// TIA Portal V20 export
// export: Created 2025-12-01T14:56:31.3857543Z, ExportSetting None, DisplayName Totally Integrated Automation Portal, DisplayVersion V20 Update 3, DisplayName TIA Portal Openness, DisplayVersion V20 Update 3, DisplayName TIA Portal Version Control Interface, DisplayVersion V20 Update 3, DisplayName STEP 7 Professional, DisplayVersion V20 Update 3, DisplayName STEP 7 Safety, DisplayVersion V20 Update 2, DisplayName WinCC Basic/Comfort/Advanced, DisplayVersion V20 Update 3, DisplayName WinCC Professional, DisplayVersion V20 Update 3, DisplayName WinCC Unified, DisplayVersion V20 Update 3
FUNCTION_BLOCK "FB438_CRTL_W_E1_S234_BLOQ_OrdJDT"   // FB438, LAD
TITLE = Control del Ramal de Salidas
{ S7_Optimized_Access := 'FALSE' }
AUTHOR : ROUTERA
NAME : 20190213
VERSION : 3.1
// stored: AutoNumber false, SetENOAutomatically false
   VAR_INPUT
      Mesa : UInt;   // Número de mesa
      En_Tension : Bool;
      pHsMx_E1 : Bool;   // pHs DE PRESENCIA de la Mesa en E1
      pHsMx_S2 : Bool;   // pHs DE AUSENCIA de la Mesa en S2
      pHsMx_S3 : Bool;   // pHs DE AUSENCIA de la Mesa en S3
      pHsMx_S4 : Bool;   // pHs DE AUSENCIA de la Mesa en S4
      Pos_WS_S2 : Bool;   // posición del desviador en S2
      Pos_WS_S3 : Bool;   // posición del desviador en S3
      Pos_WS_S4 : Bool;   // posición del desviador en S4
      Termico_E1E3 : Bool;   // Proteccion del Tx en E1E3
      Avance_Tx_Ent { ExternalVisible := 'False'} : Bool;   // Avance del Tx de entrada. Primer tramo
      Avance_Tx_Sal : Bool;   // Avance del Tx de salida.
      PTF_Sal_M2 : Bool;   // S2 >> Mesa Siguiente PTF
      NXT_Avance_S2 : Bool;   // S2 >> Mesa Siguiente avanzando
      PTF_Sal_M3 : Bool;   // S3 >> Mesa Siguiente PTF
      NXT_Avance_S3 : Bool;   // S3 >> Mesa Siguiente avanzando
      PTF_Sal_M4 : Bool;   // S4 >> Mesa Siguiente PTF
      NXT_Avance_S4 : Bool;   // S4 >> Mesa Siguiente avanzando
      F_EnvMens_Mx : Bool;   // Fin de Envio de Mensaje
      Mx_Bloq_Activo : Bool;   // Bloqueo Activo de la Mesa
      MX_FlujoPrin_S2 : Bool;   // El flujo principal es Saliendo por S2
      MX_FlujoPrin_S4 : Bool;   // El flujo principal es Saliendo por S4
      AVTF_MAnt_Mx : Bool;   // E1 >> Mesa Anterior AVTF
      Habilitar_orden_JDT : Bool := false;   // El JDT tendrá el control del cruce con orden
      Num_Cruce : UInt;   // Número de cruce.
      DB_FIFO_Cruce : UInt := 213;   // DB de la FIFO de ordenes del cruce
      Lng_FIFO_Cruce : UInt := 1;   // Longitut de la FIFO de ordenes del cruce
      Valor_Orden_S2 : Word := 16#81;   // Con que orden entra por S2
      Valor_Orden_S4 : Word := 16#82;   // Con que orden entra por S4
      MesaS2 : UInt;   // Número de mesa por S2
      MesaS3 : UInt;   // Número de mesa por S3
      MesaS4 : UInt;   // Número de mesa por S4
      V_CNT_pHsMx : UDInt := 500;   // Valor de Presencia en ms
      V_Vaciado : UDInt := 5000;   // Valor de vaciado en ms
      V_TOut_Desviador : UDInt := 2000;   // en ms
      V_TOut_Tx_Mx : UDInt := 3000;   // TimeOut de Atasco en ms
      V_CNT_ApHsMx_E1 : UDInt := 250;   // Valor de Ausencia por E1 en ms
      V_CNT_ApHsMx_S2 : UDInt := 250;   // Valor de Ausencia por S2 en ms
      V_CNT_ApHsMx_S3 : UDInt := 250;   // Valor de Ausencia por S3 en ms
      V_CNT_ApHsMx_S4 : UDInt := 250;   // Valor de Ausencia por S4 en ms
      V_Orden_bloqueo : UDInt := 3000;   // en ms
   END_VAR
   VAR_OUTPUT
      P_EnvMens_PMx : Bool;   // Permiso de Enviar Mensaje de Presencia
      Etiqueta_Jdt : UDInt;   // Etiqueta que ha sido leida
      Orden_Ejecutada_Jdt : UInt;   // Orden que se ha ejecutado
      PTF_MAnt_Mx : Bool;   // E1 >> Mesa Anterior PTF
      AVTF_Sal_M2 : Bool;   // S2 >> Mesa Siguiente AVTF
      NXT_Descarga_Act_S2 : Bool;   // S2 >> Mesa Siguiente descarga activa
      AVTF_Sal_M3 : Bool;   // S3 >> Mesa Siguiente AVTF
      NXT_Descarga_Act_S3 : Bool;   // S3 >> Mesa Siguiente descarga activa
      AVTF_Sal_M4 : Bool;   // S4 >> Mesa Siguiente AVTF
      NXT_Descarga_Act_S4 : Bool;   // S4 >> Mesa Siguiente descarga activa
   END_VAR
   VAR
      T1_ET00 : Bool;   // Reset
      T1_ET08 : Bool;
      T1_ET01 : Bool;   // Entrada Vacia
      T1_ET10 : Bool;   // Carga Entrada
      T1_ET02 : Bool;   // Entrada Cargada
      T1_ET02_JDT : Bool;
      T1_ET03 : Bool;   // Vaciando Entrada
      T1_ET20 : Bool;   // Carga Salida
      T1_ET21 : Bool;   // Salida Vacia
      T1_ET50 : Bool;   // Continuar
      T1_ET60 : Bool;   // Entrar
      T1_ET70 : Bool;   // Vaciado
      T1_ET80 : Bool;
      T1_ET110 : Bool;   // Extraer orden
      T1_ET111 : Bool;
      T1_ET112 : Bool;
      FP_ET2_JDT : Bool;
      FIFO_OK : Bool;
      TRANS_OK : Bool;
      O_Bloqueo : Bool;
      Vaciado_1 : Bool;
      PRV_CargaOK_ET03 : Bool;
      FN_ET20 : Bool;
      MemoPresenciaJDT : Bool;
      maux_fp_disparo : Bool;
      Vaciado_entrada_ok : Bool;
      Vaciado_salida_s2_ok : Bool;
      Vaciado_salida_s3_ok : Bool;
      Vaciado_salida_s4_ok : Bool;
      Maux_FN_Phs_S2 : Bool;
      mem_fn_phs_s2 : Bool;
      Maux_FN_Phs_E1 : Bool;
      mem_fn_phs_e1 : Bool;
      Maux_FP_phs_S3 : Bool;
      mem_fp_phs_s3 : Bool;
      Maux_FN_Phs_S4 : Bool;
      mem_fn_phs_s4 : Bool;
      paro : Bool;
      CNT_ERR_PHS : Int;
      TIMV_WS_E1 : UDInt;
      TIMV_WS_S2 : UDInt;
      TIMV_WS_S3 : UDInt;
      TIMV_WS_S4 : UDInt;
      TMP_Err_Piston : UDInt;
      TMP_Paro : UDInt;
      TMP_Err_Tout_avance_E : UDInt;
      TMP_Err_Tout_avance_S : UDInt;
      CNT_pHs_WS : UDInt;
      CNT_aus_s2 : UDInt;
      CNT_aus_s4 : UDInt;
      CNT_aus_e1 : UDInt;
      CNT_pres_s3 : UDInt;
      CNT_bloqueo : UDInt;
      TMP_En_tension : UDInt;
      Datos_Scanner { S7_SetPoint := 'True'} : "ROUT_Orden_Fifo_Scanner";
   END_VAR
   VAR_TEMP
      EstadoZona : "EstadoZona";   // Estado de Zona de la Mesa
      EstadoVI : "EstadosMesa";   // Estado del Vehiculo Inteliguente de la Mesa
      ConfigFB : "UDT_ConfigFB";   // Configuracion de la FB de la Mesa
      TEMP_ET00 : Bool;
      O_Salir_S3 : Bool;
      O_Salir_S2 : Bool;
      O_Salir_S4 : Bool;
      O_Vaciar : Bool;
      cnt_phs_ok : Bool;
      OK_Aus_S2 : Bool;
      OK_Aus_E1 : Bool;
      OK_Pres_S3 : Bool;
      OK_Aus_S4 : Bool;
      atasco_entrada : Bool;
      atasco_salida : Bool;
      ok_tension : Bool;
      Aux_W_Moti : Word;
      Moti_INIC : Bool;
      Moti_ERRO : Bool;
      Moti_NENC : Bool;
      Moti_NORM : Bool;
      ok_bloqueo : Bool;
      timeout_piston : Bool;
      O_S2_JDT : Bool;
      O_S3_JDT : Bool;
      O_S4_JDT : Bool;
      I_V_Ord_Salir_S2 : UInt;
      I_V_Ord_Salir_S4 : UInt;
      I_Ord_Filtrada : UInt;
      INT_ORDEN : UInt;
      Aux_W_Orden : Word;
      retval : Int;
   END_VAR
   VAR_TEMP   // added for the SCL form of the ladder/FBD networks
      _w1 : Bool;
      _w2 : Bool;
      _w3 : Bool;
      _w4 : Bool;
      _w5 : Bool;
      _w6 : Bool;
      _w7 : Bool;
   END_VAR
BEGIN

REGION Network 1: INICIALIZAR - Recoger las Variables de Estado de la Mesa
   // Se recoge - Estado_CBx
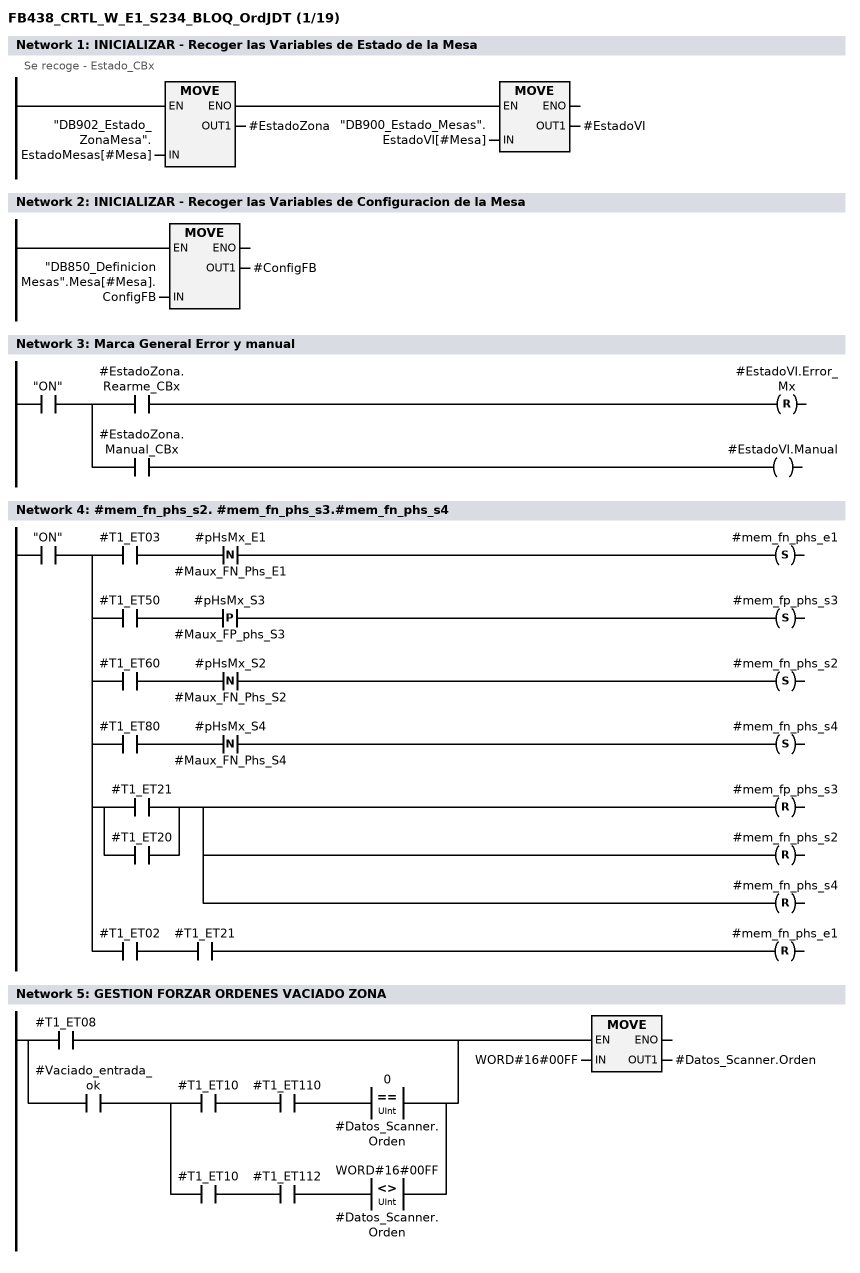
   RUNG wire#powerrail
      Move(in := "DB902_Estado_ZonaMesa".EstadoMesas[#Mesa], out1 => #EstadoZona)
      Move(in := "DB900_Estado_Mesas".EstadoVI[#Mesa], out1 => #EstadoVI)
   END_RUNG
   // the same network as SCL:
   #EstadoZona := "DB902_Estado_ZonaMesa".EstadoMesas[#Mesa];
   #EstadoVI := "DB900_Estado_Mesas".EstadoVI[#Mesa];
END_REGION

REGION Network 2: INICIALIZAR - Recoger las Variables de Configuracion de la Mesa
   RUNG wire#powerrail
      Move(in := "DB850_DefinicionMesas".Mesa[#Mesa].ConfigFB, out1 => #ConfigFB)
   END_RUNG
   // the same network as SCL:
   #ConfigFB := "DB850_DefinicionMesas".Mesa[#Mesa].ConfigFB;
END_REGION

REGION Network 3: Marca General Error y manual
   RUNG wire#powerrail
      Contact( "ON" )
      wire#w1
      Contact( #EstadoZona.Rearme_CBx )
      R_Coil( #EstadoVI.Error_Mx )
   END_RUNG
   RUNG wire#w1
      Contact( #EstadoZona.Manual_CBx )
      Coil( #EstadoVI.Manual )
   END_RUNG
   // the same network as SCL:
   IF "ON" AND #EstadoZona.Rearme_CBx THEN #EstadoVI.Error_Mx := FALSE; END_IF;
   #EstadoVI.Manual := "ON" AND #EstadoZona.Manual_CBx;
END_REGION

REGION Network 4: #mem_fn_phs_s2. #mem_fn_phs_s3.#mem_fn_phs_s4
   RUNG wire#powerrail
      Contact( "ON" )
      wire#w1
      Contact( #T1_ET03 )
      N_Contact(operand := #pHsMx_E1, bit := #Maux_FN_Phs_E1)
      S_Coil( #mem_fn_phs_e1 )
   END_RUNG
   RUNG wire#w1
      Contact( #T1_ET50 )
      P_Contact(operand := #pHsMx_S3, bit := #Maux_FP_phs_S3)
      S_Coil( #mem_fp_phs_s3 )
   END_RUNG
   RUNG wire#w1
      Contact( #T1_ET60 )
      N_Contact(operand := #pHsMx_S2, bit := #Maux_FN_Phs_S2)
      S_Coil( #mem_fn_phs_s2 )
   END_RUNG
   RUNG wire#w1
      Contact( #T1_ET80 )
      N_Contact(operand := #pHsMx_S4, bit := #Maux_FN_Phs_S4)
      S_Coil( #mem_fn_phs_s4 )
   END_RUNG
   RUNG wire#w1
      Contact( #T1_ET21 )
      wire#w2
      R_Coil( #mem_fp_phs_s3 )
   END_RUNG
   RUNG wire#w1
      Contact( #T1_ET20 )
   END_RUNG wire#w2
   RUNG wire#w2
      R_Coil( #mem_fn_phs_s2 )
   END_RUNG
   RUNG wire#w2
      R_Coil( #mem_fn_phs_s4 )
   END_RUNG
   RUNG wire#w1
      Contact( #T1_ET02 )
      Contact( #T1_ET21 )
      R_Coil( #mem_fn_phs_e1 )
   END_RUNG
   // the same network as SCL:
   #_w1 := "ON" AND #T1_ET03 AND NOT #pHsMx_E1 AND #Maux_FN_Phs_E1;   // falling edge of #pHsMx_E1
   #Maux_FN_Phs_E1 := #pHsMx_E1;
   IF #_w1 THEN #mem_fn_phs_e1 := TRUE; END_IF;
   #_w2 := "ON" AND #T1_ET50 AND #pHsMx_S3 AND NOT #Maux_FP_phs_S3;   // rising edge of #pHsMx_S3
   #Maux_FP_phs_S3 := #pHsMx_S3;
   IF #_w2 THEN #mem_fp_phs_s3 := TRUE; END_IF;
   #_w3 := "ON" AND #T1_ET60 AND NOT #pHsMx_S2 AND #Maux_FN_Phs_S2;   // falling edge of #pHsMx_S2
   #Maux_FN_Phs_S2 := #pHsMx_S2;
   IF #_w3 THEN #mem_fn_phs_s2 := TRUE; END_IF;
   #_w4 := "ON" AND #T1_ET80 AND NOT #pHsMx_S4 AND #Maux_FN_Phs_S4;   // falling edge of #pHsMx_S4
   #Maux_FN_Phs_S4 := #pHsMx_S4;
   IF #_w4 THEN #mem_fn_phs_s4 := TRUE; END_IF;
   IF "ON" AND (#T1_ET21 OR #T1_ET20) THEN
       #mem_fp_phs_s3 := FALSE;
       #mem_fn_phs_s2 := FALSE;
       #mem_fn_phs_s4 := FALSE;
   END_IF;
   IF "ON" AND #T1_ET02 AND #T1_ET21 THEN #mem_fn_phs_e1 := FALSE; END_IF;
END_REGION

REGION Network 5: GESTION FORZAR ORDENES VACIADO ZONA
   RUNG wire#powerrail
      Contact( #T1_ET08 )
      wire#w1
      { S7_GenerateENO := "TRUE" } Move(in := WORD#16#00FF, out1 => #Datos_Scanner.Orden)
   END_RUNG
   RUNG wire#powerrail
      Contact( #Vaciado_entrada_ok )
      wire#w2
      Contact( #T1_ET10 )
      Contact( #T1_ET110 )
      { S7_Templates := "SrcType := UInt" } EQ_Contact(in1 := 0, in2 := #Datos_Scanner.Orden)
   END_RUNG wire#w1
   RUNG wire#w2
      Contact( #T1_ET10 )
      Contact( #T1_ET112 )
      { S7_Templates := "SrcType := UInt" } NE_Contact(in1 := WORD#16#00FF, in2 := #Datos_Scanner.Orden)
   END_RUNG wire#w1
   // the same network as SCL:
   IF #T1_ET08 OR (#Vaciado_entrada_ok AND ((#T1_ET10 AND #T1_ET110 AND (0 = #Datos_Scanner.Orden)) OR (#T1_ET10 AND #T1_ET112 AND (WORD#16#00FF <> #Datos_Scanner.Orden)))) THEN
       #Datos_Scanner.Orden := WORD#16#00FF;
   END_IF;
END_REGION

REGION Network 6: Ordenes del JDT
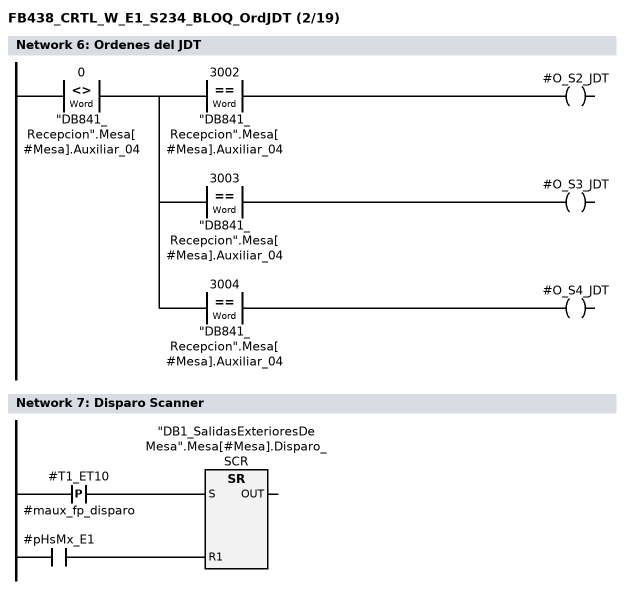
   RUNG wire#powerrail
      { S7_Templates := "SrcType := Word" } NE_Contact(in1 := 0, in2 := "DB841_Recepcion".Mesa[#Mesa].Auxiliar_04)
      wire#w1
      { S7_Templates := "SrcType := Word" } EQ_Contact(in1 := 3002, in2 := "DB841_Recepcion".Mesa[#Mesa].Auxiliar_04)
      Coil( #O_S2_JDT )
   END_RUNG
   RUNG wire#w1
      { S7_Templates := "SrcType := Word" } EQ_Contact(in1 := 3003, in2 := "DB841_Recepcion".Mesa[#Mesa].Auxiliar_04)
      Coil( #O_S3_JDT )
   END_RUNG
   RUNG wire#w1
      { S7_Templates := "SrcType := Word" } EQ_Contact(in1 := 3004, in2 := "DB841_Recepcion".Mesa[#Mesa].Auxiliar_04)
      Coil( #O_S4_JDT )
   END_RUNG
   // the same network as SCL:
   #_w1 := 0 <> "DB841_Recepcion".Mesa[#Mesa].Auxiliar_04;
   #O_S2_JDT := #_w1 AND (3002 = "DB841_Recepcion".Mesa[#Mesa].Auxiliar_04);
   #O_S3_JDT := #_w1 AND (3003 = "DB841_Recepcion".Mesa[#Mesa].Auxiliar_04);
   #O_S4_JDT := #_w1 AND (3004 = "DB841_Recepcion".Mesa[#Mesa].Auxiliar_04);
END_REGION

REGION Network 7: Disparo Scanner
   RUNG wire#powerrail
      P_Contact(operand := #T1_ET10, bit := #maux_fp_disparo)
      S_SR(operand := "DB1_SalidasExterioresDeMesa".Mesa[#Mesa].Disparo_SCR, r1 := wire#w1)
   END_RUNG
   RUNG wire#powerrail
      Contact( #pHsMx_E1 )
   END_RUNG wire#w1
   // the same network as SCL:
   #_w1 := #T1_ET10 AND NOT #maux_fp_disparo;   // rising edge of #T1_ET10
   #maux_fp_disparo := #T1_ET10;
   IF #_w1 THEN
       "DB1_SalidasExterioresDeMesa".Mesa[#Mesa].Disparo_SCR := TRUE;   // SR flip-flop
   END_IF;
   IF #pHsMx_E1 THEN "DB1_SalidasExterioresDeMesa".Mesa[#Mesa].Disparo_SCR := FALSE; END_IF;
END_REGION

REGION Network 8: extraer orden
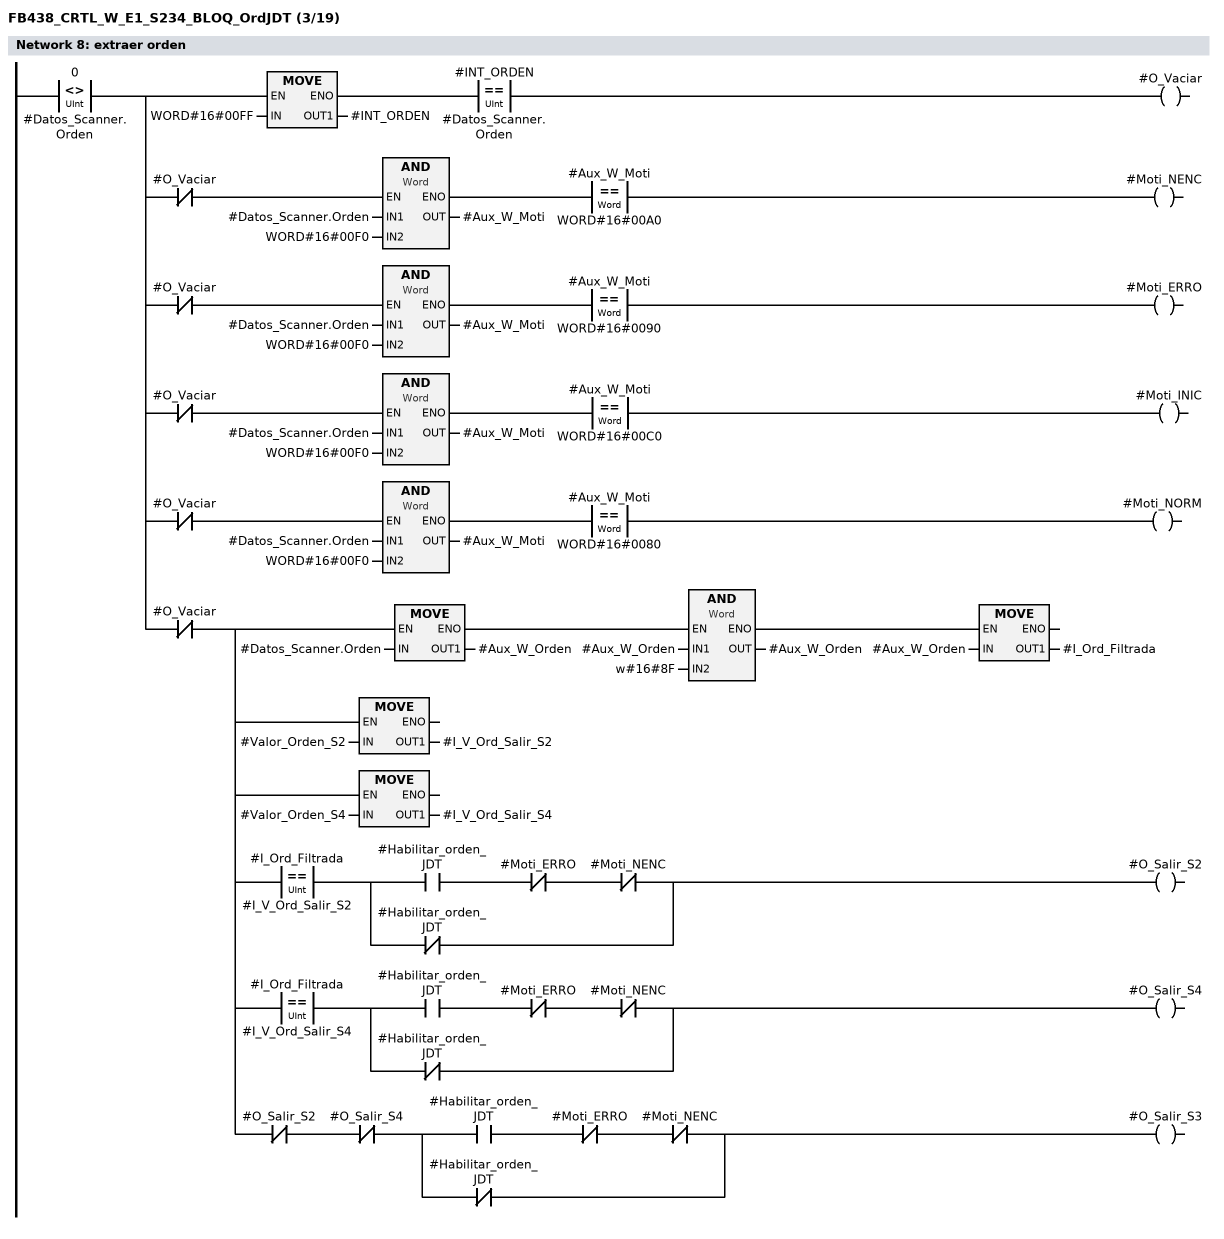
   RUNG wire#powerrail
      { S7_Templates := "SrcType := UInt" } NE_Contact(in1 := 0, in2 := #Datos_Scanner.Orden)
      wire#w1
      { S7_GenerateENO := "TRUE" } Move(in := WORD#16#00FF, out1 => #INT_ORDEN)
      { S7_Templates := "SrcType := UInt" } EQ_Contact(in1 := #INT_ORDEN, in2 := #Datos_Scanner.Orden)
      Coil( #O_Vaciar )
   END_RUNG
   RUNG wire#w1
      I_Contact( #O_Vaciar )
      { S7_Templates := "SrcType := Word"; S7_GenerateENO := "TRUE" } And(in1 := #Datos_Scanner.Orden, in2 := WORD#16#00F0, out => #Aux_W_Moti)
      { S7_Templates := "SrcType := Word" } EQ_Contact(in1 := #Aux_W_Moti, in2 := WORD#16#00A0)
      Coil( #Moti_NENC )
   END_RUNG
   RUNG wire#w1
      I_Contact( #O_Vaciar )
      { S7_Templates := "SrcType := Word"; S7_GenerateENO := "TRUE" } And(in1 := #Datos_Scanner.Orden, in2 := WORD#16#00F0, out => #Aux_W_Moti)
      { S7_Templates := "SrcType := Word" } EQ_Contact(in1 := #Aux_W_Moti, in2 := WORD#16#0090)
      Coil( #Moti_ERRO )
   END_RUNG
   RUNG wire#w1
      I_Contact( #O_Vaciar )
      { S7_Templates := "SrcType := Word"; S7_GenerateENO := "TRUE" } And(in1 := #Datos_Scanner.Orden, in2 := WORD#16#00F0, out => #Aux_W_Moti)
      { S7_Templates := "SrcType := Word" } EQ_Contact(in1 := #Aux_W_Moti, in2 := WORD#16#00C0)
      Coil( #Moti_INIC )
   END_RUNG
   RUNG wire#w1
      I_Contact( #O_Vaciar )
      { S7_Templates := "SrcType := Word"; S7_GenerateENO := "TRUE" } And(in1 := #Datos_Scanner.Orden, in2 := WORD#16#00F0, out => #Aux_W_Moti)
      { S7_Templates := "SrcType := Word" } EQ_Contact(in1 := #Aux_W_Moti, in2 := WORD#16#0080)
      Coil( #Moti_NORM )
   END_RUNG
   RUNG wire#w1
      I_Contact( #O_Vaciar )
      wire#w2
      { S7_GenerateENO := "TRUE" } Move(in := #Datos_Scanner.Orden, out1 => #Aux_W_Orden)
      { S7_Templates := "SrcType := Word"; S7_GenerateENO := "TRUE" } And(in1 := #Aux_W_Orden, in2 := w#16#8F, out => #Aux_W_Orden)
      { S7_GenerateENO := "TRUE" } Move(in := #Aux_W_Orden, out1 => #I_Ord_Filtrada)
   END_RUNG
   RUNG wire#w2
      { S7_GenerateENO := "TRUE" } Move(in := #Valor_Orden_S2, out1 => #I_V_Ord_Salir_S2)
   END_RUNG
   RUNG wire#w2
      { S7_GenerateENO := "TRUE" } Move(in := #Valor_Orden_S4, out1 => #I_V_Ord_Salir_S4)
   END_RUNG
   RUNG wire#w2
      { S7_Templates := "SrcType := UInt" } EQ_Contact(in1 := #I_Ord_Filtrada, in2 := #I_V_Ord_Salir_S2)
      wire#w3
      Contact( #Habilitar_orden_JDT )
      I_Contact( #Moti_ERRO )
      I_Contact( #Moti_NENC )
      wire#w4
      Coil( #O_Salir_S2 )
   END_RUNG
   RUNG wire#w3
      I_Contact( #Habilitar_orden_JDT )
   END_RUNG wire#w4
   RUNG wire#w2
      { S7_Templates := "SrcType := UInt" } EQ_Contact(in1 := #I_Ord_Filtrada, in2 := #I_V_Ord_Salir_S4)
      wire#w5
      Contact( #Habilitar_orden_JDT )
      I_Contact( #Moti_ERRO )
      I_Contact( #Moti_NENC )
      wire#w6
      Coil( #O_Salir_S4 )
   END_RUNG
   RUNG wire#w5
      I_Contact( #Habilitar_orden_JDT )
   END_RUNG wire#w6
   RUNG wire#w2
      I_Contact( #O_Salir_S2 )
      I_Contact( #O_Salir_S4 )
      wire#w7
      Contact( #Habilitar_orden_JDT )
      I_Contact( #Moti_ERRO )
      I_Contact( #Moti_NENC )
      wire#w8
      Coil( #O_Salir_S3 )
   END_RUNG
   RUNG wire#w7
      I_Contact( #Habilitar_orden_JDT )
   END_RUNG wire#w8
   // the same network as SCL:
   // ENO of a box is taken as its EN; it also drops when the box reports an error
   #_w1 := 0 <> #Datos_Scanner.Orden;
   IF #_w1 THEN #INT_ORDEN := WORD#16#00FF; END_IF;
   #O_Vaciar := #_w1 AND (#INT_ORDEN = #Datos_Scanner.Orden);
   #_w2 := #_w1 AND NOT #O_Vaciar;
   IF #_w2 THEN #Aux_W_Moti := #Datos_Scanner.Orden AND WORD#16#00F0; END_IF;
   #Moti_NENC := #_w2 AND (#Aux_W_Moti = WORD#16#00A0);
   #_w3 := #_w1 AND NOT #O_Vaciar;
   IF #_w3 THEN #Aux_W_Moti := #Datos_Scanner.Orden AND WORD#16#00F0; END_IF;
   #Moti_ERRO := #_w3 AND (#Aux_W_Moti = WORD#16#0090);
   #_w4 := #_w1 AND NOT #O_Vaciar;
   IF #_w4 THEN #Aux_W_Moti := #Datos_Scanner.Orden AND WORD#16#00F0; END_IF;
   #Moti_INIC := #_w4 AND (#Aux_W_Moti = WORD#16#00C0);
   #_w5 := #_w1 AND NOT #O_Vaciar;
   IF #_w5 THEN #Aux_W_Moti := #Datos_Scanner.Orden AND WORD#16#00F0; END_IF;
   #Moti_NORM := #_w5 AND (#Aux_W_Moti = WORD#16#0080);
   #_w6 := #_w1 AND NOT #O_Vaciar;
   IF #_w6 THEN
       #Aux_W_Orden := #Datos_Scanner.Orden;
       #Aux_W_Orden := #Aux_W_Orden AND w#16#8F;
       #I_Ord_Filtrada := #Aux_W_Orden;
       #I_V_Ord_Salir_S2 := #Valor_Orden_S2;
       #I_V_Ord_Salir_S4 := #Valor_Orden_S4;
   END_IF;
   #O_Salir_S2 := #_w6 AND (#I_Ord_Filtrada = #I_V_Ord_Salir_S2) AND ((#Habilitar_orden_JDT AND NOT #Moti_ERRO AND NOT #Moti_NENC) OR NOT #Habilitar_orden_JDT);
   #O_Salir_S4 := #_w6 AND (#I_Ord_Filtrada = #I_V_Ord_Salir_S4) AND ((#Habilitar_orden_JDT AND NOT #Moti_ERRO AND NOT #Moti_NENC) OR NOT #Habilitar_orden_JDT);
   #O_Salir_S3 := #_w6 AND NOT #O_Salir_S2 AND NOT #O_Salir_S4 AND ((#Habilitar_orden_JDT AND NOT #Moti_ERRO AND NOT #Moti_NENC) OR NOT #Habilitar_orden_JDT);
END_REGION

REGION Network 9: cnt presencia
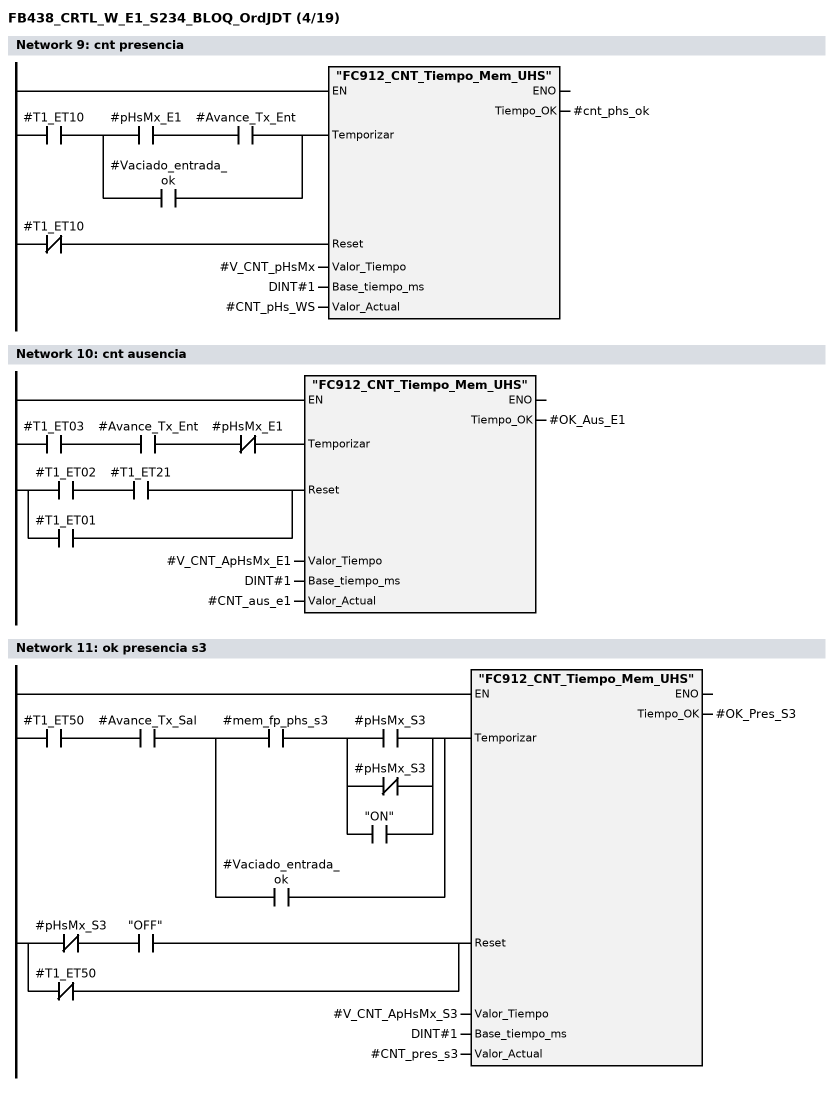
   RUNG wire#powerrail
      "FC912_CNT_Tiempo_Mem_UHS"(Temporizar := wire#w2, Reset := wire#w3, Valor_Tiempo := #V_CNT_pHsMx, Base_tiempo_ms := DINT#1, Valor_Actual := #CNT_pHs_WS, Tiempo_OK => #cnt_phs_ok)
   END_RUNG
   RUNG wire#powerrail
      Contact( #T1_ET10 )
      wire#w1
      Contact( #pHsMx_E1 )
      Contact( #Avance_Tx_Ent )
   END_RUNG wire#w2
   RUNG wire#w1
      Contact( #Vaciado_entrada_ok )
   END_RUNG wire#w2
   RUNG wire#powerrail
      I_Contact( #T1_ET10 )
   END_RUNG wire#w3
   // the same network as SCL:
   "FC912_CNT_Tiempo_Mem_UHS"(Temporizar := #T1_ET10 AND ((#pHsMx_E1 AND #Avance_Tx_Ent) OR #Vaciado_entrada_ok),
                           Reset := NOT #T1_ET10,
                           Valor_Tiempo := #V_CNT_pHsMx,
                           Base_tiempo_ms := DINT#1,
                           Valor_Actual := #CNT_pHs_WS,
                           Tiempo_OK => #cnt_phs_ok);
END_REGION

REGION Network 10: cnt ausencia
   RUNG wire#powerrail
      "FC912_CNT_Tiempo_Mem_UHS"(Temporizar := wire#w1, Reset := wire#w2, Valor_Tiempo := #V_CNT_ApHsMx_E1, Base_tiempo_ms := DINT#1, Valor_Actual := #CNT_aus_e1, Tiempo_OK => #OK_Aus_E1)
   END_RUNG
   RUNG wire#powerrail
      Contact( #T1_ET03 )
      Contact( #Avance_Tx_Ent )
      I_Contact( #pHsMx_E1 )
   END_RUNG wire#w1
   RUNG wire#powerrail
      Contact( #T1_ET02 )
      Contact( #T1_ET21 )
   END_RUNG wire#w2
   RUNG wire#powerrail
      Contact( #T1_ET01 )
   END_RUNG wire#w2
   // the same network as SCL:
   "FC912_CNT_Tiempo_Mem_UHS"(Temporizar := #T1_ET03 AND #Avance_Tx_Ent AND NOT #pHsMx_E1,
                           Reset := (#T1_ET02 AND #T1_ET21) OR #T1_ET01,
                           Valor_Tiempo := #V_CNT_ApHsMx_E1,
                           Base_tiempo_ms := DINT#1,
                           Valor_Actual := #CNT_aus_e1,
                           Tiempo_OK => #OK_Aus_E1);
END_REGION

REGION Network 11: ok presencia s3
   RUNG wire#powerrail
      "FC912_CNT_Tiempo_Mem_UHS"(Temporizar := wire#w3, Reset := wire#w4, Valor_Tiempo := #V_CNT_ApHsMx_S3, Base_tiempo_ms := DINT#1, Valor_Actual := #CNT_pres_s3, Tiempo_OK => #OK_Pres_S3)
   END_RUNG
   RUNG wire#powerrail
      Contact( #T1_ET50 )
      Contact( #Avance_Tx_Sal )
      wire#w1
      Contact( #mem_fp_phs_s3 )
      wire#w2
      Contact( #pHsMx_S3 )
   END_RUNG wire#w3
   RUNG wire#w2
      I_Contact( #pHsMx_S3 )
   END_RUNG wire#w3
   RUNG wire#w2
      Contact( "ON" )
   END_RUNG wire#w3
   RUNG wire#w1
      Contact( #Vaciado_entrada_ok )
   END_RUNG wire#w3
   RUNG wire#powerrail
      I_Contact( #pHsMx_S3 )
      Contact( "OFF" )
   END_RUNG wire#w4
   RUNG wire#powerrail
      I_Contact( #T1_ET50 )
   END_RUNG wire#w4
   // the same network as SCL:
   "FC912_CNT_Tiempo_Mem_UHS"(Temporizar := #T1_ET50 AND #Avance_Tx_Sal AND ((#mem_fp_phs_s3 AND (#pHsMx_S3 OR NOT #pHsMx_S3 OR "ON")) OR #Vaciado_entrada_ok),
                           Reset := (NOT #pHsMx_S3 AND "OFF") OR NOT #T1_ET50,
                           Valor_Tiempo := #V_CNT_ApHsMx_S3,
                           Base_tiempo_ms := DINT#1,
                           Valor_Actual := #CNT_pres_s3,
                           Tiempo_OK => #OK_Pres_S3);
END_REGION

REGION Network 12: ok ausencia s2
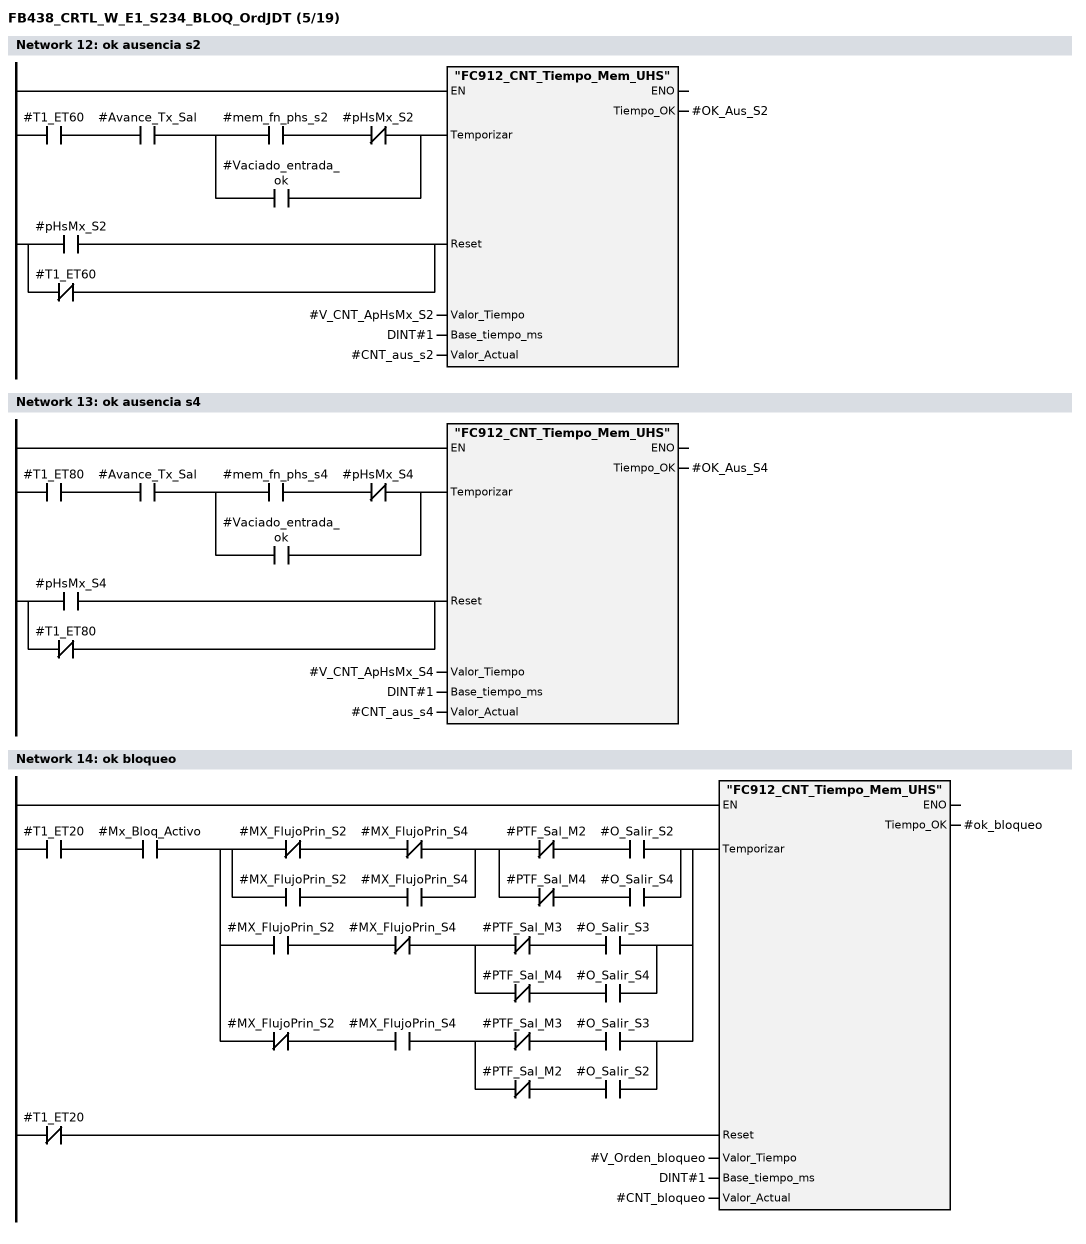
   RUNG wire#powerrail
      "FC912_CNT_Tiempo_Mem_UHS"(Temporizar := wire#w2, Reset := wire#w3, Valor_Tiempo := #V_CNT_ApHsMx_S2, Base_tiempo_ms := DINT#1, Valor_Actual := #CNT_aus_s2, Tiempo_OK => #OK_Aus_S2)
   END_RUNG
   RUNG wire#powerrail
      Contact( #T1_ET60 )
      Contact( #Avance_Tx_Sal )
      wire#w1
      Contact( #mem_fn_phs_s2 )
      I_Contact( #pHsMx_S2 )
   END_RUNG wire#w2
   RUNG wire#w1
      Contact( #Vaciado_entrada_ok )
   END_RUNG wire#w2
   RUNG wire#powerrail
      Contact( #pHsMx_S2 )
   END_RUNG wire#w3
   RUNG wire#powerrail
      I_Contact( #T1_ET60 )
   END_RUNG wire#w3
   // the same network as SCL:
   "FC912_CNT_Tiempo_Mem_UHS"(Temporizar := #T1_ET60 AND #Avance_Tx_Sal AND ((#mem_fn_phs_s2 AND NOT #pHsMx_S2) OR #Vaciado_entrada_ok),
                           Reset := #pHsMx_S2 OR NOT #T1_ET60,
                           Valor_Tiempo := #V_CNT_ApHsMx_S2,
                           Base_tiempo_ms := DINT#1,
                           Valor_Actual := #CNT_aus_s2,
                           Tiempo_OK => #OK_Aus_S2);
END_REGION

REGION Network 13: ok ausencia s4
   RUNG wire#powerrail
      "FC912_CNT_Tiempo_Mem_UHS"(Temporizar := wire#w2, Reset := wire#w3, Valor_Tiempo := #V_CNT_ApHsMx_S4, Base_tiempo_ms := DINT#1, Valor_Actual := #CNT_aus_s4, Tiempo_OK => #OK_Aus_S4)
   END_RUNG
   RUNG wire#powerrail
      Contact( #T1_ET80 )
      Contact( #Avance_Tx_Sal )
      wire#w1
      Contact( #mem_fn_phs_s4 )
      I_Contact( #pHsMx_S4 )
   END_RUNG wire#w2
   RUNG wire#w1
      Contact( #Vaciado_entrada_ok )
   END_RUNG wire#w2
   RUNG wire#powerrail
      Contact( #pHsMx_S4 )
   END_RUNG wire#w3
   RUNG wire#powerrail
      I_Contact( #T1_ET80 )
   END_RUNG wire#w3
   // the same network as SCL:
   "FC912_CNT_Tiempo_Mem_UHS"(Temporizar := #T1_ET80 AND #Avance_Tx_Sal AND ((#mem_fn_phs_s4 AND NOT #pHsMx_S4) OR #Vaciado_entrada_ok),
                           Reset := #pHsMx_S4 OR NOT #T1_ET80,
                           Valor_Tiempo := #V_CNT_ApHsMx_S4,
                           Base_tiempo_ms := DINT#1,
                           Valor_Actual := #CNT_aus_s4,
                           Tiempo_OK => #OK_Aus_S4);
END_REGION

REGION Network 14: ok bloqueo
   RUNG wire#powerrail
      "FC912_CNT_Tiempo_Mem_UHS"(Temporizar := wire#w5, Reset := wire#w6, Valor_Tiempo := #V_Orden_bloqueo, Base_tiempo_ms := DINT#1, Valor_Actual := #CNT_bloqueo, Tiempo_OK => #ok_bloqueo)
   END_RUNG
   RUNG wire#powerrail
      Contact( #T1_ET20 )
      Contact( #Mx_Bloq_Activo )
      wire#w1
      I_Contact( #MX_FlujoPrin_S2 )
      I_Contact( #MX_FlujoPrin_S4 )
      wire#w2
      I_Contact( #PTF_Sal_M2 )
      Contact( #O_Salir_S2 )
   END_RUNG wire#w5
   RUNG wire#w1
      Contact( #MX_FlujoPrin_S2 )
      Contact( #MX_FlujoPrin_S4 )
   END_RUNG wire#w2
   RUNG wire#w2
      I_Contact( #PTF_Sal_M4 )
      Contact( #O_Salir_S4 )
   END_RUNG wire#w5
   RUNG wire#w1
      Contact( #MX_FlujoPrin_S2 )
      I_Contact( #MX_FlujoPrin_S4 )
      wire#w3
      I_Contact( #PTF_Sal_M3 )
      Contact( #O_Salir_S3 )
   END_RUNG wire#w5
   RUNG wire#w3
      I_Contact( #PTF_Sal_M4 )
      Contact( #O_Salir_S4 )
   END_RUNG wire#w5
   RUNG wire#w1
      I_Contact( #MX_FlujoPrin_S2 )
      Contact( #MX_FlujoPrin_S4 )
      wire#w4
      I_Contact( #PTF_Sal_M3 )
      Contact( #O_Salir_S3 )
   END_RUNG wire#w5
   RUNG wire#w4
      I_Contact( #PTF_Sal_M2 )
      Contact( #O_Salir_S2 )
   END_RUNG wire#w5
   RUNG wire#powerrail
      I_Contact( #T1_ET20 )
   END_RUNG wire#w6
   // the same network as SCL:
   "FC912_CNT_Tiempo_Mem_UHS"(Temporizar := #T1_ET20 AND #Mx_Bloq_Activo AND ((((NOT #MX_FlujoPrin_S2 AND NOT #MX_FlujoPrin_S4) OR (#MX_FlujoPrin_S2 AND #MX_FlujoPrin_S4)) AND ((NOT #PTF_Sal_M2 AND #O_Salir_S2) OR (NOT #PTF_Sal_M4 AND #O_Salir_S4))) OR (#MX_FlujoPrin_S2 AND NOT #MX_FlujoPrin_S4 AND ((NOT #PTF_Sal_M3 AND #O_Salir_S3) OR (NOT #PTF_Sal_M4 AND #O_Salir_S4))) OR (NOT #MX_FlujoPrin_S2 AND #MX_FlujoPrin_S4 AND ((NOT #PTF_Sal_M3 AND #O_Salir_S3) OR (NOT #PTF_Sal_M2 AND #O_Salir_S2)))),
                           Reset := NOT #T1_ET20,
                           Valor_Tiempo := #V_Orden_bloqueo,
                           Base_tiempo_ms := DINT#1,
                           Valor_Actual := #CNT_bloqueo,
                           Tiempo_OK => #ok_bloqueo);
END_REGION

REGION Network 15: TIMV_WS_E1
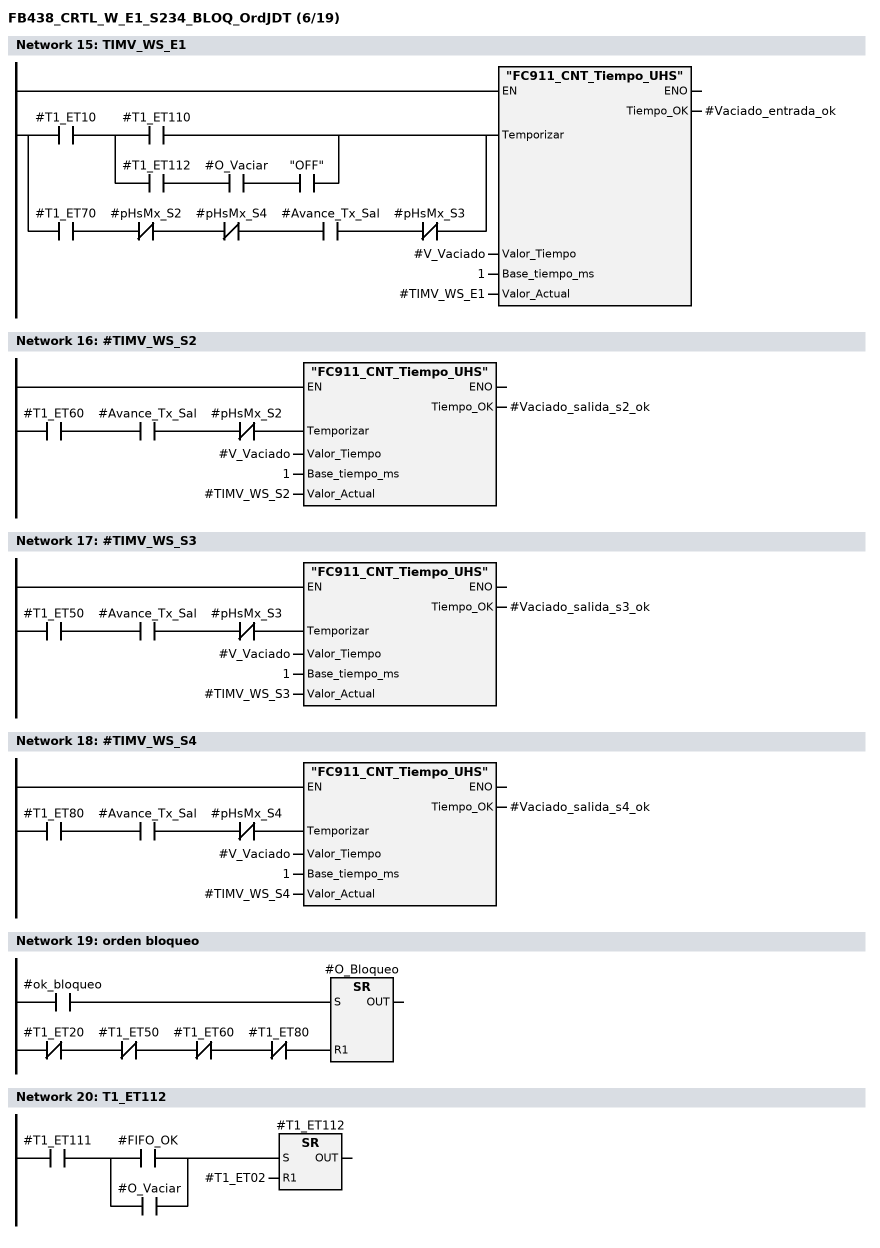
   RUNG wire#powerrail
      "FC911_CNT_Tiempo_UHS"(Temporizar := wire#w2, Valor_Tiempo := #V_Vaciado, Base_tiempo_ms := 1, Valor_Actual := #TIMV_WS_E1, Tiempo_OK => #Vaciado_entrada_ok)
   END_RUNG
   RUNG wire#powerrail
      Contact( #T1_ET10 )
      wire#w1
      Contact( #T1_ET110 )
   END_RUNG wire#w2
   RUNG wire#w1
      Contact( #T1_ET112 )
      Contact( #O_Vaciar )
      Contact( "OFF" )
   END_RUNG wire#w2
   RUNG wire#powerrail
      Contact( #T1_ET70 )
      I_Contact( #pHsMx_S2 )
      I_Contact( #pHsMx_S4 )
      Contact( #Avance_Tx_Sal )
      I_Contact( #pHsMx_S3 )
   END_RUNG wire#w2
   // the same network as SCL:
   "FC911_CNT_Tiempo_UHS"(Temporizar := (#T1_ET10 AND (#T1_ET110 OR (#T1_ET112 AND #O_Vaciar AND "OFF"))) OR (#T1_ET70 AND NOT #pHsMx_S2 AND NOT #pHsMx_S4 AND #Avance_Tx_Sal AND NOT #pHsMx_S3),
                          Valor_Tiempo := #V_Vaciado,
                          Base_tiempo_ms := 1,
                          Valor_Actual := #TIMV_WS_E1,
                          Tiempo_OK => #Vaciado_entrada_ok);
END_REGION

REGION Network 16: #TIMV_WS_S2
   RUNG wire#powerrail
      "FC911_CNT_Tiempo_UHS"(Temporizar := wire#w1, Valor_Tiempo := #V_Vaciado, Base_tiempo_ms := 1, Valor_Actual := #TIMV_WS_S2, Tiempo_OK => #Vaciado_salida_s2_ok)
   END_RUNG
   RUNG wire#powerrail
      Contact( #T1_ET60 )
      Contact( #Avance_Tx_Sal )
      I_Contact( #pHsMx_S2 )
   END_RUNG wire#w1
   // the same network as SCL:
   "FC911_CNT_Tiempo_UHS"(Temporizar := #T1_ET60 AND #Avance_Tx_Sal AND NOT #pHsMx_S2,
                          Valor_Tiempo := #V_Vaciado,
                          Base_tiempo_ms := 1,
                          Valor_Actual := #TIMV_WS_S2,
                          Tiempo_OK => #Vaciado_salida_s2_ok);
END_REGION

REGION Network 17: #TIMV_WS_S3
   RUNG wire#powerrail
      "FC911_CNT_Tiempo_UHS"(Temporizar := wire#w1, Valor_Tiempo := #V_Vaciado, Base_tiempo_ms := 1, Valor_Actual := #TIMV_WS_S3, Tiempo_OK => #Vaciado_salida_s3_ok)
   END_RUNG
   RUNG wire#powerrail
      Contact( #T1_ET50 )
      Contact( #Avance_Tx_Sal )
      I_Contact( #pHsMx_S3 )
   END_RUNG wire#w1
   // the same network as SCL:
   "FC911_CNT_Tiempo_UHS"(Temporizar := #T1_ET50 AND #Avance_Tx_Sal AND NOT #pHsMx_S3,
                          Valor_Tiempo := #V_Vaciado,
                          Base_tiempo_ms := 1,
                          Valor_Actual := #TIMV_WS_S3,
                          Tiempo_OK => #Vaciado_salida_s3_ok);
END_REGION

REGION Network 18: #TIMV_WS_S4
   RUNG wire#powerrail
      "FC911_CNT_Tiempo_UHS"(Temporizar := wire#w1, Valor_Tiempo := #V_Vaciado, Base_tiempo_ms := 1, Valor_Actual := #TIMV_WS_S4, Tiempo_OK => #Vaciado_salida_s4_ok)
   END_RUNG
   RUNG wire#powerrail
      Contact( #T1_ET80 )
      Contact( #Avance_Tx_Sal )
      I_Contact( #pHsMx_S4 )
   END_RUNG wire#w1
   // the same network as SCL:
   "FC911_CNT_Tiempo_UHS"(Temporizar := #T1_ET80 AND #Avance_Tx_Sal AND NOT #pHsMx_S4,
                          Valor_Tiempo := #V_Vaciado,
                          Base_tiempo_ms := 1,
                          Valor_Actual := #TIMV_WS_S4,
                          Tiempo_OK => #Vaciado_salida_s4_ok);
END_REGION

REGION Network 19: orden bloqueo
   RUNG wire#powerrail
      Contact( #ok_bloqueo )
      S_SR(operand := #O_Bloqueo, r1 := wire#w1)
   END_RUNG
   RUNG wire#powerrail
      I_Contact( #T1_ET20 )
      I_Contact( #T1_ET50 )
      I_Contact( #T1_ET60 )
      I_Contact( #T1_ET80 )
   END_RUNG wire#w1
   // the same network as SCL:
   IF #ok_bloqueo THEN
       #O_Bloqueo := TRUE;   // SR flip-flop
   END_IF;
   IF NOT #T1_ET20 AND NOT #T1_ET50 AND NOT #T1_ET60 AND NOT #T1_ET80 THEN #O_Bloqueo := FALSE; END_IF;
END_REGION

REGION Network 20: T1_ET112
   RUNG wire#powerrail
      Contact( #T1_ET111 )
      wire#w1
      Contact( #FIFO_OK )
      wire#w2
      S_SR(operand := #T1_ET112, r1 := #T1_ET02)
   END_RUNG
   RUNG wire#w1
      Contact( #O_Vaciar )
   END_RUNG wire#w2
   // the same network as SCL:
   IF #T1_ET111 AND (#FIFO_OK OR #O_Vaciar) THEN
       #T1_ET112 := TRUE;   // SR flip-flop
   END_IF;
   IF #T1_ET02 THEN #T1_ET112 := FALSE; END_IF;
END_REGION

REGION Network 21: T1_ET111
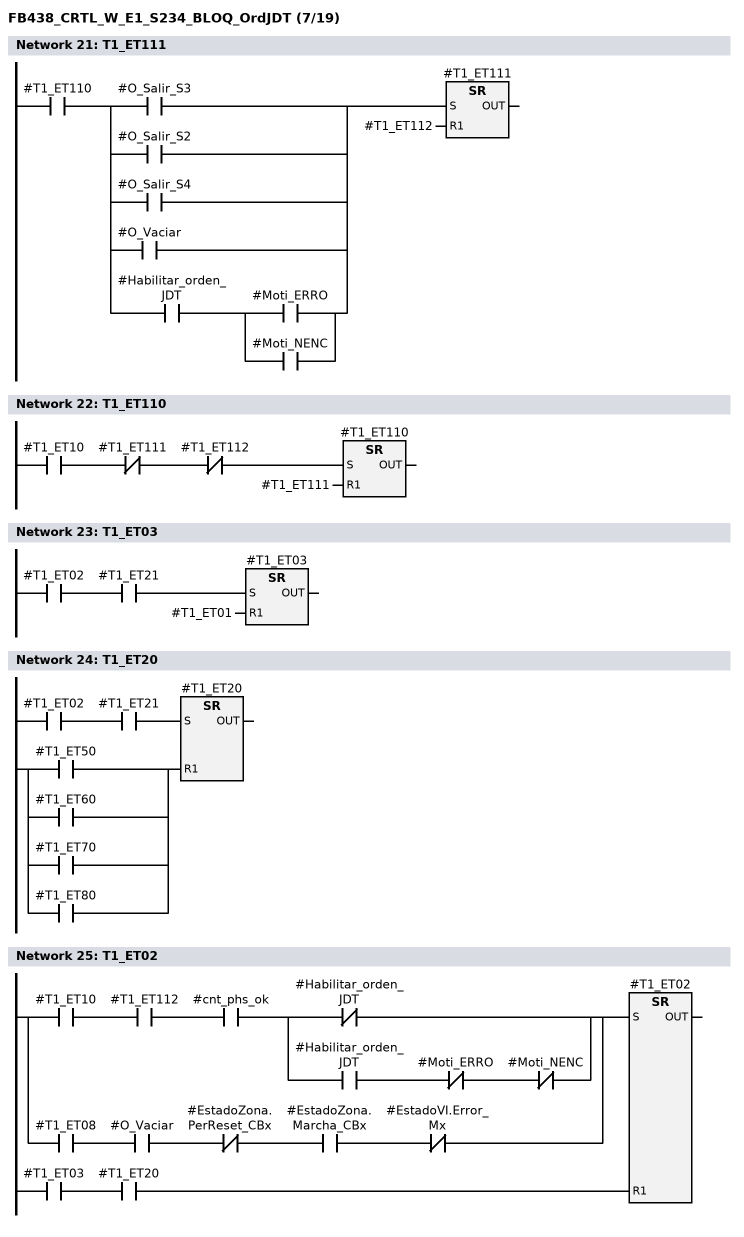
   RUNG wire#powerrail
      Contact( #T1_ET110 )
      wire#w1
      Contact( #O_Salir_S3 )
      wire#w2
      S_SR(operand := #T1_ET111, r1 := #T1_ET112)
   END_RUNG
   RUNG wire#w1
      Contact( #O_Salir_S2 )
   END_RUNG wire#w2
   RUNG wire#w1
      Contact( #O_Salir_S4 )
   END_RUNG wire#w2
   RUNG wire#w1
      Contact( #O_Vaciar )
   END_RUNG wire#w2
   RUNG wire#w1
      Contact( #Habilitar_orden_JDT )
      wire#w3
      Contact( #Moti_ERRO )
   END_RUNG wire#w2
   RUNG wire#w3
      Contact( #Moti_NENC )
   END_RUNG wire#w2
   // the same network as SCL:
   IF #T1_ET110 AND (#O_Salir_S3 OR #O_Salir_S2 OR #O_Salir_S4 OR #O_Vaciar OR (#Habilitar_orden_JDT AND (#Moti_ERRO OR #Moti_NENC))) THEN
       #T1_ET111 := TRUE;   // SR flip-flop
   END_IF;
   IF #T1_ET112 THEN #T1_ET111 := FALSE; END_IF;
END_REGION

REGION Network 22: T1_ET110
   RUNG wire#powerrail
      Contact( #T1_ET10 )
      I_Contact( #T1_ET111 )
      I_Contact( #T1_ET112 )
      S_SR(operand := #T1_ET110, r1 := #T1_ET111)
   END_RUNG
   // the same network as SCL:
   IF #T1_ET10 AND NOT #T1_ET111 AND NOT #T1_ET112 THEN
       #T1_ET110 := TRUE;   // SR flip-flop
   END_IF;
   IF #T1_ET111 THEN #T1_ET110 := FALSE; END_IF;
END_REGION

REGION Network 23: T1_ET03
   RUNG wire#powerrail
      Contact( #T1_ET02 )
      Contact( #T1_ET21 )
      S_SR(operand := #T1_ET03, r1 := #T1_ET01)
   END_RUNG
   // the same network as SCL:
   IF #T1_ET02 AND #T1_ET21 THEN
       #T1_ET03 := TRUE;   // SR flip-flop
   END_IF;
   IF #T1_ET01 THEN #T1_ET03 := FALSE; END_IF;
END_REGION

REGION Network 24: T1_ET20
   RUNG wire#powerrail
      Contact( #T1_ET02 )
      Contact( #T1_ET21 )
      S_SR(operand := #T1_ET20, r1 := wire#w1)
   END_RUNG
   RUNG wire#powerrail
      Contact( #T1_ET50 )
   END_RUNG wire#w1
   RUNG wire#powerrail
      Contact( #T1_ET60 )
   END_RUNG wire#w1
   RUNG wire#powerrail
      Contact( #T1_ET70 )
   END_RUNG wire#w1
   RUNG wire#powerrail
      Contact( #T1_ET80 )
   END_RUNG wire#w1
   // the same network as SCL:
   IF #T1_ET02 AND #T1_ET21 THEN
       #T1_ET20 := TRUE;   // SR flip-flop
   END_IF;
   IF #T1_ET50 OR #T1_ET60 OR #T1_ET70 OR #T1_ET80 THEN #T1_ET20 := FALSE; END_IF;
END_REGION

REGION Network 25: T1_ET02
   RUNG wire#powerrail
      Contact( #T1_ET10 )
      Contact( #T1_ET112 )
      Contact( #cnt_phs_ok )
      wire#w1
      I_Contact( #Habilitar_orden_JDT )
      wire#w2
      S_SR(operand := #T1_ET02, r1 := wire#w3)
   END_RUNG
   RUNG wire#w1
      Contact( #Habilitar_orden_JDT )
      I_Contact( #Moti_ERRO )
      I_Contact( #Moti_NENC )
   END_RUNG wire#w2
   RUNG wire#powerrail
      Contact( #T1_ET08 )
      Contact( #O_Vaciar )
      I_Contact( #EstadoZona.PerReset_CBx )
      Contact( #EstadoZona.Marcha_CBx )
      I_Contact( #EstadoVI.Error_Mx )
   END_RUNG wire#w2
   RUNG wire#powerrail
      Contact( #T1_ET03 )
      Contact( #T1_ET20 )
   END_RUNG wire#w3
   // the same network as SCL:
   IF (#T1_ET10 AND #T1_ET112 AND #cnt_phs_ok AND (NOT #Habilitar_orden_JDT OR (#Habilitar_orden_JDT AND NOT #Moti_ERRO AND NOT #Moti_NENC))) OR (#T1_ET08 AND #O_Vaciar AND NOT #EstadoZona.PerReset_CBx AND #EstadoZona.Marcha_CBx AND NOT #EstadoVI.Error_Mx) THEN
       #T1_ET02 := TRUE;   // SR flip-flop
   END_IF;
   IF #T1_ET03 AND #T1_ET20 THEN #T1_ET02 := FALSE; END_IF;
END_REGION

REGION Network 26: T1_ET02_JDT
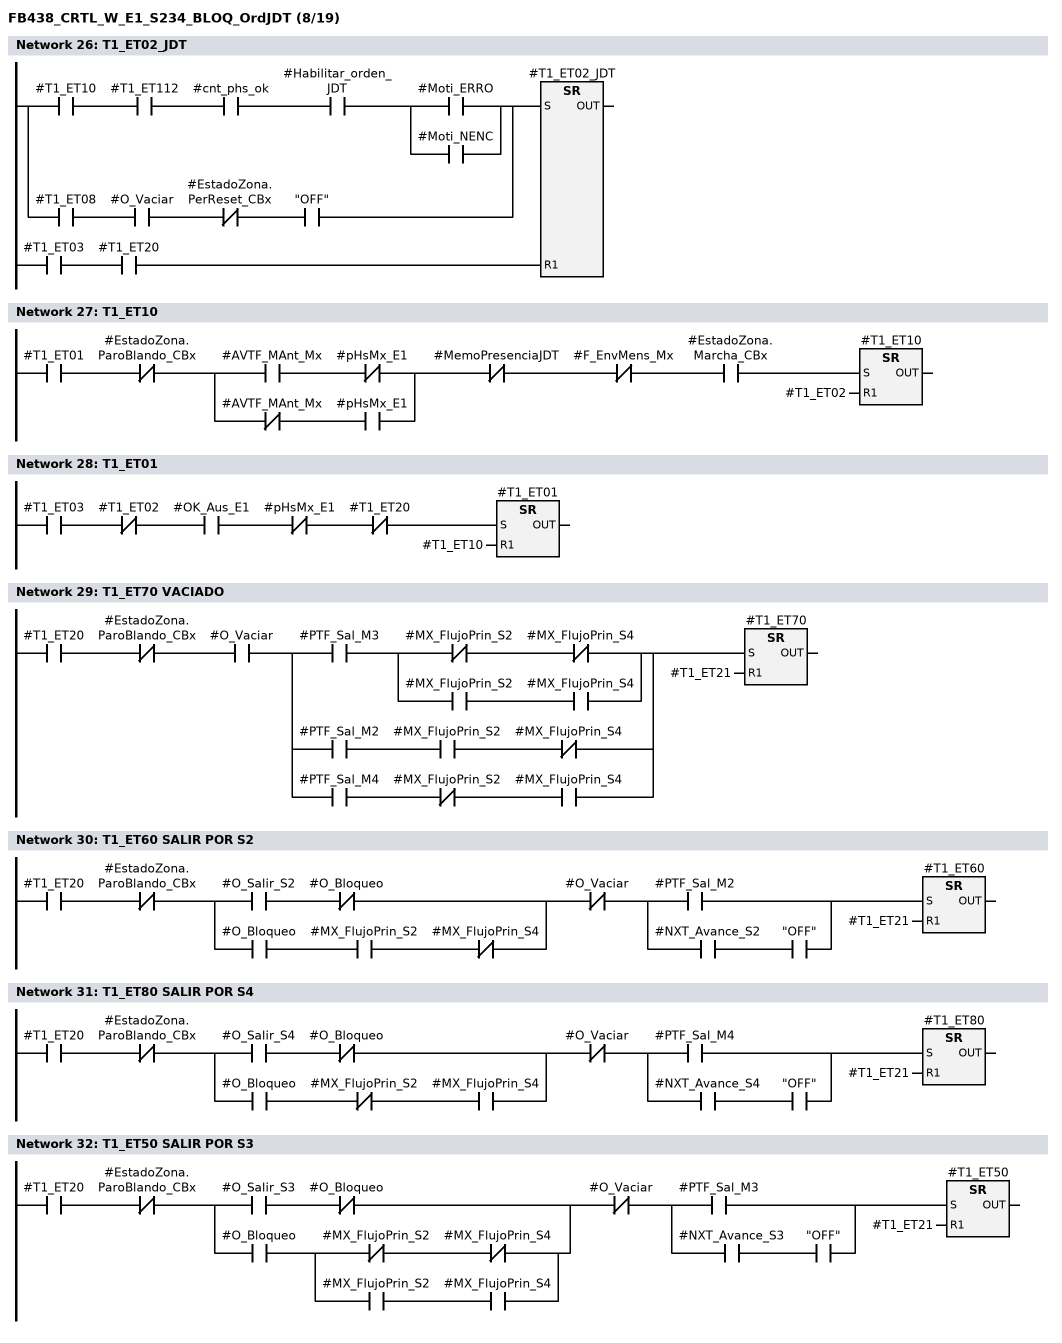
   RUNG wire#powerrail
      Contact( #T1_ET10 )
      Contact( #T1_ET112 )
      Contact( #cnt_phs_ok )
      Contact( #Habilitar_orden_JDT )
      wire#w1
      Contact( #Moti_ERRO )
      wire#w2
      S_SR(operand := #T1_ET02_JDT, r1 := wire#w3)
   END_RUNG
   RUNG wire#w1
      Contact( #Moti_NENC )
   END_RUNG wire#w2
   RUNG wire#powerrail
      Contact( #T1_ET08 )
      Contact( #O_Vaciar )
      I_Contact( #EstadoZona.PerReset_CBx )
      Contact( "OFF" )
   END_RUNG wire#w2
   RUNG wire#powerrail
      Contact( #T1_ET03 )
      Contact( #T1_ET20 )
   END_RUNG wire#w3
   // the same network as SCL:
   IF (#T1_ET10 AND #T1_ET112 AND #cnt_phs_ok AND #Habilitar_orden_JDT AND (#Moti_ERRO OR #Moti_NENC)) OR (#T1_ET08 AND #O_Vaciar AND NOT #EstadoZona.PerReset_CBx AND "OFF") THEN
       #T1_ET02_JDT := TRUE;   // SR flip-flop
   END_IF;
   IF #T1_ET03 AND #T1_ET20 THEN #T1_ET02_JDT := FALSE; END_IF;
END_REGION

REGION Network 27: T1_ET10
   RUNG wire#powerrail
      Contact( #T1_ET01 )
      I_Contact( #EstadoZona.ParoBlando_CBx )
      wire#w1
      Contact( #AVTF_MAnt_Mx )
      I_Contact( #pHsMx_E1 )
      wire#w2
      I_Contact( #MemoPresenciaJDT )
      I_Contact( #F_EnvMens_Mx )
      Contact( #EstadoZona.Marcha_CBx )
      S_SR(operand := #T1_ET10, r1 := #T1_ET02)
   END_RUNG
   RUNG wire#w1
      I_Contact( #AVTF_MAnt_Mx )
      Contact( #pHsMx_E1 )
   END_RUNG wire#w2
   // the same network as SCL:
   IF #T1_ET01 AND NOT #EstadoZona.ParoBlando_CBx AND ((#AVTF_MAnt_Mx AND NOT #pHsMx_E1) OR (NOT #AVTF_MAnt_Mx AND #pHsMx_E1)) AND NOT #MemoPresenciaJDT AND NOT #F_EnvMens_Mx AND #EstadoZona.Marcha_CBx THEN
       #T1_ET10 := TRUE;   // SR flip-flop
   END_IF;
   IF #T1_ET02 THEN #T1_ET10 := FALSE; END_IF;
END_REGION

REGION Network 28: T1_ET01
   RUNG wire#powerrail
      Contact( #T1_ET03 )
      I_Contact( #T1_ET02 )
      Contact( #OK_Aus_E1 )
      I_Contact( #pHsMx_E1 )
      I_Contact( #T1_ET20 )
      S_SR(operand := #T1_ET01, r1 := #T1_ET10)
   END_RUNG
   // the same network as SCL:
   IF #T1_ET03 AND NOT #T1_ET02 AND #OK_Aus_E1 AND NOT #pHsMx_E1 AND NOT #T1_ET20 THEN
       #T1_ET01 := TRUE;   // SR flip-flop
   END_IF;
   IF #T1_ET10 THEN #T1_ET01 := FALSE; END_IF;
END_REGION

REGION Network 29: T1_ET70 VACIADO
   RUNG wire#powerrail
      Contact( #T1_ET20 )
      I_Contact( #EstadoZona.ParoBlando_CBx )
      Contact( #O_Vaciar )
      wire#w1
      Contact( #PTF_Sal_M3 )
      wire#w2
      I_Contact( #MX_FlujoPrin_S2 )
      I_Contact( #MX_FlujoPrin_S4 )
      wire#w3
      S_SR(operand := #T1_ET70, r1 := #T1_ET21)
   END_RUNG
   RUNG wire#w2
      Contact( #MX_FlujoPrin_S2 )
      Contact( #MX_FlujoPrin_S4 )
   END_RUNG wire#w3
   RUNG wire#w1
      Contact( #PTF_Sal_M2 )
      Contact( #MX_FlujoPrin_S2 )
      I_Contact( #MX_FlujoPrin_S4 )
   END_RUNG wire#w3
   RUNG wire#w1
      Contact( #PTF_Sal_M4 )
      I_Contact( #MX_FlujoPrin_S2 )
      Contact( #MX_FlujoPrin_S4 )
   END_RUNG wire#w3
   // the same network as SCL:
   IF #T1_ET20 AND NOT #EstadoZona.ParoBlando_CBx AND #O_Vaciar AND ((#PTF_Sal_M3 AND ((NOT #MX_FlujoPrin_S2 AND NOT #MX_FlujoPrin_S4) OR (#MX_FlujoPrin_S2 AND #MX_FlujoPrin_S4))) OR (#PTF_Sal_M2 AND #MX_FlujoPrin_S2 AND NOT #MX_FlujoPrin_S4) OR (#PTF_Sal_M4 AND NOT #MX_FlujoPrin_S2 AND #MX_FlujoPrin_S4)) THEN
       #T1_ET70 := TRUE;   // SR flip-flop
   END_IF;
   IF #T1_ET21 THEN #T1_ET70 := FALSE; END_IF;
END_REGION

REGION Network 30: T1_ET60 SALIR POR S2
   RUNG wire#powerrail
      Contact( #T1_ET20 )
      I_Contact( #EstadoZona.ParoBlando_CBx )
      wire#w1
      Contact( #O_Salir_S2 )
      I_Contact( #O_Bloqueo )
      wire#w2
      I_Contact( #O_Vaciar )
      wire#w3
      Contact( #PTF_Sal_M2 )
      wire#w4
      S_SR(operand := #T1_ET60, r1 := #T1_ET21)
   END_RUNG
   RUNG wire#w1
      Contact( #O_Bloqueo )
      Contact( #MX_FlujoPrin_S2 )
      I_Contact( #MX_FlujoPrin_S4 )
   END_RUNG wire#w2
   RUNG wire#w3
      Contact( #NXT_Avance_S2 )
      Contact( "OFF" )
   END_RUNG wire#w4
   // the same network as SCL:
   IF #T1_ET20 AND NOT #EstadoZona.ParoBlando_CBx AND ((#O_Salir_S2 AND NOT #O_Bloqueo) OR (#O_Bloqueo AND #MX_FlujoPrin_S2 AND NOT #MX_FlujoPrin_S4)) AND NOT #O_Vaciar AND (#PTF_Sal_M2 OR (#NXT_Avance_S2 AND "OFF")) THEN
       #T1_ET60 := TRUE;   // SR flip-flop
   END_IF;
   IF #T1_ET21 THEN #T1_ET60 := FALSE; END_IF;
END_REGION

REGION Network 31: T1_ET80 SALIR POR S4
   RUNG wire#powerrail
      Contact( #T1_ET20 )
      I_Contact( #EstadoZona.ParoBlando_CBx )
      wire#w1
      Contact( #O_Salir_S4 )
      I_Contact( #O_Bloqueo )
      wire#w2
      I_Contact( #O_Vaciar )
      wire#w3
      Contact( #PTF_Sal_M4 )
      wire#w4
      S_SR(operand := #T1_ET80, r1 := #T1_ET21)
   END_RUNG
   RUNG wire#w1
      Contact( #O_Bloqueo )
      I_Contact( #MX_FlujoPrin_S2 )
      Contact( #MX_FlujoPrin_S4 )
   END_RUNG wire#w2
   RUNG wire#w3
      Contact( #NXT_Avance_S4 )
      Contact( "OFF" )
   END_RUNG wire#w4
   // the same network as SCL:
   IF #T1_ET20 AND NOT #EstadoZona.ParoBlando_CBx AND ((#O_Salir_S4 AND NOT #O_Bloqueo) OR (#O_Bloqueo AND NOT #MX_FlujoPrin_S2 AND #MX_FlujoPrin_S4)) AND NOT #O_Vaciar AND (#PTF_Sal_M4 OR (#NXT_Avance_S4 AND "OFF")) THEN
       #T1_ET80 := TRUE;   // SR flip-flop
   END_IF;
   IF #T1_ET21 THEN #T1_ET80 := FALSE; END_IF;
END_REGION

REGION Network 32: T1_ET50 SALIR POR S3
   RUNG wire#powerrail
      Contact( #T1_ET20 )
      I_Contact( #EstadoZona.ParoBlando_CBx )
      wire#w1
      Contact( #O_Salir_S3 )
      I_Contact( #O_Bloqueo )
      wire#w2
      I_Contact( #O_Vaciar )
      wire#w4
      Contact( #PTF_Sal_M3 )
      wire#w5
      S_SR(operand := #T1_ET50, r1 := #T1_ET21)
   END_RUNG
   RUNG wire#w1
      Contact( #O_Bloqueo )
      wire#w3
      I_Contact( #MX_FlujoPrin_S2 )
      I_Contact( #MX_FlujoPrin_S4 )
   END_RUNG wire#w2
   RUNG wire#w3
      Contact( #MX_FlujoPrin_S2 )
      Contact( #MX_FlujoPrin_S4 )
   END_RUNG wire#w2
   RUNG wire#w4
      Contact( #NXT_Avance_S3 )
      Contact( "OFF" )
   END_RUNG wire#w5
   // the same network as SCL:
   IF #T1_ET20 AND NOT #EstadoZona.ParoBlando_CBx AND ((#O_Salir_S3 AND NOT #O_Bloqueo) OR (#O_Bloqueo AND ((NOT #MX_FlujoPrin_S2 AND NOT #MX_FlujoPrin_S4) OR (#MX_FlujoPrin_S2 AND #MX_FlujoPrin_S4)))) AND NOT #O_Vaciar AND (#PTF_Sal_M3 OR (#NXT_Avance_S3 AND "OFF")) THEN
       #T1_ET50 := TRUE;   // SR flip-flop
   END_IF;
   IF #T1_ET21 THEN #T1_ET50 := FALSE; END_IF;
END_REGION

REGION Network 33: T1_ET21
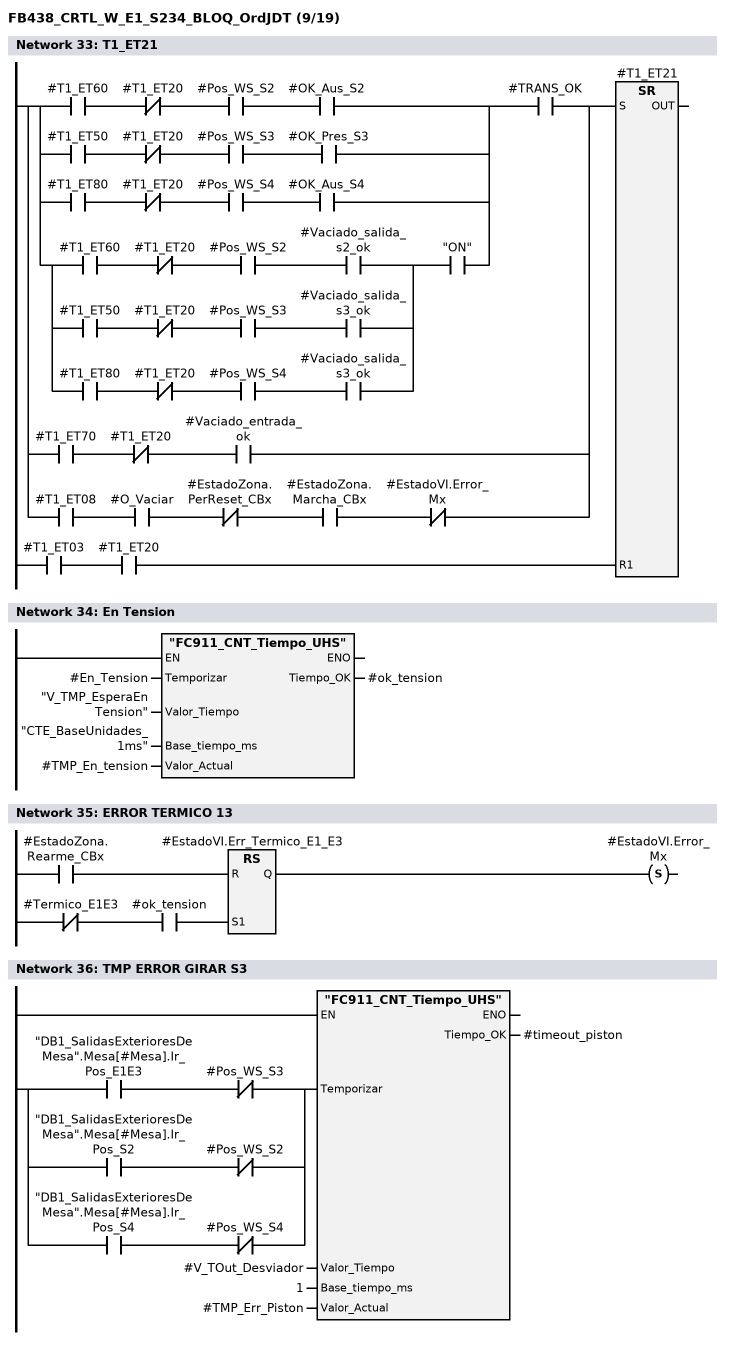
   RUNG wire#powerrail
      Contact( #T1_ET60 )
      I_Contact( #T1_ET20 )
      Contact( #Pos_WS_S2 )
      Contact( #OK_Aus_S2 )
      wire#w1
      Contact( #TRANS_OK )
      wire#w3
      S_SR(operand := #T1_ET21, r1 := wire#w4)
   END_RUNG
   RUNG wire#powerrail
      Contact( #T1_ET50 )
      I_Contact( #T1_ET20 )
      Contact( #Pos_WS_S3 )
      Contact( #OK_Pres_S3 )
   END_RUNG wire#w1
   RUNG wire#powerrail
      Contact( #T1_ET80 )
      I_Contact( #T1_ET20 )
      Contact( #Pos_WS_S4 )
      Contact( #OK_Aus_S4 )
   END_RUNG wire#w1
   RUNG wire#powerrail
      Contact( #T1_ET60 )
      I_Contact( #T1_ET20 )
      Contact( #Pos_WS_S2 )
      Contact( #Vaciado_salida_s2_ok )
      wire#w2
      Contact( "ON" )
   END_RUNG wire#w1
   RUNG wire#powerrail
      Contact( #T1_ET50 )
      I_Contact( #T1_ET20 )
      Contact( #Pos_WS_S3 )
      Contact( #Vaciado_salida_s3_ok )
   END_RUNG wire#w2
   RUNG wire#powerrail
      Contact( #T1_ET80 )
      I_Contact( #T1_ET20 )
      Contact( #Pos_WS_S4 )
      Contact( #Vaciado_salida_s3_ok )
   END_RUNG wire#w2
   RUNG wire#powerrail
      Contact( #T1_ET70 )
      I_Contact( #T1_ET20 )
      Contact( #Vaciado_entrada_ok )
   END_RUNG wire#w3
   RUNG wire#powerrail
      Contact( #T1_ET08 )
      Contact( #O_Vaciar )
      I_Contact( #EstadoZona.PerReset_CBx )
      Contact( #EstadoZona.Marcha_CBx )
      I_Contact( #EstadoVI.Error_Mx )
   END_RUNG wire#w3
   RUNG wire#powerrail
      Contact( #T1_ET03 )
      Contact( #T1_ET20 )
   END_RUNG wire#w4
   // the same network as SCL:
   IF (((#T1_ET60 AND NOT #T1_ET20 AND #Pos_WS_S2 AND #OK_Aus_S2) OR (#T1_ET50 AND NOT #T1_ET20 AND #Pos_WS_S3 AND #OK_Pres_S3) OR (#T1_ET80 AND NOT #T1_ET20 AND #Pos_WS_S4 AND #OK_Aus_S4) OR (((#T1_ET60 AND NOT #T1_ET20 AND #Pos_WS_S2 AND #Vaciado_salida_s2_ok) OR (#T1_ET50 AND NOT #T1_ET20 AND #Pos_WS_S3 AND #Vaciado_salida_s3_ok) OR (#T1_ET80 AND NOT #T1_ET20 AND #Pos_WS_S4 AND #Vaciado_salida_s3_ok)) AND "ON")) AND #TRANS_OK) OR (#T1_ET70 AND NOT #T1_ET20 AND #Vaciado_entrada_ok) OR (#T1_ET08 AND #O_Vaciar AND NOT #EstadoZona.PerReset_CBx AND #EstadoZona.Marcha_CBx AND NOT #EstadoVI.Error_Mx) THEN
       #T1_ET21 := TRUE;   // SR flip-flop
   END_IF;
   IF #T1_ET03 AND #T1_ET20 THEN #T1_ET21 := FALSE; END_IF;
END_REGION

REGION Network 34: En Tension
   RUNG wire#powerrail
      "FC911_CNT_Tiempo_UHS"(Temporizar := #En_Tension, Valor_Tiempo := "V_TMP_EsperaEnTension", Base_tiempo_ms := "CTE_BaseUnidades_1ms", Valor_Actual := #TMP_En_tension, Tiempo_OK => #ok_tension)
   END_RUNG
   // the same network as SCL:
   "FC911_CNT_Tiempo_UHS"(Temporizar := #En_Tension,
                          Valor_Tiempo := "V_TMP_EsperaEnTension",
                          Base_tiempo_ms := "CTE_BaseUnidades_1ms",
                          Valor_Actual := #TMP_En_tension,
                          Tiempo_OK => #ok_tension);
END_REGION

REGION Network 35: ERROR TERMICO 13
   RUNG wire#powerrail
      Contact( #EstadoZona.Rearme_CBx )
      S_RS(operand := #EstadoVI.Err_Termico_E1_E3, s1 := wire#w1)
      S_Coil( #EstadoVI.Error_Mx )
   END_RUNG
   RUNG wire#powerrail
      I_Contact( #Termico_E1E3 )
      Contact( #ok_tension )
   END_RUNG wire#w1
   // the same network as SCL:
   IF #EstadoZona.Rearme_CBx THEN
       #EstadoVI.Err_Termico_E1_E3 := FALSE;   // RS flip-flop
   END_IF;
   IF NOT #Termico_E1E3 AND #ok_tension THEN #EstadoVI.Err_Termico_E1_E3 := TRUE; END_IF;
   IF #EstadoVI.Err_Termico_E1_E3 THEN #EstadoVI.Error_Mx := TRUE; END_IF;
END_REGION

REGION Network 36: TMP ERROR GIRAR S3
   RUNG wire#powerrail
      "FC911_CNT_Tiempo_UHS"(Temporizar := wire#w1, Valor_Tiempo := #V_TOut_Desviador, Base_tiempo_ms := 1, Valor_Actual := #TMP_Err_Piston, Tiempo_OK => #timeout_piston)
   END_RUNG
   RUNG wire#powerrail
      Contact( "DB1_SalidasExterioresDeMesa".Mesa[#Mesa].Ir_Pos_E1E3 )
      I_Contact( #Pos_WS_S3 )
   END_RUNG wire#w1
   RUNG wire#powerrail
      Contact( "DB1_SalidasExterioresDeMesa".Mesa[#Mesa].Ir_Pos_S2 )
      I_Contact( #Pos_WS_S2 )
   END_RUNG wire#w1
   RUNG wire#powerrail
      Contact( "DB1_SalidasExterioresDeMesa".Mesa[#Mesa].Ir_Pos_S4 )
      I_Contact( #Pos_WS_S4 )
   END_RUNG wire#w1
   // the same network as SCL:
   "FC911_CNT_Tiempo_UHS"(Temporizar := ("DB1_SalidasExterioresDeMesa".Mesa[#Mesa].Ir_Pos_E1E3 AND NOT #Pos_WS_S3) OR ("DB1_SalidasExterioresDeMesa".Mesa[#Mesa].Ir_Pos_S2 AND NOT #Pos_WS_S2) OR ("DB1_SalidasExterioresDeMesa".Mesa[#Mesa].Ir_Pos_S4 AND NOT #Pos_WS_S4),
                          Valor_Tiempo := #V_TOut_Desviador,
                          Base_tiempo_ms := 1,
                          Valor_Actual := #TMP_Err_Piston,
                          Tiempo_OK => #timeout_piston);
END_REGION

REGION Network 37: ERROR POSICION 0
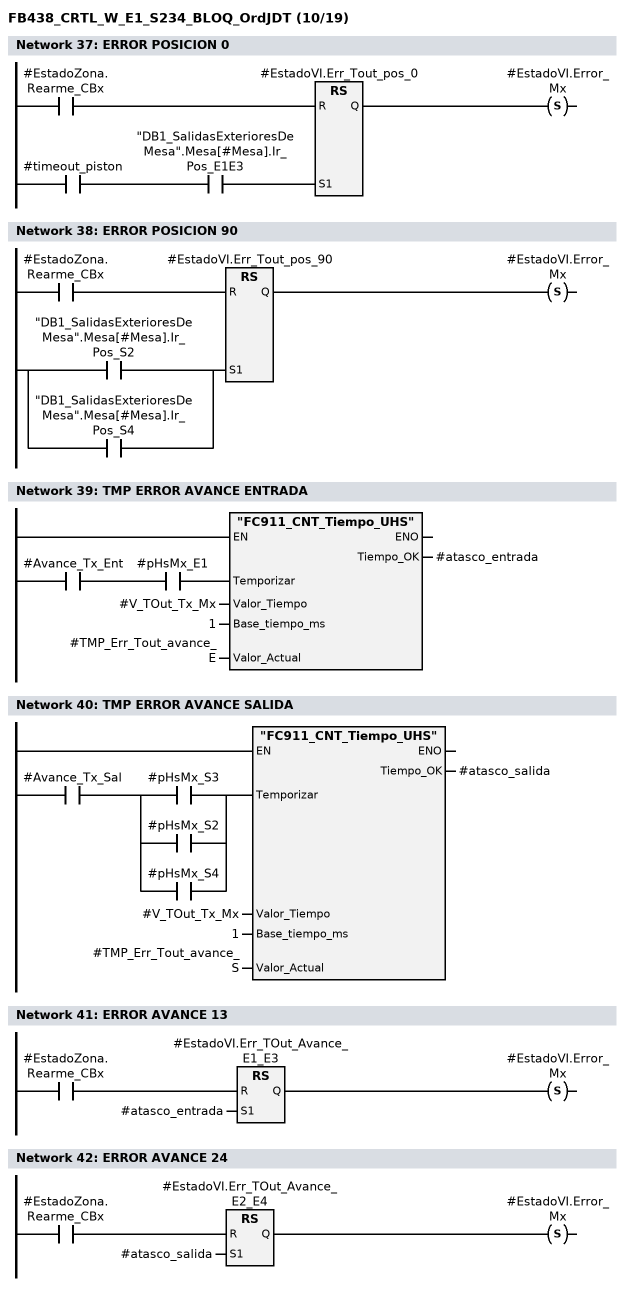
   RUNG wire#powerrail
      Contact( #EstadoZona.Rearme_CBx )
      S_RS(operand := #EstadoVI.Err_Tout_pos_0, s1 := wire#w1)
      S_Coil( #EstadoVI.Error_Mx )
   END_RUNG
   RUNG wire#powerrail
      Contact( #timeout_piston )
      Contact( "DB1_SalidasExterioresDeMesa".Mesa[#Mesa].Ir_Pos_E1E3 )
   END_RUNG wire#w1
   // the same network as SCL:
   IF #EstadoZona.Rearme_CBx THEN
       #EstadoVI.Err_Tout_pos_0 := FALSE;   // RS flip-flop
   END_IF;
   IF #timeout_piston AND "DB1_SalidasExterioresDeMesa".Mesa[#Mesa].Ir_Pos_E1E3 THEN
       #EstadoVI.Err_Tout_pos_0 := TRUE;
   END_IF;
   IF #EstadoVI.Err_Tout_pos_0 THEN #EstadoVI.Error_Mx := TRUE; END_IF;
END_REGION

REGION Network 38: ERROR POSICION 90
   RUNG wire#powerrail
      Contact( #EstadoZona.Rearme_CBx )
      S_RS(operand := #EstadoVI.Err_Tout_pos_90, s1 := wire#w1)
      S_Coil( #EstadoVI.Error_Mx )
   END_RUNG
   RUNG wire#powerrail
      Contact( "DB1_SalidasExterioresDeMesa".Mesa[#Mesa].Ir_Pos_S2 )
   END_RUNG wire#w1
   RUNG wire#powerrail
      Contact( "DB1_SalidasExterioresDeMesa".Mesa[#Mesa].Ir_Pos_S4 )
   END_RUNG wire#w1
   // the same network as SCL:
   IF #EstadoZona.Rearme_CBx THEN
       #EstadoVI.Err_Tout_pos_90 := FALSE;   // RS flip-flop
   END_IF;
   IF "DB1_SalidasExterioresDeMesa".Mesa[#Mesa].Ir_Pos_S2 OR "DB1_SalidasExterioresDeMesa".Mesa[#Mesa].Ir_Pos_S4 THEN
       #EstadoVI.Err_Tout_pos_90 := TRUE;
   END_IF;
   IF #EstadoVI.Err_Tout_pos_90 THEN #EstadoVI.Error_Mx := TRUE; END_IF;
END_REGION

REGION Network 39: TMP ERROR AVANCE ENTRADA
   RUNG wire#powerrail
      "FC911_CNT_Tiempo_UHS"(Temporizar := wire#w1, Valor_Tiempo := #V_TOut_Tx_Mx, Base_tiempo_ms := 1, Valor_Actual := #TMP_Err_Tout_avance_E, Tiempo_OK => #atasco_entrada)
   END_RUNG
   RUNG wire#powerrail
      Contact( #Avance_Tx_Ent )
      Contact( #pHsMx_E1 )
   END_RUNG wire#w1
   // the same network as SCL:
   "FC911_CNT_Tiempo_UHS"(Temporizar := #Avance_Tx_Ent AND #pHsMx_E1,
                          Valor_Tiempo := #V_TOut_Tx_Mx,
                          Base_tiempo_ms := 1,
                          Valor_Actual := #TMP_Err_Tout_avance_E,
                          Tiempo_OK => #atasco_entrada);
END_REGION

REGION Network 40: TMP ERROR AVANCE SALIDA
   RUNG wire#powerrail
      "FC911_CNT_Tiempo_UHS"(Temporizar := wire#w2, Valor_Tiempo := #V_TOut_Tx_Mx, Base_tiempo_ms := 1, Valor_Actual := #TMP_Err_Tout_avance_S, Tiempo_OK => #atasco_salida)
   END_RUNG
   RUNG wire#powerrail
      Contact( #Avance_Tx_Sal )
      wire#w1
      Contact( #pHsMx_S3 )
   END_RUNG wire#w2
   RUNG wire#w1
      Contact( #pHsMx_S2 )
   END_RUNG wire#w2
   RUNG wire#w1
      Contact( #pHsMx_S4 )
   END_RUNG wire#w2
   // the same network as SCL:
   "FC911_CNT_Tiempo_UHS"(Temporizar := #Avance_Tx_Sal AND (#pHsMx_S3 OR #pHsMx_S2 OR #pHsMx_S4),
                          Valor_Tiempo := #V_TOut_Tx_Mx,
                          Base_tiempo_ms := 1,
                          Valor_Actual := #TMP_Err_Tout_avance_S,
                          Tiempo_OK => #atasco_salida);
END_REGION

REGION Network 41: ERROR AVANCE 13
   RUNG wire#powerrail
      Contact( #EstadoZona.Rearme_CBx )
      S_RS(operand := #EstadoVI.Err_TOut_Avance_E1_E3, s1 := #atasco_entrada)
      S_Coil( #EstadoVI.Error_Mx )
   END_RUNG
   // the same network as SCL:
   IF #EstadoZona.Rearme_CBx THEN
       #EstadoVI.Err_TOut_Avance_E1_E3 := FALSE;   // RS flip-flop
   END_IF;
   IF #atasco_entrada THEN #EstadoVI.Err_TOut_Avance_E1_E3 := TRUE; END_IF;
   IF #EstadoVI.Err_TOut_Avance_E1_E3 THEN #EstadoVI.Error_Mx := TRUE; END_IF;
END_REGION

REGION Network 42: ERROR AVANCE 24
   RUNG wire#powerrail
      Contact( #EstadoZona.Rearme_CBx )
      S_RS(operand := #EstadoVI.Err_TOut_Avance_E2_E4, s1 := #atasco_salida)
      S_Coil( #EstadoVI.Error_Mx )
   END_RUNG
   // the same network as SCL:
   IF #EstadoZona.Rearme_CBx THEN
       #EstadoVI.Err_TOut_Avance_E2_E4 := FALSE;   // RS flip-flop
   END_IF;
   IF #atasco_salida THEN #EstadoVI.Err_TOut_Avance_E2_E4 := TRUE; END_IF;
   IF #EstadoVI.Err_TOut_Avance_E2_E4 THEN #EstadoVI.Error_Mx := TRUE; END_IF;
END_REGION

REGION Network 43: ERROR MESA OCUPADA
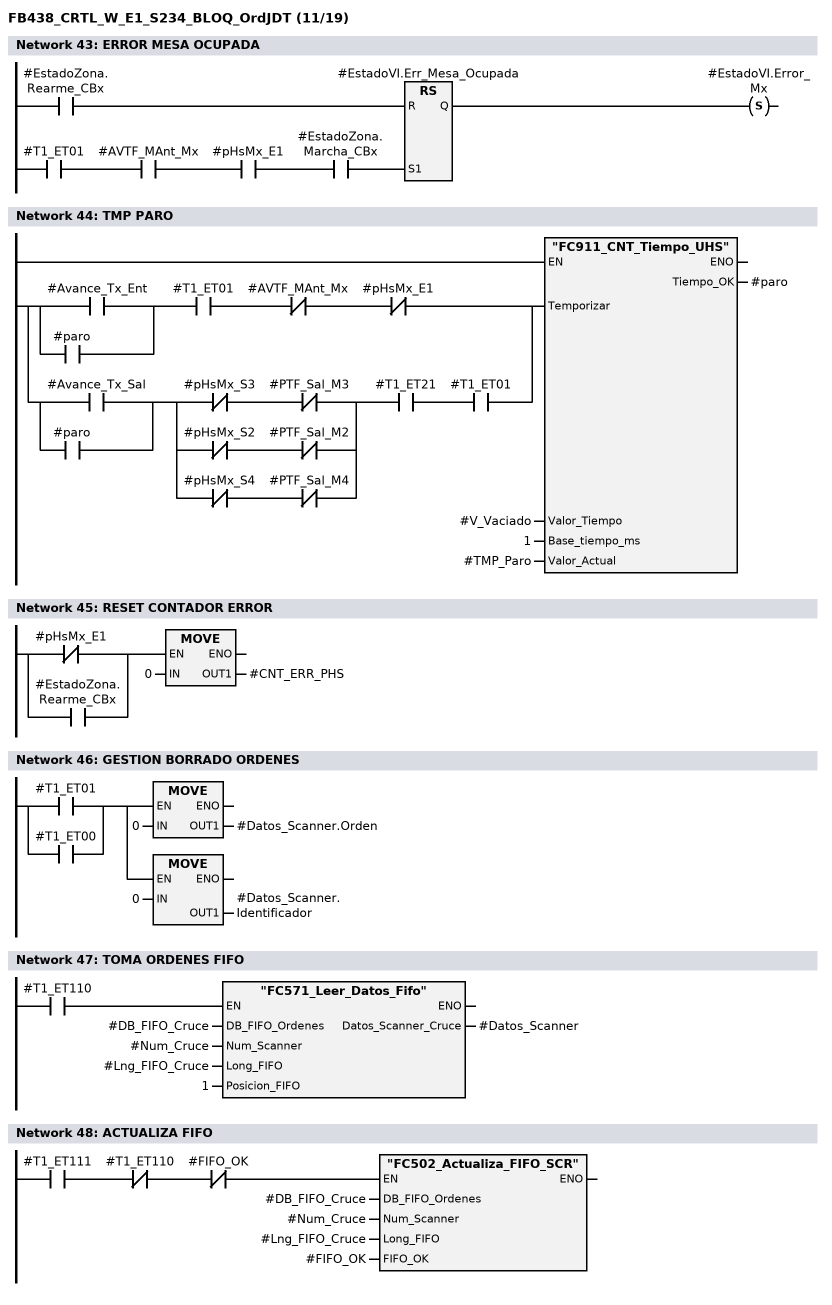
   RUNG wire#powerrail
      Contact( #EstadoZona.Rearme_CBx )
      S_RS(operand := #EstadoVI.Err_Mesa_Ocupada, s1 := wire#w1)
      S_Coil( #EstadoVI.Error_Mx )
   END_RUNG
   RUNG wire#powerrail
      Contact( #T1_ET01 )
      Contact( #AVTF_MAnt_Mx )
      Contact( #pHsMx_E1 )
      Contact( #EstadoZona.Marcha_CBx )
   END_RUNG wire#w1
   // the same network as SCL:
   IF #EstadoZona.Rearme_CBx THEN
       #EstadoVI.Err_Mesa_Ocupada := FALSE;   // RS flip-flop
   END_IF;
   IF #T1_ET01 AND #AVTF_MAnt_Mx AND #pHsMx_E1 AND #EstadoZona.Marcha_CBx THEN
       #EstadoVI.Err_Mesa_Ocupada := TRUE;
   END_IF;
   IF #EstadoVI.Err_Mesa_Ocupada THEN #EstadoVI.Error_Mx := TRUE; END_IF;
END_REGION

REGION Network 44: TMP PARO
   RUNG wire#powerrail
      "FC911_CNT_Tiempo_UHS"(Temporizar := wire#w4, Valor_Tiempo := #V_Vaciado, Base_tiempo_ms := 1, Valor_Actual := #TMP_Paro, Tiempo_OK => #paro)
   END_RUNG
   RUNG wire#powerrail
      Contact( #Avance_Tx_Ent )
      wire#w1
      Contact( #T1_ET01 )
      I_Contact( #AVTF_MAnt_Mx )
      I_Contact( #pHsMx_E1 )
   END_RUNG wire#w4
   RUNG wire#powerrail
      Contact( #paro )
   END_RUNG wire#w1
   RUNG wire#powerrail
      Contact( #Avance_Tx_Sal )
      wire#w2
      I_Contact( #pHsMx_S3 )
      I_Contact( #PTF_Sal_M3 )
      wire#w3
      Contact( #T1_ET21 )
      Contact( #T1_ET01 )
   END_RUNG wire#w4
   RUNG wire#powerrail
      Contact( #paro )
   END_RUNG wire#w2
   RUNG wire#w2
      I_Contact( #pHsMx_S2 )
      I_Contact( #PTF_Sal_M2 )
   END_RUNG wire#w3
   RUNG wire#w2
      I_Contact( #pHsMx_S4 )
      I_Contact( #PTF_Sal_M4 )
   END_RUNG wire#w3
   // the same network as SCL:
   "FC911_CNT_Tiempo_UHS"(Temporizar := ((#Avance_Tx_Ent OR #paro) AND #T1_ET01 AND NOT #AVTF_MAnt_Mx AND NOT #pHsMx_E1) OR ((#Avance_Tx_Sal OR #paro) AND ((NOT #pHsMx_S3 AND NOT #PTF_Sal_M3) OR (NOT #pHsMx_S2 AND NOT #PTF_Sal_M2) OR (NOT #pHsMx_S4 AND NOT #PTF_Sal_M4)) AND #T1_ET21 AND #T1_ET01),
                          Valor_Tiempo := #V_Vaciado,
                          Base_tiempo_ms := 1,
                          Valor_Actual := #TMP_Paro,
                          Tiempo_OK => #paro);
END_REGION

REGION Network 45: RESET CONTADOR ERROR
   RUNG wire#powerrail
      I_Contact( #pHsMx_E1 )
      wire#w1
      { S7_GenerateENO := "TRUE" } Move(in := 0, out1 => #CNT_ERR_PHS)
   END_RUNG
   RUNG wire#powerrail
      Contact( #EstadoZona.Rearme_CBx )
   END_RUNG wire#w1
   // the same network as SCL:
   IF NOT #pHsMx_E1 OR #EstadoZona.Rearme_CBx THEN #CNT_ERR_PHS := 0; END_IF;
END_REGION

REGION Network 46: GESTION BORRADO ORDENES
   RUNG wire#powerrail
      Contact( #T1_ET01 )
      wire#w1
      { S7_GenerateENO := "TRUE" } Move(in := 0, out1 => #Datos_Scanner.Orden)
   END_RUNG
   RUNG wire#powerrail
      Contact( #T1_ET00 )
   END_RUNG wire#w1
   RUNG wire#w1
      { S7_GenerateENO := "TRUE" } Move(in := 0, out1 => #Datos_Scanner.Identificador)
   END_RUNG
   // the same network as SCL:
   IF #T1_ET01 OR #T1_ET00 THEN
       #Datos_Scanner.Orden := 0;
       #Datos_Scanner.Identificador := 0;
   END_IF;
END_REGION

REGION Network 47: TOMA ORDENES FIFO
   RUNG wire#powerrail
      Contact( #T1_ET110 )
      "FC571_Leer_Datos_Fifo"(DB_FIFO_Ordenes := #DB_FIFO_Cruce, Num_Scanner := #Num_Cruce, Long_FIFO := #Lng_FIFO_Cruce, Posicion_FIFO := 1, Datos_Scanner_Cruce => #Datos_Scanner)
   END_RUNG
   // the same network as SCL:
   IF #T1_ET110 THEN
       "FC571_Leer_Datos_Fifo"(DB_FIFO_Ordenes := #DB_FIFO_Cruce,
                               Num_Scanner := #Num_Cruce,
                               Long_FIFO := #Lng_FIFO_Cruce,
                               Posicion_FIFO := 1,
                               Datos_Scanner_Cruce => #Datos_Scanner);
   END_IF;
END_REGION

REGION Network 48: ACTUALIZA FIFO
   RUNG wire#powerrail
      Contact( #T1_ET111 )
      I_Contact( #T1_ET110 )
      I_Contact( #FIFO_OK )
      "FC502_Actualiza_FIFO_SCR"(DB_FIFO_Ordenes := #DB_FIFO_Cruce, Num_Scanner := #Num_Cruce, Long_FIFO := #Lng_FIFO_Cruce, FIFO_OK := #FIFO_OK)
   END_RUNG
   // the same network as SCL:
   IF #T1_ET111 AND NOT #T1_ET110 AND NOT #FIFO_OK THEN
       "FC502_Actualiza_FIFO_SCR"(DB_FIFO_Ordenes := #DB_FIFO_Cruce,
                               Num_Scanner := #Num_Cruce,
                               Long_FIFO := #Lng_FIFO_Cruce,
                               FIFO_OK := #FIFO_OK);
   END_IF;
END_REGION

REGION Network 49: BORRA FIFO
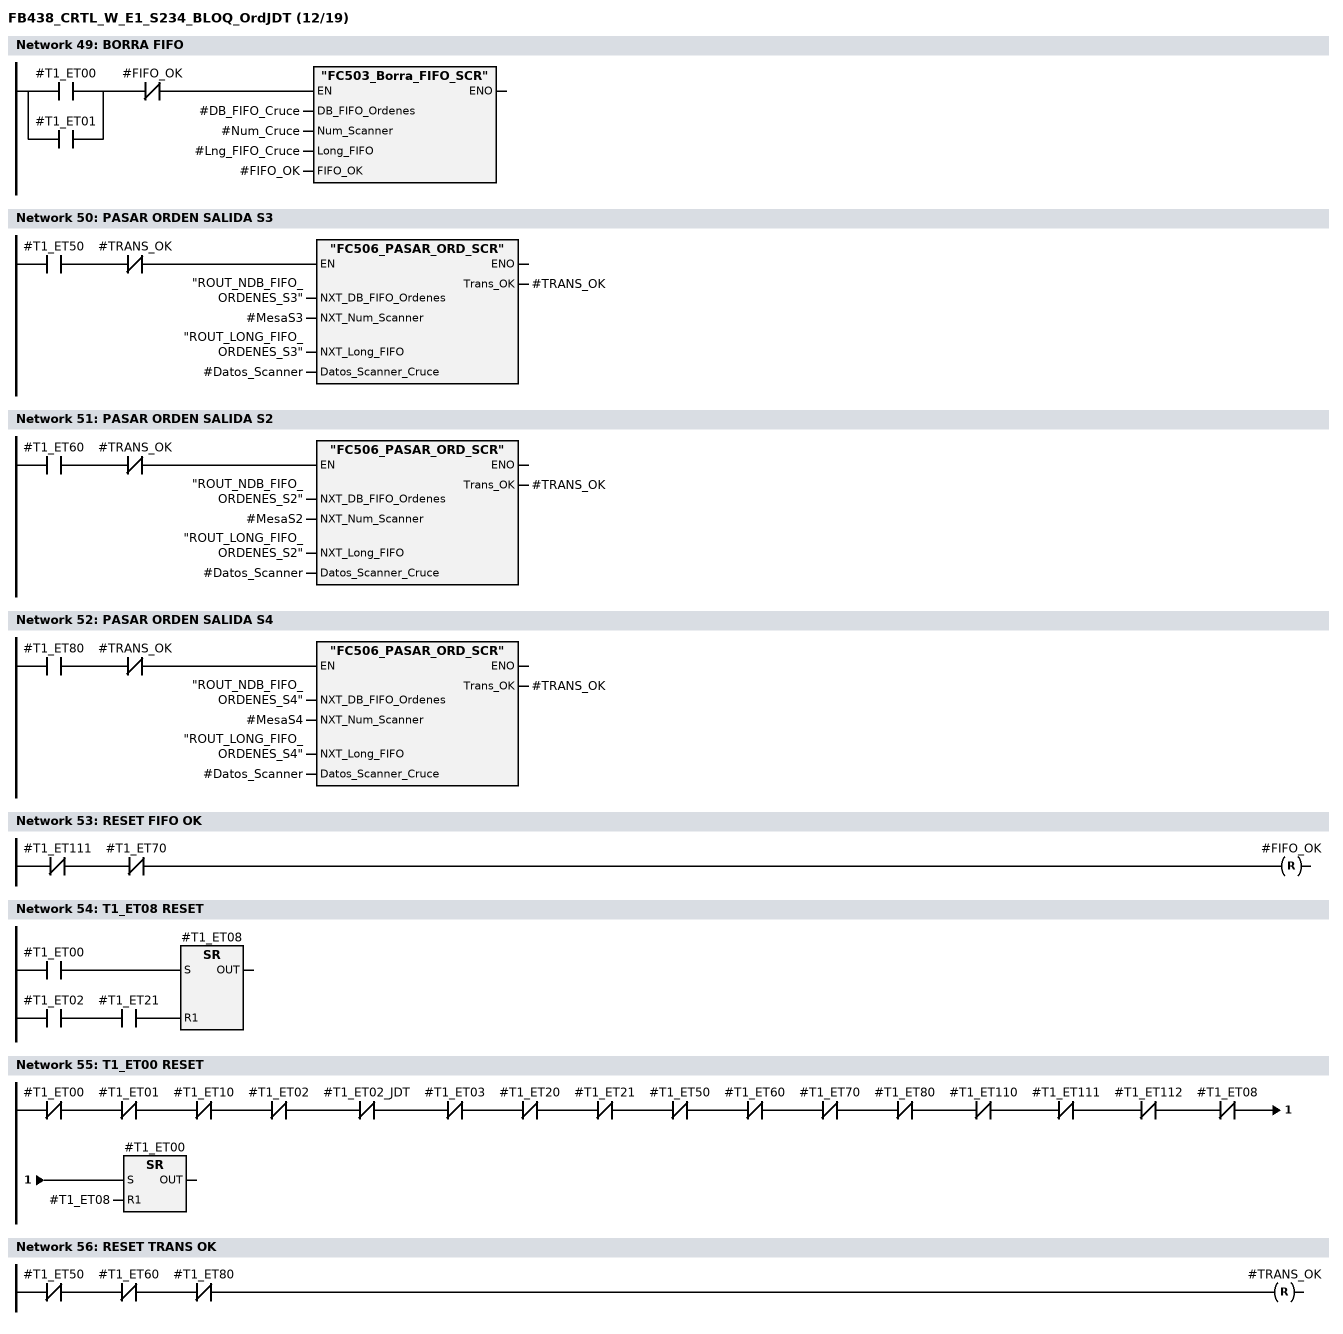
   RUNG wire#powerrail
      Contact( #T1_ET00 )
      wire#w1
      I_Contact( #FIFO_OK )
      "FC503_Borra_FIFO_SCR"(DB_FIFO_Ordenes := #DB_FIFO_Cruce, Num_Scanner := #Num_Cruce, Long_FIFO := #Lng_FIFO_Cruce, FIFO_OK := #FIFO_OK)
   END_RUNG
   RUNG wire#powerrail
      Contact( #T1_ET01 )
   END_RUNG wire#w1
   // the same network as SCL:
   IF (#T1_ET00 OR #T1_ET01) AND NOT #FIFO_OK THEN
       "FC503_Borra_FIFO_SCR"(DB_FIFO_Ordenes := #DB_FIFO_Cruce,
                              Num_Scanner := #Num_Cruce,
                              Long_FIFO := #Lng_FIFO_Cruce,
                              FIFO_OK := #FIFO_OK);
   END_IF;
END_REGION

REGION Network 50: PASAR ORDEN SALIDA S3
   RUNG wire#powerrail
      Contact( #T1_ET50 )
      I_Contact( #TRANS_OK )
      "FC506_PASAR_ORD_SCR"(NXT_DB_FIFO_Ordenes := "ROUT_NDB_FIFO_ORDENES_S3", NXT_Num_Scanner := #MesaS3, NXT_Long_FIFO := "ROUT_LONG_FIFO_ORDENES_S3", Datos_Scanner_Cruce := #Datos_Scanner, Trans_OK => #TRANS_OK)
   END_RUNG
   // the same network as SCL:
   IF #T1_ET50 AND NOT #TRANS_OK THEN
       "FC506_PASAR_ORD_SCR"(NXT_DB_FIFO_Ordenes := "ROUT_NDB_FIFO_ORDENES_S3",
                             NXT_Num_Scanner := #MesaS3,
                             NXT_Long_FIFO := "ROUT_LONG_FIFO_ORDENES_S3",
                             Datos_Scanner_Cruce := #Datos_Scanner,
                             Trans_OK => #TRANS_OK);
   END_IF;
END_REGION

REGION Network 51: PASAR ORDEN SALIDA S2
   RUNG wire#powerrail
      Contact( #T1_ET60 )
      I_Contact( #TRANS_OK )
      "FC506_PASAR_ORD_SCR"(NXT_DB_FIFO_Ordenes := "ROUT_NDB_FIFO_ORDENES_S2", NXT_Num_Scanner := #MesaS2, NXT_Long_FIFO := "ROUT_LONG_FIFO_ORDENES_S2", Datos_Scanner_Cruce := #Datos_Scanner, Trans_OK => #TRANS_OK)
   END_RUNG
   // the same network as SCL:
   IF #T1_ET60 AND NOT #TRANS_OK THEN
       "FC506_PASAR_ORD_SCR"(NXT_DB_FIFO_Ordenes := "ROUT_NDB_FIFO_ORDENES_S2",
                             NXT_Num_Scanner := #MesaS2,
                             NXT_Long_FIFO := "ROUT_LONG_FIFO_ORDENES_S2",
                             Datos_Scanner_Cruce := #Datos_Scanner,
                             Trans_OK => #TRANS_OK);
   END_IF;
END_REGION

REGION Network 52: PASAR ORDEN SALIDA S4
   RUNG wire#powerrail
      Contact( #T1_ET80 )
      I_Contact( #TRANS_OK )
      "FC506_PASAR_ORD_SCR"(NXT_DB_FIFO_Ordenes := "ROUT_NDB_FIFO_ORDENES_S4", NXT_Num_Scanner := #MesaS4, NXT_Long_FIFO := "ROUT_LONG_FIFO_ORDENES_S4", Datos_Scanner_Cruce := #Datos_Scanner, Trans_OK => #TRANS_OK)
   END_RUNG
   // the same network as SCL:
   IF #T1_ET80 AND NOT #TRANS_OK THEN
       "FC506_PASAR_ORD_SCR"(NXT_DB_FIFO_Ordenes := "ROUT_NDB_FIFO_ORDENES_S4",
                             NXT_Num_Scanner := #MesaS4,
                             NXT_Long_FIFO := "ROUT_LONG_FIFO_ORDENES_S4",
                             Datos_Scanner_Cruce := #Datos_Scanner,
                             Trans_OK => #TRANS_OK);
   END_IF;
END_REGION

REGION Network 53: RESET FIFO OK
   RUNG wire#powerrail
      I_Contact( #T1_ET111 )
      I_Contact( #T1_ET70 )
      R_Coil( #FIFO_OK )
   END_RUNG
   // the same network as SCL:
   IF NOT #T1_ET111 AND NOT #T1_ET70 THEN #FIFO_OK := FALSE; END_IF;
END_REGION

REGION Network 54: T1_ET08 RESET
   RUNG wire#powerrail
      Contact( #T1_ET00 )
      S_SR(operand := #T1_ET08, r1 := wire#w1)
   END_RUNG
   RUNG wire#powerrail
      Contact( #T1_ET02 )
      Contact( #T1_ET21 )
   END_RUNG wire#w1
   // the same network as SCL:
   IF #T1_ET00 THEN
       #T1_ET08 := TRUE;   // SR flip-flop
   END_IF;
   IF #T1_ET02 AND #T1_ET21 THEN #T1_ET08 := FALSE; END_IF;
END_REGION

REGION Network 55: T1_ET00 RESET
   RUNG wire#powerrail
      I_Contact( #T1_ET00 )
      I_Contact( #T1_ET01 )
      I_Contact( #T1_ET10 )
      I_Contact( #T1_ET02 )
      I_Contact( #T1_ET02_JDT )
      I_Contact( #T1_ET03 )
      I_Contact( #T1_ET20 )
      I_Contact( #T1_ET21 )
      I_Contact( #T1_ET50 )
      I_Contact( #T1_ET60 )
      I_Contact( #T1_ET70 )
      I_Contact( #T1_ET80 )
      I_Contact( #T1_ET110 )
      I_Contact( #T1_ET111 )
      I_Contact( #T1_ET112 )
      I_Contact( #T1_ET08 )
      S_SR(operand := #T1_ET00, r1 := #T1_ET08)
   END_RUNG
   // the same network as SCL:
   IF NOT #T1_ET00 AND NOT #T1_ET01 AND NOT #T1_ET10 AND NOT #T1_ET02 AND NOT #T1_ET02_JDT AND NOT #T1_ET03 AND NOT #T1_ET20 AND NOT #T1_ET21 AND NOT #T1_ET50 AND NOT #T1_ET60 AND NOT #T1_ET70 AND NOT #T1_ET80 AND NOT #T1_ET110 AND NOT #T1_ET111 AND NOT #T1_ET112 AND NOT #T1_ET08 THEN
       #T1_ET00 := TRUE;   // SR flip-flop
   END_IF;
   IF #T1_ET08 THEN #T1_ET00 := FALSE; END_IF;
END_REGION

REGION Network 56: RESET TRANS OK
   RUNG wire#powerrail
      I_Contact( #T1_ET50 )
      I_Contact( #T1_ET60 )
      I_Contact( #T1_ET80 )
      R_Coil( #TRANS_OK )
   END_RUNG
   // the same network as SCL:
   IF NOT #T1_ET50 AND NOT #T1_ET60 AND NOT #T1_ET80 THEN #TRANS_OK := FALSE; END_IF;
END_REGION

REGION Network 57: #PRV_CARGA_OK
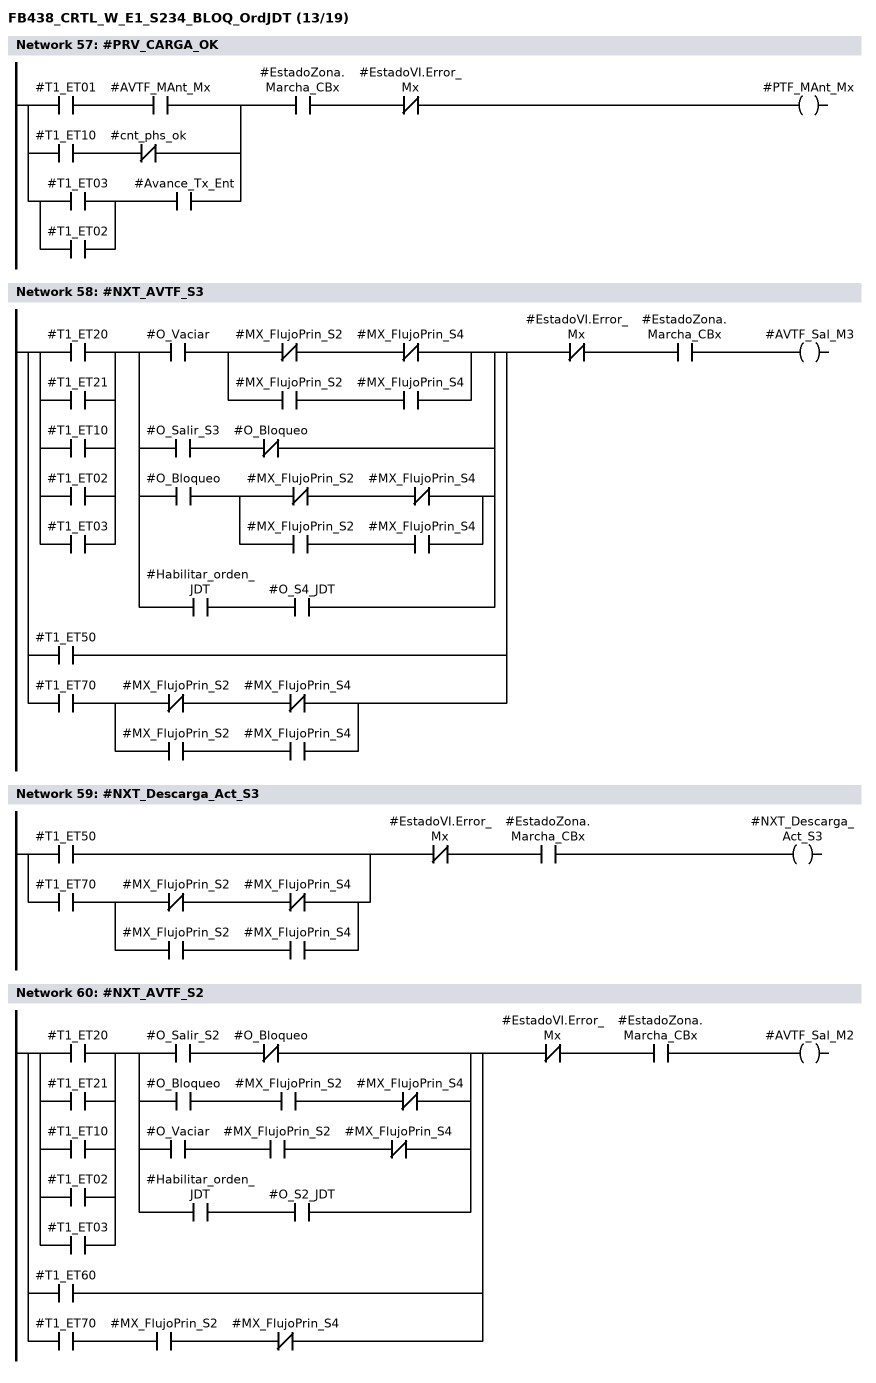
   RUNG wire#powerrail
      Contact( #T1_ET01 )
      Contact( #AVTF_MAnt_Mx )
      wire#w1
      Contact( #EstadoZona.Marcha_CBx )
      I_Contact( #EstadoVI.Error_Mx )
      Coil( #PTF_MAnt_Mx )
   END_RUNG
   RUNG wire#powerrail
      Contact( #T1_ET10 )
      I_Contact( #cnt_phs_ok )
   END_RUNG wire#w1
   RUNG wire#powerrail
      Contact( #T1_ET03 )
      wire#w2
      Contact( #Avance_Tx_Ent )
   END_RUNG wire#w1
   RUNG wire#powerrail
      Contact( #T1_ET02 )
   END_RUNG wire#w2
   // the same network as SCL:
   #PTF_MAnt_Mx := ((#T1_ET01 AND #AVTF_MAnt_Mx) OR (#T1_ET10 AND NOT #cnt_phs_ok) OR ((#T1_ET03 OR #T1_ET02) AND #Avance_Tx_Ent)) AND #EstadoZona.Marcha_CBx AND NOT #EstadoVI.Error_Mx;
END_REGION

REGION Network 58: #NXT_AVTF_S3
   RUNG wire#powerrail
      Contact( #T1_ET20 )
      wire#w1
      Contact( #O_Vaciar )
      wire#w2
      I_Contact( #MX_FlujoPrin_S2 )
      I_Contact( #MX_FlujoPrin_S4 )
      wire#w3
      I_Contact( #EstadoVI.Error_Mx )
      Contact( #EstadoZona.Marcha_CBx )
      Coil( #AVTF_Sal_M3 )
   END_RUNG
   RUNG wire#powerrail
      Contact( #T1_ET21 )
   END_RUNG wire#w1
   RUNG wire#powerrail
      Contact( #T1_ET10 )
   END_RUNG wire#w1
   RUNG wire#powerrail
      Contact( #T1_ET02 )
   END_RUNG wire#w1
   RUNG wire#powerrail
      Contact( #T1_ET03 )
   END_RUNG wire#w1
   RUNG wire#w2
      Contact( #MX_FlujoPrin_S2 )
      Contact( #MX_FlujoPrin_S4 )
   END_RUNG wire#w3
   RUNG wire#w1
      Contact( #O_Salir_S3 )
      I_Contact( #O_Bloqueo )
   END_RUNG wire#w3
   RUNG wire#w1
      Contact( #O_Bloqueo )
      wire#w4
      I_Contact( #MX_FlujoPrin_S2 )
      I_Contact( #MX_FlujoPrin_S4 )
   END_RUNG wire#w3
   RUNG wire#w4
      Contact( #MX_FlujoPrin_S2 )
      Contact( #MX_FlujoPrin_S4 )
   END_RUNG wire#w3
   RUNG wire#w1
      Contact( #Habilitar_orden_JDT )
      Contact( #O_S4_JDT )
   END_RUNG wire#w3
   RUNG wire#powerrail
      Contact( #T1_ET50 )
   END_RUNG wire#w3
   RUNG wire#powerrail
      Contact( #T1_ET70 )
      wire#w5
      I_Contact( #MX_FlujoPrin_S2 )
      I_Contact( #MX_FlujoPrin_S4 )
   END_RUNG wire#w3
   RUNG wire#w5
      Contact( #MX_FlujoPrin_S2 )
      Contact( #MX_FlujoPrin_S4 )
   END_RUNG wire#w3
   // the same network as SCL:
   #AVTF_Sal_M3 := (((#T1_ET20 OR #T1_ET21 OR #T1_ET10 OR #T1_ET02 OR #T1_ET03) AND ((#O_Vaciar AND ((NOT #MX_FlujoPrin_S2 AND NOT #MX_FlujoPrin_S4) OR (#MX_FlujoPrin_S2 AND #MX_FlujoPrin_S4))) OR (#O_Salir_S3 AND NOT #O_Bloqueo) OR (#O_Bloqueo AND ((NOT #MX_FlujoPrin_S2 AND NOT #MX_FlujoPrin_S4) OR (#MX_FlujoPrin_S2 AND #MX_FlujoPrin_S4))) OR (#Habilitar_orden_JDT AND #O_S4_JDT))) OR #T1_ET50 OR (#T1_ET70 AND ((NOT #MX_FlujoPrin_S2 AND NOT #MX_FlujoPrin_S4) OR (#MX_FlujoPrin_S2 AND #MX_FlujoPrin_S4)))) AND NOT #EstadoVI.Error_Mx AND #EstadoZona.Marcha_CBx;
END_REGION

REGION Network 59: #NXT_Descarga_Act_S3
   RUNG wire#powerrail
      Contact( #T1_ET50 )
      wire#w1
      I_Contact( #EstadoVI.Error_Mx )
      Contact( #EstadoZona.Marcha_CBx )
      Coil( #NXT_Descarga_Act_S3 )
   END_RUNG
   RUNG wire#powerrail
      Contact( #T1_ET70 )
      wire#w2
      I_Contact( #MX_FlujoPrin_S2 )
      I_Contact( #MX_FlujoPrin_S4 )
   END_RUNG wire#w1
   RUNG wire#w2
      Contact( #MX_FlujoPrin_S2 )
      Contact( #MX_FlujoPrin_S4 )
   END_RUNG wire#w1
   // the same network as SCL:
   #NXT_Descarga_Act_S3 := (#T1_ET50 OR (#T1_ET70 AND ((NOT #MX_FlujoPrin_S2 AND NOT #MX_FlujoPrin_S4) OR (#MX_FlujoPrin_S2 AND #MX_FlujoPrin_S4)))) AND NOT #EstadoVI.Error_Mx AND #EstadoZona.Marcha_CBx;
END_REGION

REGION Network 60: #NXT_AVTF_S2
   RUNG wire#powerrail
      Contact( #T1_ET20 )
      wire#w1
      Contact( #O_Salir_S2 )
      I_Contact( #O_Bloqueo )
      wire#w2
      I_Contact( #EstadoVI.Error_Mx )
      Contact( #EstadoZona.Marcha_CBx )
      Coil( #AVTF_Sal_M2 )
   END_RUNG
   RUNG wire#powerrail
      Contact( #T1_ET21 )
   END_RUNG wire#w1
   RUNG wire#powerrail
      Contact( #T1_ET10 )
   END_RUNG wire#w1
   RUNG wire#powerrail
      Contact( #T1_ET02 )
   END_RUNG wire#w1
   RUNG wire#powerrail
      Contact( #T1_ET03 )
   END_RUNG wire#w1
   RUNG wire#w1
      Contact( #O_Bloqueo )
      Contact( #MX_FlujoPrin_S2 )
      I_Contact( #MX_FlujoPrin_S4 )
   END_RUNG wire#w2
   RUNG wire#w1
      Contact( #O_Vaciar )
      Contact( #MX_FlujoPrin_S2 )
      I_Contact( #MX_FlujoPrin_S4 )
   END_RUNG wire#w2
   RUNG wire#w1
      Contact( #Habilitar_orden_JDT )
      Contact( #O_S2_JDT )
   END_RUNG wire#w2
   RUNG wire#powerrail
      Contact( #T1_ET60 )
   END_RUNG wire#w2
   RUNG wire#powerrail
      Contact( #T1_ET70 )
      Contact( #MX_FlujoPrin_S2 )
      I_Contact( #MX_FlujoPrin_S4 )
   END_RUNG wire#w2
   // the same network as SCL:
   #AVTF_Sal_M2 := (((#T1_ET20 OR #T1_ET21 OR #T1_ET10 OR #T1_ET02 OR #T1_ET03) AND ((#O_Salir_S2 AND NOT #O_Bloqueo) OR (#O_Bloqueo AND #MX_FlujoPrin_S2 AND NOT #MX_FlujoPrin_S4) OR (#O_Vaciar AND #MX_FlujoPrin_S2 AND NOT #MX_FlujoPrin_S4) OR (#Habilitar_orden_JDT AND #O_S2_JDT))) OR #T1_ET60 OR (#T1_ET70 AND #MX_FlujoPrin_S2 AND NOT #MX_FlujoPrin_S4)) AND NOT #EstadoVI.Error_Mx AND #EstadoZona.Marcha_CBx;
END_REGION

REGION Network 61: #NXT_AVTF_S4
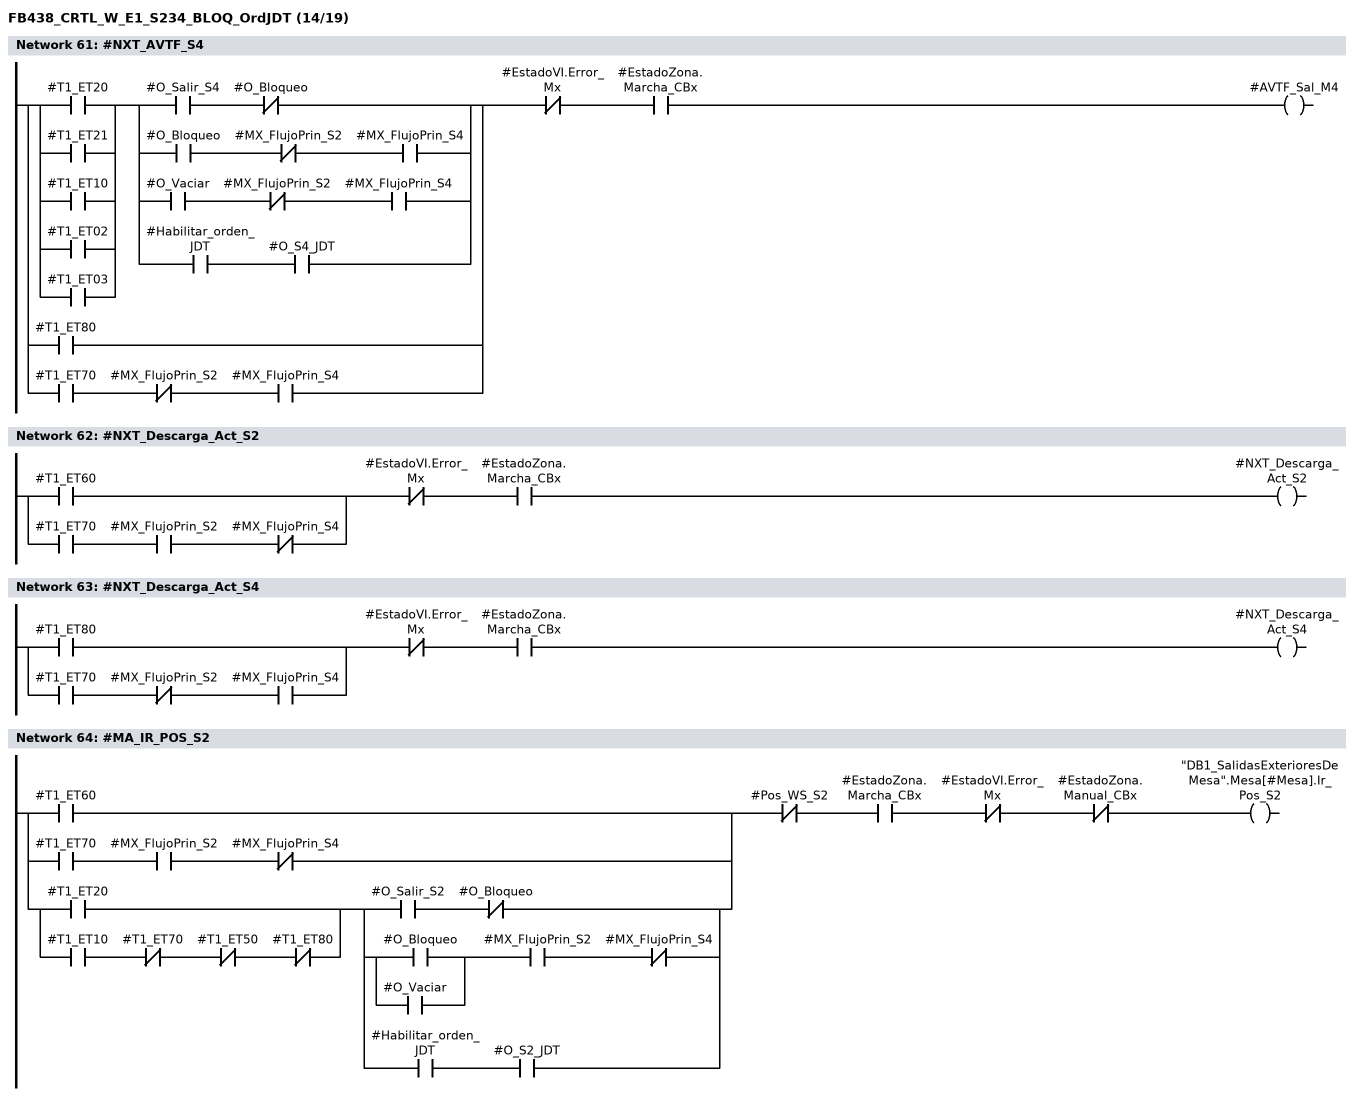
   RUNG wire#powerrail
      Contact( #T1_ET20 )
      wire#w1
      Contact( #O_Salir_S4 )
      I_Contact( #O_Bloqueo )
      wire#w2
      I_Contact( #EstadoVI.Error_Mx )
      Contact( #EstadoZona.Marcha_CBx )
      Coil( #AVTF_Sal_M4 )
   END_RUNG
   RUNG wire#powerrail
      Contact( #T1_ET21 )
   END_RUNG wire#w1
   RUNG wire#powerrail
      Contact( #T1_ET10 )
   END_RUNG wire#w1
   RUNG wire#powerrail
      Contact( #T1_ET02 )
   END_RUNG wire#w1
   RUNG wire#powerrail
      Contact( #T1_ET03 )
   END_RUNG wire#w1
   RUNG wire#w1
      Contact( #O_Bloqueo )
      I_Contact( #MX_FlujoPrin_S2 )
      Contact( #MX_FlujoPrin_S4 )
   END_RUNG wire#w2
   RUNG wire#w1
      Contact( #O_Vaciar )
      I_Contact( #MX_FlujoPrin_S2 )
      Contact( #MX_FlujoPrin_S4 )
   END_RUNG wire#w2
   RUNG wire#w1
      Contact( #Habilitar_orden_JDT )
      Contact( #O_S4_JDT )
   END_RUNG wire#w2
   RUNG wire#powerrail
      Contact( #T1_ET80 )
   END_RUNG wire#w2
   RUNG wire#powerrail
      Contact( #T1_ET70 )
      I_Contact( #MX_FlujoPrin_S2 )
      Contact( #MX_FlujoPrin_S4 )
   END_RUNG wire#w2
   // the same network as SCL:
   #AVTF_Sal_M4 := (((#T1_ET20 OR #T1_ET21 OR #T1_ET10 OR #T1_ET02 OR #T1_ET03) AND ((#O_Salir_S4 AND NOT #O_Bloqueo) OR (#O_Bloqueo AND NOT #MX_FlujoPrin_S2 AND #MX_FlujoPrin_S4) OR (#O_Vaciar AND NOT #MX_FlujoPrin_S2 AND #MX_FlujoPrin_S4) OR (#Habilitar_orden_JDT AND #O_S4_JDT))) OR #T1_ET80 OR (#T1_ET70 AND NOT #MX_FlujoPrin_S2 AND #MX_FlujoPrin_S4)) AND NOT #EstadoVI.Error_Mx AND #EstadoZona.Marcha_CBx;
END_REGION

REGION Network 62: #NXT_Descarga_Act_S2
   RUNG wire#powerrail
      Contact( #T1_ET60 )
      wire#w1
      I_Contact( #EstadoVI.Error_Mx )
      Contact( #EstadoZona.Marcha_CBx )
      Coil( #NXT_Descarga_Act_S2 )
   END_RUNG
   RUNG wire#powerrail
      Contact( #T1_ET70 )
      Contact( #MX_FlujoPrin_S2 )
      I_Contact( #MX_FlujoPrin_S4 )
   END_RUNG wire#w1
   // the same network as SCL:
   #NXT_Descarga_Act_S2 := (#T1_ET60 OR (#T1_ET70 AND #MX_FlujoPrin_S2 AND NOT #MX_FlujoPrin_S4)) AND NOT #EstadoVI.Error_Mx AND #EstadoZona.Marcha_CBx;
END_REGION

REGION Network 63: #NXT_Descarga_Act_S4
   RUNG wire#powerrail
      Contact( #T1_ET80 )
      wire#w1
      I_Contact( #EstadoVI.Error_Mx )
      Contact( #EstadoZona.Marcha_CBx )
      Coil( #NXT_Descarga_Act_S4 )
   END_RUNG
   RUNG wire#powerrail
      Contact( #T1_ET70 )
      I_Contact( #MX_FlujoPrin_S2 )
      Contact( #MX_FlujoPrin_S4 )
   END_RUNG wire#w1
   // the same network as SCL:
   #NXT_Descarga_Act_S4 := (#T1_ET80 OR (#T1_ET70 AND NOT #MX_FlujoPrin_S2 AND #MX_FlujoPrin_S4)) AND NOT #EstadoVI.Error_Mx AND #EstadoZona.Marcha_CBx;
END_REGION

REGION Network 64: #MA_IR_POS_S2
   RUNG wire#powerrail
      Contact( #T1_ET60 )
      wire#w1
      I_Contact( #Pos_WS_S2 )
      Contact( #EstadoZona.Marcha_CBx )
      I_Contact( #EstadoVI.Error_Mx )
      I_Contact( #EstadoZona.Manual_CBx )
      Coil( "DB1_SalidasExterioresDeMesa".Mesa[#Mesa].Ir_Pos_S2 )
   END_RUNG
   RUNG wire#powerrail
      Contact( #T1_ET70 )
      Contact( #MX_FlujoPrin_S2 )
      I_Contact( #MX_FlujoPrin_S4 )
   END_RUNG wire#w1
   RUNG wire#powerrail
      Contact( #T1_ET20 )
      wire#w2
      Contact( #O_Salir_S2 )
      I_Contact( #O_Bloqueo )
   END_RUNG wire#w1
   RUNG wire#powerrail
      Contact( #T1_ET10 )
      I_Contact( #T1_ET70 )
      I_Contact( #T1_ET50 )
      I_Contact( #T1_ET80 )
   END_RUNG wire#w2
   RUNG wire#w2
      Contact( #O_Bloqueo )
      wire#w3
      Contact( #MX_FlujoPrin_S2 )
      I_Contact( #MX_FlujoPrin_S4 )
   END_RUNG wire#w1
   RUNG wire#w2
      Contact( #O_Vaciar )
   END_RUNG wire#w3
   RUNG wire#w2
      Contact( #Habilitar_orden_JDT )
      Contact( #O_S2_JDT )
   END_RUNG wire#w1
   // the same network as SCL:
   "DB1_SalidasExterioresDeMesa".Mesa[#Mesa].Ir_Pos_S2 := (#T1_ET60 OR (#T1_ET70 AND #MX_FlujoPrin_S2 AND NOT #MX_FlujoPrin_S4) OR ((#T1_ET20 OR (#T1_ET10 AND NOT #T1_ET70 AND NOT #T1_ET50 AND NOT #T1_ET80)) AND ((#O_Salir_S2 AND NOT #O_Bloqueo) OR ((#O_Bloqueo OR #O_Vaciar) AND #MX_FlujoPrin_S2 AND NOT #MX_FlujoPrin_S4) OR (#Habilitar_orden_JDT AND #O_S2_JDT)))) AND NOT #Pos_WS_S2 AND #EstadoZona.Marcha_CBx AND NOT #EstadoVI.Error_Mx AND NOT #EstadoZona.Manual_CBx;
END_REGION

REGION Network 65: #MA_IR_POS_S4
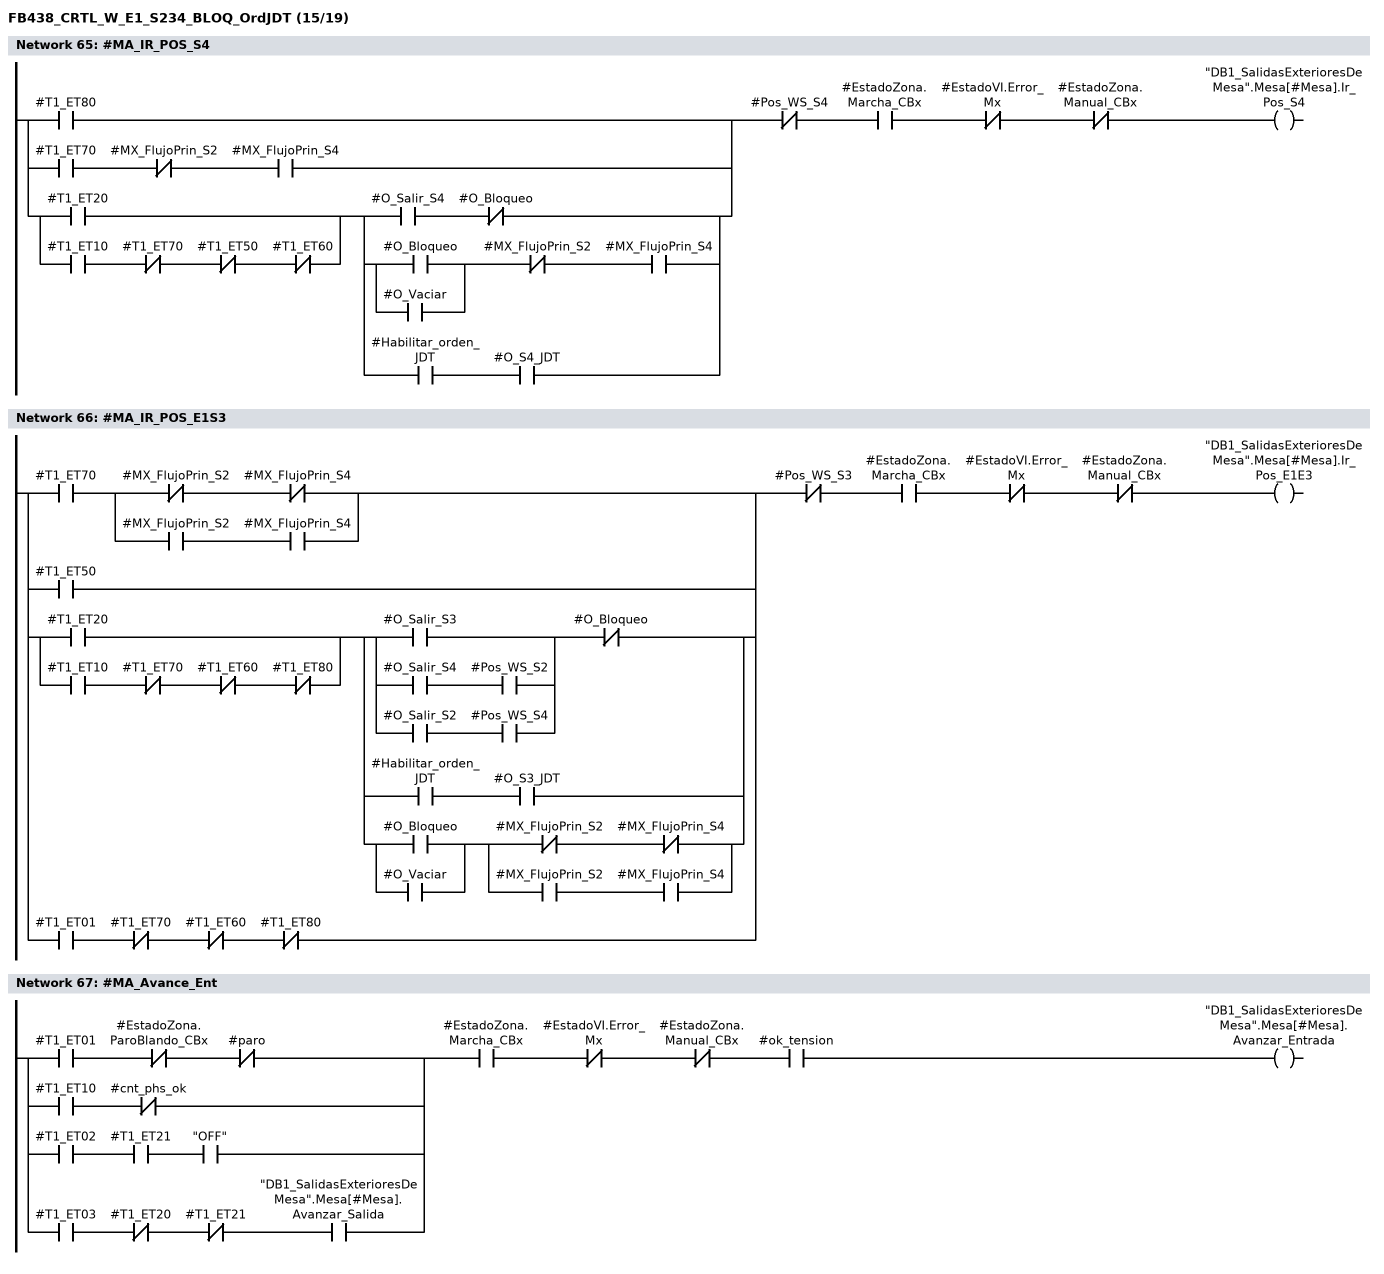
   RUNG wire#powerrail
      Contact( #T1_ET80 )
      wire#w1
      I_Contact( #Pos_WS_S4 )
      Contact( #EstadoZona.Marcha_CBx )
      I_Contact( #EstadoVI.Error_Mx )
      I_Contact( #EstadoZona.Manual_CBx )
      Coil( "DB1_SalidasExterioresDeMesa".Mesa[#Mesa].Ir_Pos_S4 )
   END_RUNG
   RUNG wire#powerrail
      Contact( #T1_ET70 )
      I_Contact( #MX_FlujoPrin_S2 )
      Contact( #MX_FlujoPrin_S4 )
   END_RUNG wire#w1
   RUNG wire#powerrail
      Contact( #T1_ET20 )
      wire#w2
      Contact( #O_Salir_S4 )
      I_Contact( #O_Bloqueo )
   END_RUNG wire#w1
   RUNG wire#powerrail
      Contact( #T1_ET10 )
      I_Contact( #T1_ET70 )
      I_Contact( #T1_ET50 )
      I_Contact( #T1_ET60 )
   END_RUNG wire#w2
   RUNG wire#w2
      Contact( #O_Bloqueo )
      wire#w3
      I_Contact( #MX_FlujoPrin_S2 )
      Contact( #MX_FlujoPrin_S4 )
   END_RUNG wire#w1
   RUNG wire#w2
      Contact( #O_Vaciar )
   END_RUNG wire#w3
   RUNG wire#w2
      Contact( #Habilitar_orden_JDT )
      Contact( #O_S4_JDT )
   END_RUNG wire#w1
   // the same network as SCL:
   "DB1_SalidasExterioresDeMesa".Mesa[#Mesa].Ir_Pos_S4 := (#T1_ET80 OR (#T1_ET70 AND NOT #MX_FlujoPrin_S2 AND #MX_FlujoPrin_S4) OR ((#T1_ET20 OR (#T1_ET10 AND NOT #T1_ET70 AND NOT #T1_ET50 AND NOT #T1_ET60)) AND ((#O_Salir_S4 AND NOT #O_Bloqueo) OR ((#O_Bloqueo OR #O_Vaciar) AND NOT #MX_FlujoPrin_S2 AND #MX_FlujoPrin_S4) OR (#Habilitar_orden_JDT AND #O_S4_JDT)))) AND NOT #Pos_WS_S4 AND #EstadoZona.Marcha_CBx AND NOT #EstadoVI.Error_Mx AND NOT #EstadoZona.Manual_CBx;
END_REGION

REGION Network 66: #MA_IR_POS_E1S3
   RUNG wire#powerrail
      Contact( #T1_ET70 )
      wire#w1
      I_Contact( #MX_FlujoPrin_S2 )
      I_Contact( #MX_FlujoPrin_S4 )
      wire#w2
      I_Contact( #Pos_WS_S3 )
      Contact( #EstadoZona.Marcha_CBx )
      I_Contact( #EstadoVI.Error_Mx )
      I_Contact( #EstadoZona.Manual_CBx )
      Coil( "DB1_SalidasExterioresDeMesa".Mesa[#Mesa].Ir_Pos_E1E3 )
   END_RUNG
   RUNG wire#w1
      Contact( #MX_FlujoPrin_S2 )
      Contact( #MX_FlujoPrin_S4 )
   END_RUNG wire#w2
   RUNG wire#powerrail
      Contact( #T1_ET50 )
   END_RUNG wire#w2
   RUNG wire#powerrail
      Contact( #T1_ET20 )
      wire#w3
      Contact( #O_Salir_S3 )
      wire#w4
      I_Contact( #O_Bloqueo )
   END_RUNG wire#w2
   RUNG wire#powerrail
      Contact( #T1_ET10 )
      I_Contact( #T1_ET70 )
      I_Contact( #T1_ET60 )
      I_Contact( #T1_ET80 )
   END_RUNG wire#w3
   RUNG wire#w3
      Contact( #O_Salir_S4 )
      Contact( #Pos_WS_S2 )
   END_RUNG wire#w4
   RUNG wire#w3
      Contact( #O_Salir_S2 )
      Contact( #Pos_WS_S4 )
   END_RUNG wire#w4
   RUNG wire#w3
      Contact( #Habilitar_orden_JDT )
      Contact( #O_S3_JDT )
   END_RUNG wire#w2
   RUNG wire#w3
      Contact( #O_Bloqueo )
      wire#w5
      I_Contact( #MX_FlujoPrin_S2 )
      I_Contact( #MX_FlujoPrin_S4 )
   END_RUNG wire#w2
   RUNG wire#w3
      Contact( #O_Vaciar )
   END_RUNG wire#w5
   RUNG wire#w5
      Contact( #MX_FlujoPrin_S2 )
      Contact( #MX_FlujoPrin_S4 )
   END_RUNG wire#w2
   RUNG wire#powerrail
      Contact( #T1_ET01 )
      I_Contact( #T1_ET70 )
      I_Contact( #T1_ET60 )
      I_Contact( #T1_ET80 )
   END_RUNG wire#w2
   // the same network as SCL:
   "DB1_SalidasExterioresDeMesa".Mesa[#Mesa].Ir_Pos_E1E3 := ((#T1_ET70 AND ((NOT #MX_FlujoPrin_S2 AND NOT #MX_FlujoPrin_S4) OR (#MX_FlujoPrin_S2 AND #MX_FlujoPrin_S4))) OR #T1_ET50 OR ((#T1_ET20 OR (#T1_ET10 AND NOT #T1_ET70 AND NOT #T1_ET60 AND NOT #T1_ET80)) AND (((#O_Salir_S3 OR (#O_Salir_S4 AND #Pos_WS_S2) OR (#O_Salir_S2 AND #Pos_WS_S4)) AND NOT #O_Bloqueo) OR (#Habilitar_orden_JDT AND #O_S3_JDT) OR ((#O_Bloqueo OR #O_Vaciar) AND ((NOT #MX_FlujoPrin_S2 AND NOT #MX_FlujoPrin_S4) OR (#MX_FlujoPrin_S2 AND #MX_FlujoPrin_S4))))) OR (#T1_ET01 AND NOT #T1_ET70 AND NOT #T1_ET60 AND NOT #T1_ET80)) AND NOT #Pos_WS_S3 AND #EstadoZona.Marcha_CBx AND NOT #EstadoVI.Error_Mx AND NOT #EstadoZona.Manual_CBx;
END_REGION

REGION Network 67: #MA_Avance_Ent
   RUNG wire#powerrail
      Contact( #T1_ET01 )
      I_Contact( #EstadoZona.ParoBlando_CBx )
      I_Contact( #paro )
      wire#w1
      Contact( #EstadoZona.Marcha_CBx )
      I_Contact( #EstadoVI.Error_Mx )
      I_Contact( #EstadoZona.Manual_CBx )
      Contact( #ok_tension )
      Coil( "DB1_SalidasExterioresDeMesa".Mesa[#Mesa].Avanzar_Entrada )
   END_RUNG
   RUNG wire#powerrail
      Contact( #T1_ET10 )
      I_Contact( #cnt_phs_ok )
   END_RUNG wire#w1
   RUNG wire#powerrail
      Contact( #T1_ET02 )
      Contact( #T1_ET21 )
      Contact( "OFF" )
   END_RUNG wire#w1
   RUNG wire#powerrail
      Contact( #T1_ET03 )
      I_Contact( #T1_ET20 )
      I_Contact( #T1_ET21 )
      Contact( "DB1_SalidasExterioresDeMesa".Mesa[#Mesa].Avanzar_Salida )
   END_RUNG wire#w1
   // the same network as SCL:
   "DB1_SalidasExterioresDeMesa".Mesa[#Mesa].Avanzar_Entrada := ((#T1_ET01 AND NOT #EstadoZona.ParoBlando_CBx AND NOT #paro) OR (#T1_ET10 AND NOT #cnt_phs_ok) OR (#T1_ET02 AND #T1_ET21 AND "OFF") OR (#T1_ET03 AND NOT #T1_ET20 AND NOT #T1_ET21 AND "DB1_SalidasExterioresDeMesa".Mesa[#Mesa].Avanzar_Salida)) AND #EstadoZona.Marcha_CBx AND NOT #EstadoVI.Error_Mx AND NOT #EstadoZona.Manual_CBx AND #ok_tension;
END_REGION

REGION Network 68: #MA_Avance_Sal
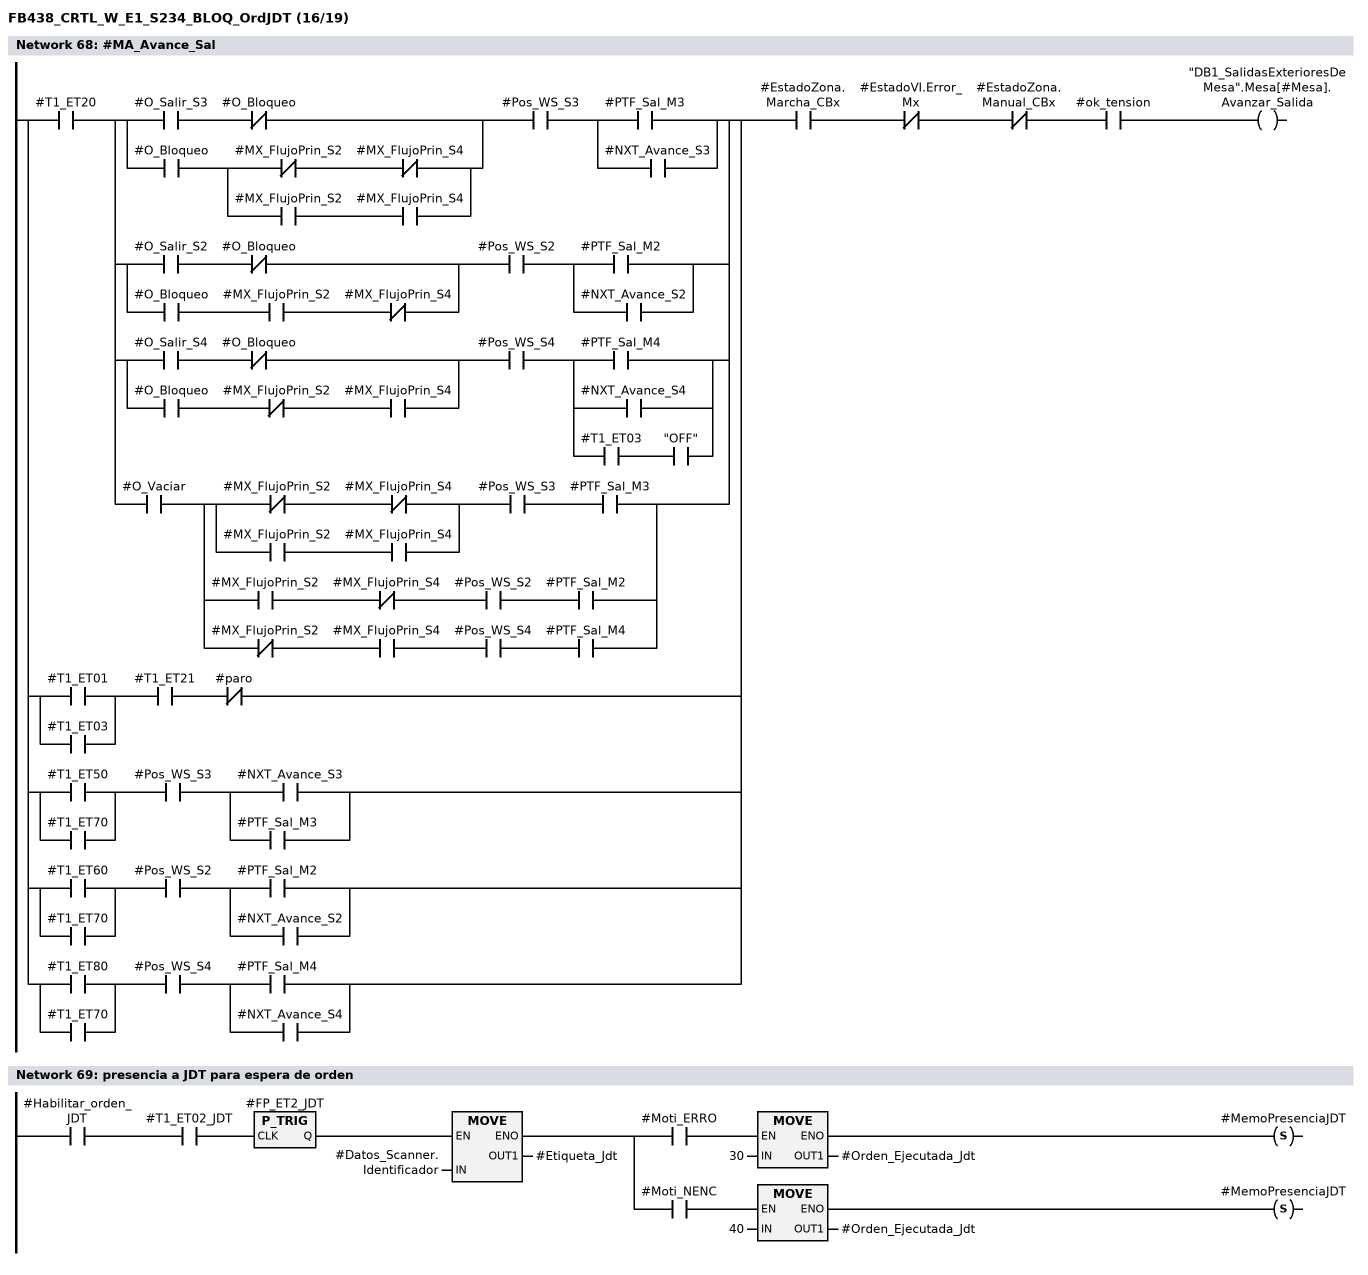
   RUNG wire#powerrail
      Contact( #T1_ET20 )
      wire#w1
      Contact( #O_Salir_S3 )
      I_Contact( #O_Bloqueo )
      wire#w2
      Contact( #Pos_WS_S3 )
      wire#w4
      Contact( #PTF_Sal_M3 )
      wire#w5
      Contact( #EstadoZona.Marcha_CBx )
      I_Contact( #EstadoVI.Error_Mx )
      I_Contact( #EstadoZona.Manual_CBx )
      Contact( #ok_tension )
      Coil( "DB1_SalidasExterioresDeMesa".Mesa[#Mesa].Avanzar_Salida )
   END_RUNG
   RUNG wire#w1
      Contact( #O_Bloqueo )
      wire#w3
      I_Contact( #MX_FlujoPrin_S2 )
      I_Contact( #MX_FlujoPrin_S4 )
   END_RUNG wire#w2
   RUNG wire#w3
      Contact( #MX_FlujoPrin_S2 )
      Contact( #MX_FlujoPrin_S4 )
   END_RUNG wire#w2
   RUNG wire#w4
      Contact( #NXT_Avance_S3 )
   END_RUNG wire#w5
   RUNG wire#w1
      Contact( #O_Salir_S2 )
      I_Contact( #O_Bloqueo )
      wire#w6
      Contact( #Pos_WS_S2 )
      wire#w7
      Contact( #PTF_Sal_M2 )
   END_RUNG wire#w5
   RUNG wire#w1
      Contact( #O_Bloqueo )
      Contact( #MX_FlujoPrin_S2 )
      I_Contact( #MX_FlujoPrin_S4 )
   END_RUNG wire#w6
   RUNG wire#w7
      Contact( #NXT_Avance_S2 )
   END_RUNG wire#w5
   RUNG wire#w1
      Contact( #O_Salir_S4 )
      I_Contact( #O_Bloqueo )
      wire#w8
      Contact( #Pos_WS_S4 )
      wire#w9
      Contact( #PTF_Sal_M4 )
   END_RUNG wire#w5
   RUNG wire#w1
      Contact( #O_Bloqueo )
      I_Contact( #MX_FlujoPrin_S2 )
      Contact( #MX_FlujoPrin_S4 )
   END_RUNG wire#w8
   RUNG wire#w9
      Contact( #NXT_Avance_S4 )
   END_RUNG wire#w5
   RUNG wire#w9
      Contact( #T1_ET03 )
      Contact( "OFF" )
   END_RUNG wire#w5
   RUNG wire#w1
      Contact( #O_Vaciar )
      wire#w10
      I_Contact( #MX_FlujoPrin_S2 )
      I_Contact( #MX_FlujoPrin_S4 )
      wire#w11
      Contact( #Pos_WS_S3 )
      Contact( #PTF_Sal_M3 )
   END_RUNG wire#w5
   RUNG wire#w10
      Contact( #MX_FlujoPrin_S2 )
      Contact( #MX_FlujoPrin_S4 )
   END_RUNG wire#w11
   RUNG wire#w10
      Contact( #MX_FlujoPrin_S2 )
      I_Contact( #MX_FlujoPrin_S4 )
      Contact( #Pos_WS_S2 )
      Contact( #PTF_Sal_M2 )
   END_RUNG wire#w5
   RUNG wire#w10
      I_Contact( #MX_FlujoPrin_S2 )
      Contact( #MX_FlujoPrin_S4 )
      Contact( #Pos_WS_S4 )
      Contact( #PTF_Sal_M4 )
   END_RUNG wire#w5
   RUNG wire#powerrail
      Contact( #T1_ET01 )
      wire#w12
      Contact( #T1_ET21 )
      I_Contact( #paro )
   END_RUNG wire#w5
   RUNG wire#powerrail
      Contact( #T1_ET03 )
   END_RUNG wire#w12
   RUNG wire#powerrail
      Contact( #T1_ET50 )
      wire#w13
      Contact( #Pos_WS_S3 )
      wire#w14
      Contact( #NXT_Avance_S3 )
   END_RUNG wire#w5
   RUNG wire#powerrail
      Contact( #T1_ET70 )
   END_RUNG wire#w13
   RUNG wire#w14
      Contact( #PTF_Sal_M3 )
   END_RUNG wire#w5
   RUNG wire#powerrail
      Contact( #T1_ET60 )
      wire#w15
      Contact( #Pos_WS_S2 )
      wire#w16
      Contact( #PTF_Sal_M2 )
   END_RUNG wire#w5
   RUNG wire#powerrail
      Contact( #T1_ET70 )
   END_RUNG wire#w15
   RUNG wire#w16
      Contact( #NXT_Avance_S2 )
   END_RUNG wire#w5
   RUNG wire#powerrail
      Contact( #T1_ET80 )
      wire#w17
      Contact( #Pos_WS_S4 )
      wire#w18
      Contact( #PTF_Sal_M4 )
   END_RUNG wire#w5
   RUNG wire#powerrail
      Contact( #T1_ET70 )
   END_RUNG wire#w17
   RUNG wire#w18
      Contact( #NXT_Avance_S4 )
   END_RUNG wire#w5
   // the same network as SCL:
   "DB1_SalidasExterioresDeMesa".Mesa[#Mesa].Avanzar_Salida := ((#T1_ET20 AND ((((#O_Salir_S3 AND NOT #O_Bloqueo) OR (#O_Bloqueo AND ((NOT #MX_FlujoPrin_S2 AND NOT #MX_FlujoPrin_S4) OR (#MX_FlujoPrin_S2 AND #MX_FlujoPrin_S4)))) AND #Pos_WS_S3 AND (#PTF_Sal_M3 OR #NXT_Avance_S3)) OR (((#O_Salir_S2 AND NOT #O_Bloqueo) OR (#O_Bloqueo AND #MX_FlujoPrin_S2 AND NOT #MX_FlujoPrin_S4)) AND #Pos_WS_S2 AND (#PTF_Sal_M2 OR #NXT_Avance_S2)) OR (((#O_Salir_S4 AND NOT #O_Bloqueo) OR (#O_Bloqueo AND NOT #MX_FlujoPrin_S2 AND #MX_FlujoPrin_S4)) AND #Pos_WS_S4 AND (#PTF_Sal_M4 OR #NXT_Avance_S4 OR (#T1_ET03 AND "OFF"))) OR (#O_Vaciar AND ((((NOT #MX_FlujoPrin_S2 AND NOT #MX_FlujoPrin_S4) OR (#MX_FlujoPrin_S2 AND #MX_FlujoPrin_S4)) AND #Pos_WS_S3 AND #PTF_Sal_M3) OR (#MX_FlujoPrin_S2 AND NOT #MX_FlujoPrin_S4 AND #Pos_WS_S2 AND #PTF_Sal_M2) OR (NOT #MX_FlujoPrin_S2 AND #MX_FlujoPrin_S4 AND #Pos_WS_S4 AND #PTF_Sal_M4))))) OR ((#T1_ET01 OR #T1_ET03) AND #T1_ET21 AND NOT #paro) OR ((#T1_ET50 OR #T1_ET70) AND #Pos_WS_S3 AND (#NXT_Avance_S3 OR #PTF_Sal_M3)) OR ((#T1_ET60 OR #T1_ET70) AND #Pos_WS_S2 AND (#PTF_Sal_M2 OR #NXT_Avance_S2)) OR ((#T1_ET80 OR #T1_ET70) AND #Pos_WS_S4 AND (#PTF_Sal_M4 OR #NXT_Avance_S4))) AND #EstadoZona.Marcha_CBx AND NOT #EstadoVI.Error_Mx AND NOT #EstadoZona.Manual_CBx AND #ok_tension;
END_REGION

REGION Network 69: presencia a JDT para espera de orden
   RUNG wire#powerrail
      Contact( #Habilitar_orden_JDT )
      Contact( #T1_ET02_JDT )
      P_Trig( #FP_ET2_JDT )
      { S7_GenerateENO := "TRUE" } Move(in := #Datos_Scanner.Identificador, out1 => #Etiqueta_Jdt)
      wire#w1
      Contact( #Moti_ERRO )
      { S7_GenerateENO := "TRUE" } Move(in := 30, out1 => #Orden_Ejecutada_Jdt)
      S_Coil( #MemoPresenciaJDT )
   END_RUNG
   RUNG wire#w1
      Contact( #Moti_NENC )
      { S7_GenerateENO := "TRUE" } Move(in := 40, out1 => #Orden_Ejecutada_Jdt)
      S_Coil( #MemoPresenciaJDT )
   END_RUNG
   // the same network as SCL:
   // ENO of a box is taken as its EN; it also drops when the box reports an error
   #_w1 := #Habilitar_orden_JDT AND #T1_ET02_JDT;
   #_w2 := #_w1 AND NOT #FP_ET2_JDT;   // rising edge
   #FP_ET2_JDT := #_w1;
   IF #_w2 THEN #Etiqueta_Jdt := #Datos_Scanner.Identificador; END_IF;
   IF #_w2 AND #Moti_ERRO THEN
       #Orden_Ejecutada_Jdt := 30;
       #MemoPresenciaJDT := TRUE;
   END_IF;
   IF #_w2 AND #Moti_NENC THEN
       #Orden_Ejecutada_Jdt := 40;
       #MemoPresenciaJDT := TRUE;
   END_IF;
END_REGION

REGION Network 70: PASAR ETIQUETA JDT
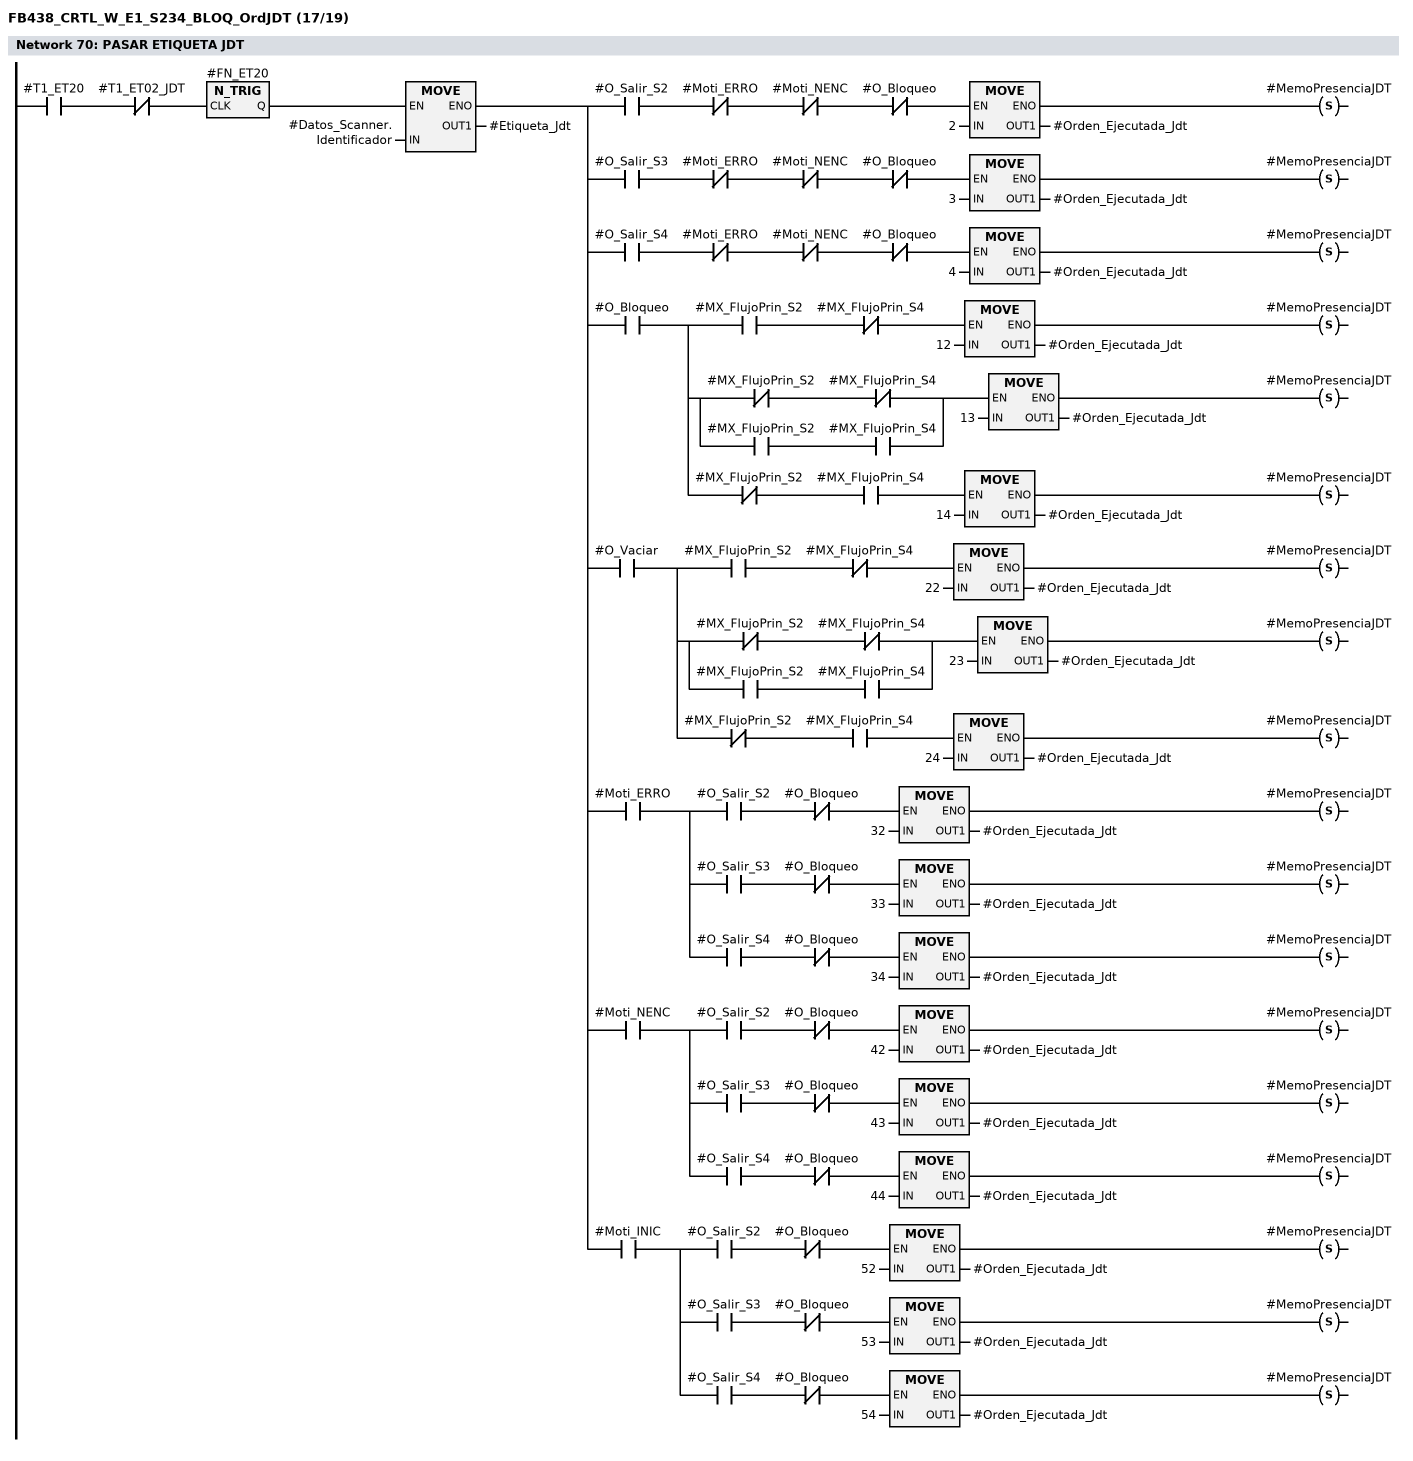
   RUNG wire#powerrail
      Contact( #T1_ET20 )
      I_Contact( #T1_ET02_JDT )
      N_Trig( #FN_ET20 )
      { S7_GenerateENO := "TRUE" } Move(in := #Datos_Scanner.Identificador, out1 => #Etiqueta_Jdt)
      wire#w1
      Contact( #O_Salir_S2 )
      I_Contact( #Moti_ERRO )
      I_Contact( #Moti_NENC )
      I_Contact( #O_Bloqueo )
      { S7_GenerateENO := "TRUE" } Move(in := 2, out1 => #Orden_Ejecutada_Jdt)
      S_Coil( #MemoPresenciaJDT )
   END_RUNG
   RUNG wire#w1
      Contact( #O_Salir_S3 )
      I_Contact( #Moti_ERRO )
      I_Contact( #Moti_NENC )
      I_Contact( #O_Bloqueo )
      { S7_GenerateENO := "TRUE" } Move(in := 3, out1 => #Orden_Ejecutada_Jdt)
      S_Coil( #MemoPresenciaJDT )
   END_RUNG
   RUNG wire#w1
      Contact( #O_Salir_S4 )
      I_Contact( #Moti_ERRO )
      I_Contact( #Moti_NENC )
      I_Contact( #O_Bloqueo )
      { S7_GenerateENO := "TRUE" } Move(in := 4, out1 => #Orden_Ejecutada_Jdt)
      S_Coil( #MemoPresenciaJDT )
   END_RUNG
   RUNG wire#w1
      Contact( #O_Bloqueo )
      wire#w2
      Contact( #MX_FlujoPrin_S2 )
      I_Contact( #MX_FlujoPrin_S4 )
      { S7_GenerateENO := "TRUE" } Move(in := 12, out1 => #Orden_Ejecutada_Jdt)
      S_Coil( #MemoPresenciaJDT )
   END_RUNG
   RUNG wire#w2
      I_Contact( #MX_FlujoPrin_S2 )
      I_Contact( #MX_FlujoPrin_S4 )
      wire#w3
      { S7_GenerateENO := "TRUE" } Move(in := 13, out1 => #Orden_Ejecutada_Jdt)
      S_Coil( #MemoPresenciaJDT )
   END_RUNG
   RUNG wire#w2
      Contact( #MX_FlujoPrin_S2 )
      Contact( #MX_FlujoPrin_S4 )
   END_RUNG wire#w3
   RUNG wire#w2
      I_Contact( #MX_FlujoPrin_S2 )
      Contact( #MX_FlujoPrin_S4 )
      { S7_GenerateENO := "TRUE" } Move(in := 14, out1 => #Orden_Ejecutada_Jdt)
      S_Coil( #MemoPresenciaJDT )
   END_RUNG
   RUNG wire#w1
      Contact( #O_Vaciar )
      wire#w4
      Contact( #MX_FlujoPrin_S2 )
      I_Contact( #MX_FlujoPrin_S4 )
      { S7_GenerateENO := "TRUE" } Move(in := 22, out1 => #Orden_Ejecutada_Jdt)
      S_Coil( #MemoPresenciaJDT )
   END_RUNG
   RUNG wire#w4
      I_Contact( #MX_FlujoPrin_S2 )
      I_Contact( #MX_FlujoPrin_S4 )
      wire#w5
      { S7_GenerateENO := "TRUE" } Move(in := 23, out1 => #Orden_Ejecutada_Jdt)
      S_Coil( #MemoPresenciaJDT )
   END_RUNG
   RUNG wire#w4
      Contact( #MX_FlujoPrin_S2 )
      Contact( #MX_FlujoPrin_S4 )
   END_RUNG wire#w5
   RUNG wire#w4
      I_Contact( #MX_FlujoPrin_S2 )
      Contact( #MX_FlujoPrin_S4 )
      { S7_GenerateENO := "TRUE" } Move(in := 24, out1 => #Orden_Ejecutada_Jdt)
      S_Coil( #MemoPresenciaJDT )
   END_RUNG
   RUNG wire#w1
      Contact( #Moti_ERRO )
      wire#w6
      Contact( #O_Salir_S2 )
      I_Contact( #O_Bloqueo )
      { S7_GenerateENO := "TRUE" } Move(in := 32, out1 => #Orden_Ejecutada_Jdt)
      S_Coil( #MemoPresenciaJDT )
   END_RUNG
   RUNG wire#w6
      Contact( #O_Salir_S3 )
      I_Contact( #O_Bloqueo )
      { S7_GenerateENO := "TRUE" } Move(in := 33, out1 => #Orden_Ejecutada_Jdt)
      S_Coil( #MemoPresenciaJDT )
   END_RUNG
   RUNG wire#w6
      Contact( #O_Salir_S4 )
      I_Contact( #O_Bloqueo )
      { S7_GenerateENO := "TRUE" } Move(in := 34, out1 => #Orden_Ejecutada_Jdt)
      S_Coil( #MemoPresenciaJDT )
   END_RUNG
   RUNG wire#w1
      Contact( #Moti_NENC )
      wire#w7
      Contact( #O_Salir_S2 )
      I_Contact( #O_Bloqueo )
      { S7_GenerateENO := "TRUE" } Move(in := 42, out1 => #Orden_Ejecutada_Jdt)
      S_Coil( #MemoPresenciaJDT )
   END_RUNG
   RUNG wire#w7
      Contact( #O_Salir_S3 )
      I_Contact( #O_Bloqueo )
      { S7_GenerateENO := "TRUE" } Move(in := 43, out1 => #Orden_Ejecutada_Jdt)
      S_Coil( #MemoPresenciaJDT )
   END_RUNG
   RUNG wire#w7
      Contact( #O_Salir_S4 )
      I_Contact( #O_Bloqueo )
      { S7_GenerateENO := "TRUE" } Move(in := 44, out1 => #Orden_Ejecutada_Jdt)
      S_Coil( #MemoPresenciaJDT )
   END_RUNG
   RUNG wire#w1
      Contact( #Moti_INIC )
      wire#w8
      Contact( #O_Salir_S2 )
      I_Contact( #O_Bloqueo )
      { S7_GenerateENO := "TRUE" } Move(in := 52, out1 => #Orden_Ejecutada_Jdt)
      S_Coil( #MemoPresenciaJDT )
   END_RUNG
   RUNG wire#w8
      Contact( #O_Salir_S3 )
      I_Contact( #O_Bloqueo )
      { S7_GenerateENO := "TRUE" } Move(in := 53, out1 => #Orden_Ejecutada_Jdt)
      S_Coil( #MemoPresenciaJDT )
   END_RUNG
   RUNG wire#w8
      Contact( #O_Salir_S4 )
      I_Contact( #O_Bloqueo )
      { S7_GenerateENO := "TRUE" } Move(in := 54, out1 => #Orden_Ejecutada_Jdt)
      S_Coil( #MemoPresenciaJDT )
   END_RUNG
   // the same network as SCL:
   // ENO of a box is taken as its EN; it also drops when the box reports an error
   #_w1 := #T1_ET20 AND NOT #T1_ET02_JDT;
   #_w2 := NOT #_w1 AND #FN_ET20;   // falling edge
   #FN_ET20 := #_w1;
   IF #_w2 THEN #Etiqueta_Jdt := #Datos_Scanner.Identificador; END_IF;
   IF #_w2 AND #O_Salir_S2 AND NOT #Moti_ERRO AND NOT #Moti_NENC AND NOT #O_Bloqueo THEN
       #Orden_Ejecutada_Jdt := 2;
       #MemoPresenciaJDT := TRUE;
   END_IF;
   IF #_w2 AND #O_Salir_S3 AND NOT #Moti_ERRO AND NOT #Moti_NENC AND NOT #O_Bloqueo THEN
       #Orden_Ejecutada_Jdt := 3;
       #MemoPresenciaJDT := TRUE;
   END_IF;
   IF #_w2 AND #O_Salir_S4 AND NOT #Moti_ERRO AND NOT #Moti_NENC AND NOT #O_Bloqueo THEN
       #Orden_Ejecutada_Jdt := 4;
       #MemoPresenciaJDT := TRUE;
   END_IF;
   #_w3 := #_w2 AND #O_Bloqueo;
   IF #_w3 AND #MX_FlujoPrin_S2 AND NOT #MX_FlujoPrin_S4 THEN
       #Orden_Ejecutada_Jdt := 12;
       #MemoPresenciaJDT := TRUE;
   END_IF;
   IF #_w3 AND ((NOT #MX_FlujoPrin_S2 AND NOT #MX_FlujoPrin_S4) OR (#MX_FlujoPrin_S2 AND #MX_FlujoPrin_S4)) THEN
       #Orden_Ejecutada_Jdt := 13;
       #MemoPresenciaJDT := TRUE;
   END_IF;
   IF #_w3 AND NOT #MX_FlujoPrin_S2 AND #MX_FlujoPrin_S4 THEN
       #Orden_Ejecutada_Jdt := 14;
       #MemoPresenciaJDT := TRUE;
   END_IF;
   #_w4 := #_w2 AND #O_Vaciar;
   IF #_w4 AND #MX_FlujoPrin_S2 AND NOT #MX_FlujoPrin_S4 THEN
       #Orden_Ejecutada_Jdt := 22;
       #MemoPresenciaJDT := TRUE;
   END_IF;
   IF #_w4 AND ((NOT #MX_FlujoPrin_S2 AND NOT #MX_FlujoPrin_S4) OR (#MX_FlujoPrin_S2 AND #MX_FlujoPrin_S4)) THEN
       #Orden_Ejecutada_Jdt := 23;
       #MemoPresenciaJDT := TRUE;
   END_IF;
   IF #_w4 AND NOT #MX_FlujoPrin_S2 AND #MX_FlujoPrin_S4 THEN
       #Orden_Ejecutada_Jdt := 24;
       #MemoPresenciaJDT := TRUE;
   END_IF;
   #_w5 := #_w2 AND #Moti_ERRO;
   IF #_w5 AND #O_Salir_S2 AND NOT #O_Bloqueo THEN
       #Orden_Ejecutada_Jdt := 32;
       #MemoPresenciaJDT := TRUE;
   END_IF;
   IF #_w5 AND #O_Salir_S3 AND NOT #O_Bloqueo THEN
       #Orden_Ejecutada_Jdt := 33;
       #MemoPresenciaJDT := TRUE;
   END_IF;
   IF #_w5 AND #O_Salir_S4 AND NOT #O_Bloqueo THEN
       #Orden_Ejecutada_Jdt := 34;
       #MemoPresenciaJDT := TRUE;
   END_IF;
   #_w6 := #_w2 AND #Moti_NENC;
   IF #_w6 AND #O_Salir_S2 AND NOT #O_Bloqueo THEN
       #Orden_Ejecutada_Jdt := 42;
       #MemoPresenciaJDT := TRUE;
   END_IF;
   IF #_w6 AND #O_Salir_S3 AND NOT #O_Bloqueo THEN
       #Orden_Ejecutada_Jdt := 43;
       #MemoPresenciaJDT := TRUE;
   END_IF;
   IF #_w6 AND #O_Salir_S4 AND NOT #O_Bloqueo THEN
       #Orden_Ejecutada_Jdt := 44;
       #MemoPresenciaJDT := TRUE;
   END_IF;
   #_w7 := #_w2 AND #Moti_INIC;
   IF #_w7 AND #O_Salir_S2 AND NOT #O_Bloqueo THEN
       #Orden_Ejecutada_Jdt := 52;
       #MemoPresenciaJDT := TRUE;
   END_IF;
   IF #_w7 AND #O_Salir_S3 AND NOT #O_Bloqueo THEN
       #Orden_Ejecutada_Jdt := 53;
       #MemoPresenciaJDT := TRUE;
   END_IF;
   IF #_w7 AND #O_Salir_S4 AND NOT #O_Bloqueo THEN
       #Orden_Ejecutada_Jdt := 54;
       #MemoPresenciaJDT := TRUE;
   END_IF;
END_REGION

REGION Network 71: PASAR ETIQUETA JDT
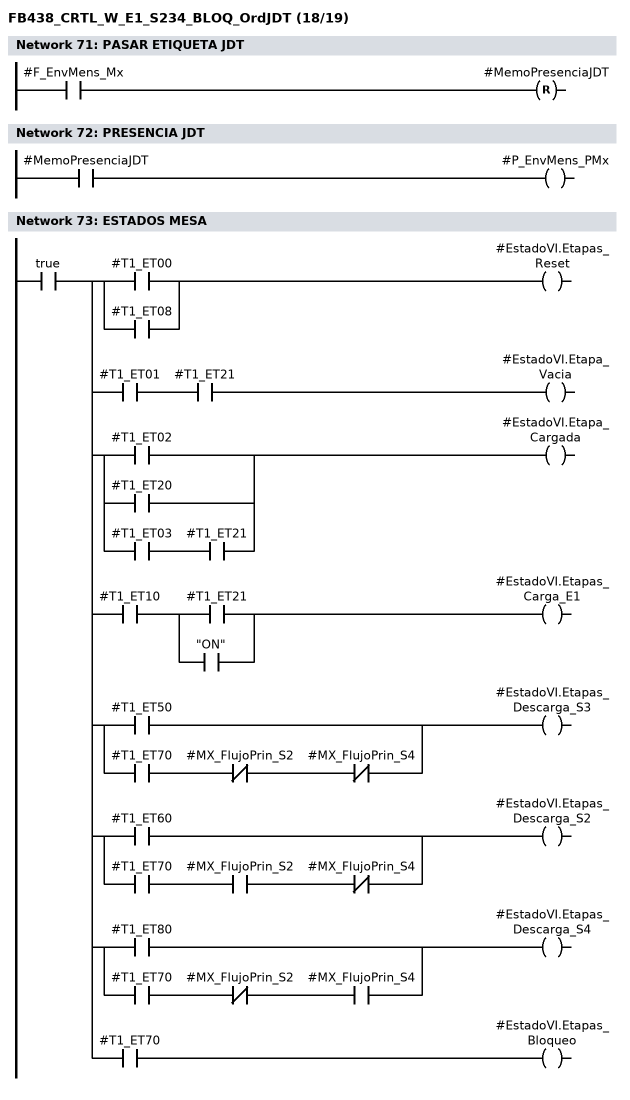
   RUNG wire#powerrail
      Contact( #F_EnvMens_Mx )
      R_Coil( #MemoPresenciaJDT )
   END_RUNG
   // the same network as SCL:
   IF #F_EnvMens_Mx THEN #MemoPresenciaJDT := FALSE; END_IF;
END_REGION

REGION Network 72: PRESENCIA JDT
   RUNG wire#powerrail
      Contact( #MemoPresenciaJDT )
      Coil( #P_EnvMens_PMx )
   END_RUNG
   // the same network as SCL:
   #P_EnvMens_PMx := #MemoPresenciaJDT;
END_REGION

REGION Network 73: ESTADOS MESA
   RUNG wire#powerrail
      Contact( true )
      wire#w1
      Contact( #T1_ET00 )
      wire#w2
      Coil( #EstadoVI.Etapas_Reset )
   END_RUNG
   RUNG wire#w1
      Contact( #T1_ET08 )
   END_RUNG wire#w2
   RUNG wire#w1
      Contact( #T1_ET01 )
      Contact( #T1_ET21 )
      Coil( #EstadoVI.Etapa_Vacia )
   END_RUNG
   RUNG wire#w1
      Contact( #T1_ET02 )
      wire#w3
      Coil( #EstadoVI.Etapa_Cargada )
   END_RUNG
   RUNG wire#w1
      Contact( #T1_ET20 )
   END_RUNG wire#w3
   RUNG wire#w1
      Contact( #T1_ET03 )
      Contact( #T1_ET21 )
   END_RUNG wire#w3
   RUNG wire#w1
      Contact( #T1_ET10 )
      wire#w4
      Contact( #T1_ET21 )
      wire#w5
      Coil( #EstadoVI.Etapas_Carga_E1 )
   END_RUNG
   RUNG wire#w4
      Contact( "ON" )
   END_RUNG wire#w5
   RUNG wire#w1
      Contact( #T1_ET50 )
      wire#w6
      Coil( #EstadoVI.Etapas_Descarga_S3 )
   END_RUNG
   RUNG wire#w1
      Contact( #T1_ET70 )
      I_Contact( #MX_FlujoPrin_S2 )
      I_Contact( #MX_FlujoPrin_S4 )
   END_RUNG wire#w6
   RUNG wire#w1
      Contact( #T1_ET60 )
      wire#w7
      Coil( #EstadoVI.Etapas_Descarga_S2 )
   END_RUNG
   RUNG wire#w1
      Contact( #T1_ET70 )
      Contact( #MX_FlujoPrin_S2 )
      I_Contact( #MX_FlujoPrin_S4 )
   END_RUNG wire#w7
   RUNG wire#w1
      Contact( #T1_ET80 )
      wire#w8
      Coil( #EstadoVI.Etapas_Descarga_S4 )
   END_RUNG
   RUNG wire#w1
      Contact( #T1_ET70 )
      I_Contact( #MX_FlujoPrin_S2 )
      Contact( #MX_FlujoPrin_S4 )
   END_RUNG wire#w8
   RUNG wire#w1
      Contact( #T1_ET70 )
      Coil( #EstadoVI.Etapas_Bloqueo )
   END_RUNG
   // the same network as SCL:
   #EstadoVI.Etapas_Reset := true AND (#T1_ET00 OR #T1_ET08);
   #EstadoVI.Etapa_Vacia := true AND #T1_ET01 AND #T1_ET21;
   #EstadoVI.Etapa_Cargada := true AND (#T1_ET02 OR #T1_ET20 OR (#T1_ET03 AND #T1_ET21));
   #EstadoVI.Etapas_Carga_E1 := true AND #T1_ET10 AND (#T1_ET21 OR "ON");
   #EstadoVI.Etapas_Descarga_S3 := true AND (#T1_ET50 OR (#T1_ET70 AND NOT #MX_FlujoPrin_S2 AND NOT #MX_FlujoPrin_S4));
   #EstadoVI.Etapas_Descarga_S2 := true AND (#T1_ET60 OR (#T1_ET70 AND #MX_FlujoPrin_S2 AND NOT #MX_FlujoPrin_S4));
   #EstadoVI.Etapas_Descarga_S4 := true AND (#T1_ET80 OR (#T1_ET70 AND NOT #MX_FlujoPrin_S2 AND #MX_FlujoPrin_S4));
   #EstadoVI.Etapas_Bloqueo := true AND #T1_ET70;
END_REGION

REGION Network 74: Entradas Mesas
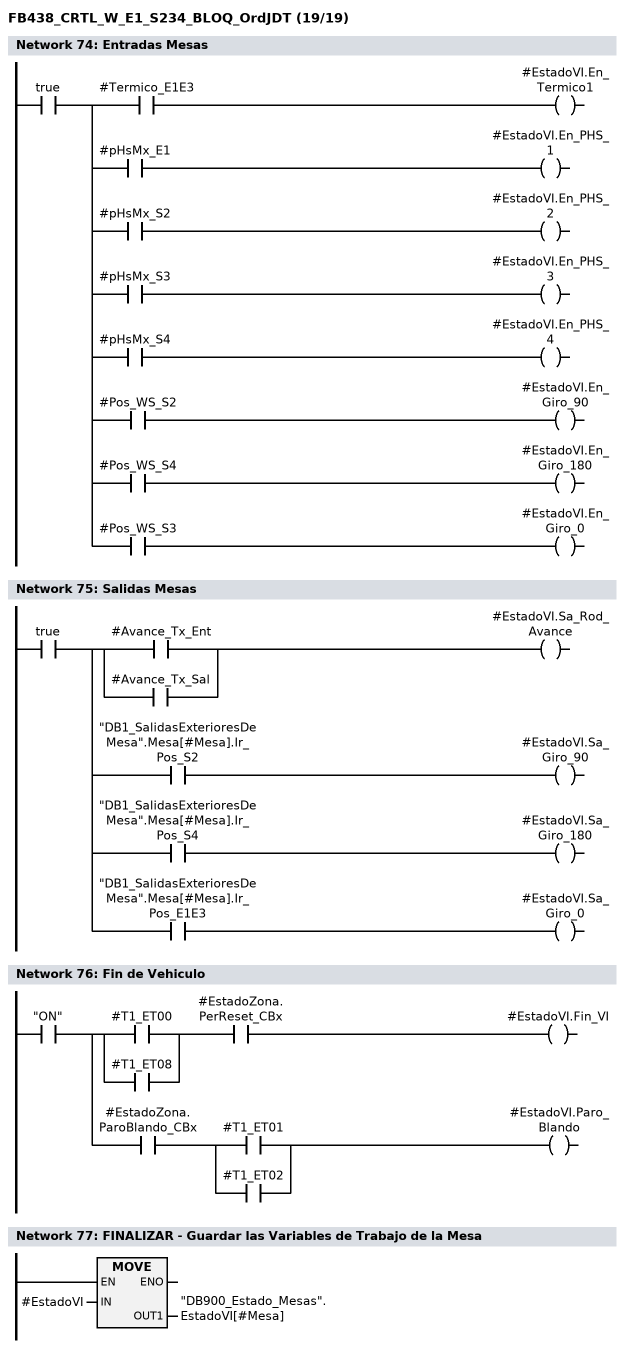
   RUNG wire#powerrail
      Contact( true )
      wire#w1
      Contact( #Termico_E1E3 )
      Coil( #EstadoVI.En_Termico1 )
   END_RUNG
   RUNG wire#w1
      Contact( #pHsMx_E1 )
      Coil( #EstadoVI.En_PHS_1 )
   END_RUNG
   RUNG wire#w1
      Contact( #pHsMx_S2 )
      Coil( #EstadoVI.En_PHS_2 )
   END_RUNG
   RUNG wire#w1
      Contact( #pHsMx_S3 )
      Coil( #EstadoVI.En_PHS_3 )
   END_RUNG
   RUNG wire#w1
      Contact( #pHsMx_S4 )
      Coil( #EstadoVI.En_PHS_4 )
   END_RUNG
   RUNG wire#w1
      Contact( #Pos_WS_S2 )
      Coil( #EstadoVI.En_Giro_90 )
   END_RUNG
   RUNG wire#w1
      Contact( #Pos_WS_S4 )
      Coil( #EstadoVI.En_Giro_180 )
   END_RUNG
   RUNG wire#w1
      Contact( #Pos_WS_S3 )
      Coil( #EstadoVI.En_Giro_0 )
   END_RUNG
   // the same network as SCL:
   #EstadoVI.En_Termico1 := true AND #Termico_E1E3;
   #EstadoVI.En_PHS_1 := true AND #pHsMx_E1;
   #EstadoVI.En_PHS_2 := true AND #pHsMx_S2;
   #EstadoVI.En_PHS_3 := true AND #pHsMx_S3;
   #EstadoVI.En_PHS_4 := true AND #pHsMx_S4;
   #EstadoVI.En_Giro_90 := true AND #Pos_WS_S2;
   #EstadoVI.En_Giro_180 := true AND #Pos_WS_S4;
   #EstadoVI.En_Giro_0 := true AND #Pos_WS_S3;
END_REGION

REGION Network 75: Salidas Mesas
   RUNG wire#powerrail
      Contact( true )
      wire#w1
      Contact( #Avance_Tx_Ent )
      wire#w2
      Coil( #EstadoVI.Sa_Rod_Avance )
   END_RUNG
   RUNG wire#w1
      Contact( #Avance_Tx_Sal )
   END_RUNG wire#w2
   RUNG wire#w1
      Contact( "DB1_SalidasExterioresDeMesa".Mesa[#Mesa].Ir_Pos_S2 )
      Coil( #EstadoVI.Sa_Giro_90 )
   END_RUNG
   RUNG wire#w1
      Contact( "DB1_SalidasExterioresDeMesa".Mesa[#Mesa].Ir_Pos_S4 )
      Coil( #EstadoVI.Sa_Giro_180 )
   END_RUNG
   RUNG wire#w1
      Contact( "DB1_SalidasExterioresDeMesa".Mesa[#Mesa].Ir_Pos_E1E3 )
      Coil( #EstadoVI.Sa_Giro_0 )
   END_RUNG
   // the same network as SCL:
   #EstadoVI.Sa_Rod_Avance := true AND (#Avance_Tx_Ent OR #Avance_Tx_Sal);
   #EstadoVI.Sa_Giro_90 := true AND "DB1_SalidasExterioresDeMesa".Mesa[#Mesa].Ir_Pos_S2;
   #EstadoVI.Sa_Giro_180 := true AND "DB1_SalidasExterioresDeMesa".Mesa[#Mesa].Ir_Pos_S4;
   #EstadoVI.Sa_Giro_0 := true AND "DB1_SalidasExterioresDeMesa".Mesa[#Mesa].Ir_Pos_E1E3;
END_REGION

REGION Network 76: Fin de Vehiculo
   RUNG wire#powerrail
      Contact( "ON" )
      wire#w1
      Contact( #T1_ET00 )
      wire#w2
      Contact( #EstadoZona.PerReset_CBx )
      Coil( #EstadoVI.Fin_VI )
   END_RUNG
   RUNG wire#w1
      Contact( #T1_ET08 )
   END_RUNG wire#w2
   RUNG wire#w1
      Contact( #EstadoZona.ParoBlando_CBx )
      wire#w3
      Contact( #T1_ET01 )
      wire#w4
      Coil( #EstadoVI.Paro_Blando )
   END_RUNG
   RUNG wire#w3
      Contact( #T1_ET02 )
   END_RUNG wire#w4
   // the same network as SCL:
   #EstadoVI.Fin_VI := "ON" AND (#T1_ET00 OR #T1_ET08) AND #EstadoZona.PerReset_CBx;
   #EstadoVI.Paro_Blando := "ON" AND #EstadoZona.ParoBlando_CBx AND (#T1_ET01 OR #T1_ET02);
END_REGION

REGION Network 77: FINALIZAR - Guardar las Variables de Trabajo de la Mesa
   RUNG wire#powerrail
      Move(in := #EstadoVI, out1 => "DB900_Estado_Mesas".EstadoVI[#Mesa])
   END_RUNG
   // the same network as SCL:
   "DB900_Estado_Mesas".EstadoVI[#Mesa] := #EstadoVI;
END_REGION
END_FUNCTION_BLOCK
